REGION Network 8: IMMEDIATE STOP & STOP END OF CYCLE ALARMS
   RUNG wire#powerrail
      I_Contact( #interlocksDB.PROGRAM_SELCT_ALARM )
      Not()
      { S7_GenerateENO := "TRUE" } Move(in := #DB_NUMBER, out1 => "DB440_MACHINE_ALARM_DECODING".GLOBAL_ALARMS_MACHINE.ALARM_DECODING)
      wire#w1
      { S7_Templates := "SrcType := Int" } EQ_Contact(in1 := #CHANNEL, in2 := 1)
      wire#w2
      S_Coil( "DB440_MACHINE_ALARM_DECODING".ALARMS_UNIT_1.ST0_TRANSFER.IS_SEOC_ALARMS )
   END_RUNG
   RUNG wire#w2
      S_Coil( "DB440_MACHINE_ALARM_DECODING".ALARMS_UNIT_1.ST1_LOAD_UNLOAD.IS_SEOC_ALARMS )
   END_RUNG
   RUNG wire#w1
      { S7_Templates := "SrcType := Int" } EQ_Contact(in1 := #CHANNEL, in2 := 2)
      S_Coil( "DB440_MACHINE_ALARM_DECODING".ALARMS_UNIT_1.ST3_CLADDING.IS_SEOC_ALARMS )
   END_RUNG
   RUNG wire#w1
      { S7_Templates := "SrcType := Int" } EQ_Contact(in1 := #CHANNEL, in2 := 3)
      S_Coil( "DB440_MACHINE_ALARM_DECODING".ALARMS_UNIT_1.ST4_CLEANING.IS_SEOC_ALARMS )
   END_RUNG
   RUNG wire#w1
      { S7_Templates := "SrcType := Int" } EQ_Contact(in1 := #CHANNEL, in2 := 4)
      wire#w3
      S_Coil( "DB440_MACHINE_ALARM_DECODING".ALARMS_UNIT_2.ST0_TRANSFER.IS_SEOC_ALARMS )
   END_RUNG
   RUNG wire#w3
      S_Coil( "DB440_MACHINE_ALARM_DECODING".ALARMS_UNIT_2.ST1_LOAD_UNLOAD.IS_SEOC_ALARMS )
   END_RUNG
   RUNG wire#w1
      { S7_Templates := "SrcType := Int" } EQ_Contact(in1 := #CHANNEL, in2 := 5)
      S_Coil( "DB440_MACHINE_ALARM_DECODING".ALARMS_UNIT_2.ST2_MEASURING.IS_SEOC_ALARMS )
   END_RUNG
   RUNG wire#w1
      { S7_Templates := "SrcType := Int" } EQ_Contact(in1 := #CHANNEL, in2 := 6)
      S_Coil( "DB440_MACHINE_ALARM_DECODING".ALARMS_UNIT_2.ST3_CLADDING.IS_SEOC_ALARMS )
   END_RUNG
   RUNG wire#w1
      { S7_Templates := "SrcType := Int" } EQ_Contact(in1 := #CHANNEL, in2 := 7)
      S_Coil( "DB440_MACHINE_ALARM_DECODING".ALARMS_UNIT_2.ST4_CLEANING.IS_SEOC_ALARMS )
   END_RUNG
   RUNG wire#w1
      { S7_Templates := "SrcType := Int" } EQ_Contact(in1 := #CHANNEL, in2 := 8)
      S_Coil( "DB440_MACHINE_ALARM_DECODING".ALARMS_UNIT_3.IS_SEOC_ALARMS )
   END_RUNG
   RUNG wire#w1
      { S7_Templates := "SrcType := Int" } EQ_Contact(in1 := #CHANNEL, in2 := 9)
      S_Coil( "DB440_MACHINE_ALARM_DECODING".ALARMS_UNIT_4.IS_SEOC_ALARMS )
   END_RUNG
   // the same network as SCL:
   // ENO of a box is taken as its EN; it also drops when the box reports an error
   #_w1 := NOT (NOT #interlocksDB.PROGRAM_SELCT_ALARM);
   IF #_w1 THEN "DB440_MACHINE_ALARM_DECODING".GLOBAL_ALARMS_MACHINE.ALARM_DECODING := #DB_NUMBER; END_IF;
   IF #_w1 AND (#CHANNEL = 1) THEN
       "DB440_MACHINE_ALARM_DECODING".ALARMS_UNIT_1.ST0_TRANSFER.IS_SEOC_ALARMS := TRUE;
       "DB440_MACHINE_ALARM_DECODING".ALARMS_UNIT_1.ST1_LOAD_UNLOAD.IS_SEOC_ALARMS := TRUE;
   END_IF;
   IF #_w1 AND (#CHANNEL = 2) THEN
       "DB440_MACHINE_ALARM_DECODING".ALARMS_UNIT_1.ST3_CLADDING.IS_SEOC_ALARMS := TRUE;
   END_IF;
   IF #_w1 AND (#CHANNEL = 3) THEN
       "DB440_MACHINE_ALARM_DECODING".ALARMS_UNIT_1.ST4_CLEANING.IS_SEOC_ALARMS := TRUE;
   END_IF;
   IF #_w1 AND (#CHANNEL = 4) THEN
       "DB440_MACHINE_ALARM_DECODING".ALARMS_UNIT_2.ST0_TRANSFER.IS_SEOC_ALARMS := TRUE;
       "DB440_MACHINE_ALARM_DECODING".ALARMS_UNIT_2.ST1_LOAD_UNLOAD.IS_SEOC_ALARMS := TRUE;
   END_IF;
   IF #_w1 AND (#CHANNEL = 5) THEN
       "DB440_MACHINE_ALARM_DECODING".ALARMS_UNIT_2.ST2_MEASURING.IS_SEOC_ALARMS := TRUE;
   END_IF;
   IF #_w1 AND (#CHANNEL = 6) THEN
       "DB440_MACHINE_ALARM_DECODING".ALARMS_UNIT_2.ST3_CLADDING.IS_SEOC_ALARMS := TRUE;
   END_IF;
   IF #_w1 AND (#CHANNEL = 7) THEN
       "DB440_MACHINE_ALARM_DECODING".ALARMS_UNIT_2.ST4_CLEANING.IS_SEOC_ALARMS := TRUE;
   END_IF;
   IF #_w1 AND (#CHANNEL = 8) THEN
       "DB440_MACHINE_ALARM_DECODING".ALARMS_UNIT_3.IS_SEOC_ALARMS := TRUE;
   END_IF;
   IF #_w1 AND (#CHANNEL = 9) THEN
       "DB440_MACHINE_ALARM_DECODING".ALARMS_UNIT_4.IS_SEOC_ALARMS := TRUE;
   END_IF;
END_REGION

REGION Network 9: PROGRAMMING ALARM
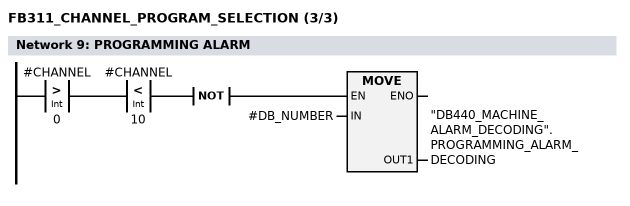
   RUNG wire#powerrail
      { S7_Templates := "SrcType := Int" } GT_Contact(in1 := #CHANNEL, in2 := 0)
      { S7_Templates := "SrcType := Int" } LT_Contact(in1 := #CHANNEL, in2 := 10)
      Not()
      Move(in := #DB_NUMBER, out1 => "DB440_MACHINE_ALARM_DECODING".PROGRAMMING_ALARM_DECODING)
   END_RUNG
   // the same network as SCL:
   IF NOT ((#CHANNEL > 0) AND (#CHANNEL < 10)) THEN
       "DB440_MACHINE_ALARM_DECODING".PROGRAMMING_ALARM_DECODING := #DB_NUMBER;
   END_IF;
END_REGION
END_FUNCTION_BLOCK

FUNCTION_BLOCK "FB321_CHANNEL"   // FB321, LAD
{ S7_Optimized_Access := 'FALSE' }
AUTHOR : ETXETAR
VERSION : 1.0
// stored: AutoNumber false, IsIECCheckEnabled false, SetENOAutomatically false, UDAEnableTagReadback false
   VAR_INPUT
      CHANNEL_MODE_GROUP : Int;   // CHANNEL MODE GROUP
      JERK_PARAMETERS_ENABLE { ExternalAccessible := 'False'; ExternalVisible := 'False'; ExternalWritable := 'False'} : Bool;   // JERK PARAMETERS ENABLE
      ENABLE_M01 { ExternalAccessible := 'False'; ExternalVisible := 'False'; ExternalWritable := 'False'} : Bool;   // ENABLE M01
      ENABLE_DRY_RUN_TEST_PRGM { ExternalAccessible := 'False'; ExternalVisible := 'False'; ExternalWritable := 'False'} : Bool;   // ENABLE DRY RUN TEST PRGM
      FEED_DISABLE { ExternalAccessible := 'False'; ExternalVisible := 'False'; ExternalWritable := 'False'} : Bool;   // FEED DISABLE
      ENABLE_OVERRIDE { ExternalAccessible := 'False'; ExternalVisible := 'False'; ExternalWritable := 'False'} : Bool;   // OVERRIDE 0 OR 100 =0 // OVERRIDE ENABLED =1
      ENABLE_OVERRIDE_FROM_MP_OR_HT10 { ExternalAccessible := 'False'; ExternalVisible := 'False'; ExternalWritable := 'False'} : Bool;   // ENABLE OVERRIDE FROM MAIN PANEL OR HT10, TRUE = YES, FALSE = NO (VALUE IS OBTAINED FROM AN HMI SCREEN OR ANOTHER DEVICE)
      OVERRIDE_VALUE : Byte;   // OVERRIDE VALUE
      BA3_SOFTKEYS_STOP { ExternalAccessible := 'False'; ExternalVisible := 'False'; ExternalWritable := 'False'} : Bool;   // BA3 SOFTKEYS STOP
      PROG_SLECT_FAULT_CH { ExternalAccessible := 'False'; ExternalVisible := 'False'; ExternalWritable := 'False'} : Bool;   // N.O / PROGRAM SELECTION FAULT CH
      MACHINE_IS_ALARMS : Bool;   // MACHINE IS ALARMS
      MACHINE_IS_WARNINGS : Bool;   // MACHINE IS WARNINGS
      UNIT_IS_SEOC { ExternalAccessible := 'False'; ExternalVisible := 'False'; ExternalWritable := 'False'} : Bool;   // UNIT IS SEOC
      CHANNEL_M201 { ExternalAccessible := 'False'; ExternalVisible := 'False'; ExternalWritable := 'False'} : Bool;   // CHANNEL M201
      CHANNEL_MCH_RESET : Bool;   // CHANNEL MACHINE RESET
      NC_START_DUMMY_FOR_OPT { ExternalAccessible := 'False'; ExternalVisible := 'False'; ExternalWritable := 'False'} : Bool;   // NC START DUMMY FOR OPTIMIZATION
      MPP_PUSH_BUTTON_START { ExternalAccessible := 'False'; ExternalVisible := 'False'; ExternalWritable := 'False'} : Bool;   // MPP PUSH BUTTON START
      MPP_PUSH_BUTTON_NC_START : Bool;   // MPP PUSH BUTTON NC START
      MPP_BUTTON_HOME_POS { ExternalAccessible := 'False'; ExternalVisible := 'False'; ExternalWritable := 'False'} : Bool;   // MPP BUTTON HOME POSITION
      UNIT_HOME_STEP_3 { ExternalAccessible := 'False'; ExternalVisible := 'False'; ExternalWritable := 'False'} : Bool;   // UNIT HOME STEP 3
      UNIT_CYCLE_STEP_3 { ExternalAccessible := 'False'; ExternalVisible := 'False'; ExternalWritable := 'False'} : Bool;   // UNIT CYCLE STEP 3
   END_VAR
   VAR_OUTPUT
      "CH_NOT_IN SOFT_MODE_ALARM" { ExternalAccessible := 'False'; ExternalVisible := 'False'; ExternalWritable := 'False'} : Bool;   // CHANNEL NOT IN SOFT MODE ALARM
   END_VAR
   VAR_IN_OUT
      ChannelDB : "LBP_typeChanX";
   END_VAR
   VAR DB_SPECIFIC
      CH_NOT_IN_SOFT_MODE { ExternalAccessible := 'False'; ExternalVisible := 'False'; ExternalWritable := 'False'} : Bool;   // CHANNEL NOT IN SOFT MODE
      RESET_CH { ExternalAccessible := 'False'; ExternalVisible := 'False'; ExternalWritable := 'False'} : Bool;   // RESET CHANNEL
      START_CH { ExternalAccessible := 'False'; ExternalVisible := 'False'; ExternalWritable := 'False'} : Bool;   // START CHANNEL
      RESET_AUX { ExternalAccessible := 'False'; ExternalVisible := 'False'; ExternalWritable := 'False'} : Bool;   // RESET AUX
      RESET_1 { ExternalAccessible := 'False'; ExternalVisible := 'False'; ExternalWritable := 'False'} : Bool;   // RESET 1
      RESET_2 { ExternalAccessible := 'False'; ExternalVisible := 'False'; ExternalWritable := 'False'} : Bool;   // RESET 2
      PULSE { ExternalAccessible := 'False'; ExternalVisible := 'False'; ExternalWritable := 'False'} : Bool;   // PULSE
      TIMER_CH_NOT_IN_SOFT_MODE { ExternalAccessible := 'False'; ExternalVisible := 'False'; ExternalWritable := 'False'; S7_SetPoint := 'True'} : TON_TIME;   // CHANNEL NOT IN SOFT MODE TIMER
   END_VAR
   VAR_TEMP
      DB_NUMBER : DInt;   // DB NUMBER FOR ALARM AND HELP DECODING
      CHANNEL_NUM : Int;   // CHANNEL NUMBER
   END_VAR
   // TIMER_CH_NOT_IN_SOFT_MODE.PT := T#1s;
   VAR_TEMP   // added for the SCL form of the ladder/FBD networks
      _w1 : Bool;
      _w2 : Bool;
   END_VAR
BEGIN

NETWORK
TITLE = READ INSTANCE DB
      L     DINO;
      +     10#800000;
      T     #DB_NUMBER;
//READ CHANNEL NUMBER
      L     DINO;
      L     10#320;
      -I;
      T     #CHANNEL_NUM;


REGION Network 2: ACTIVATE SINGLE BLOCK / ENABLE SINGLE BLOCK
   // Step by Step mode
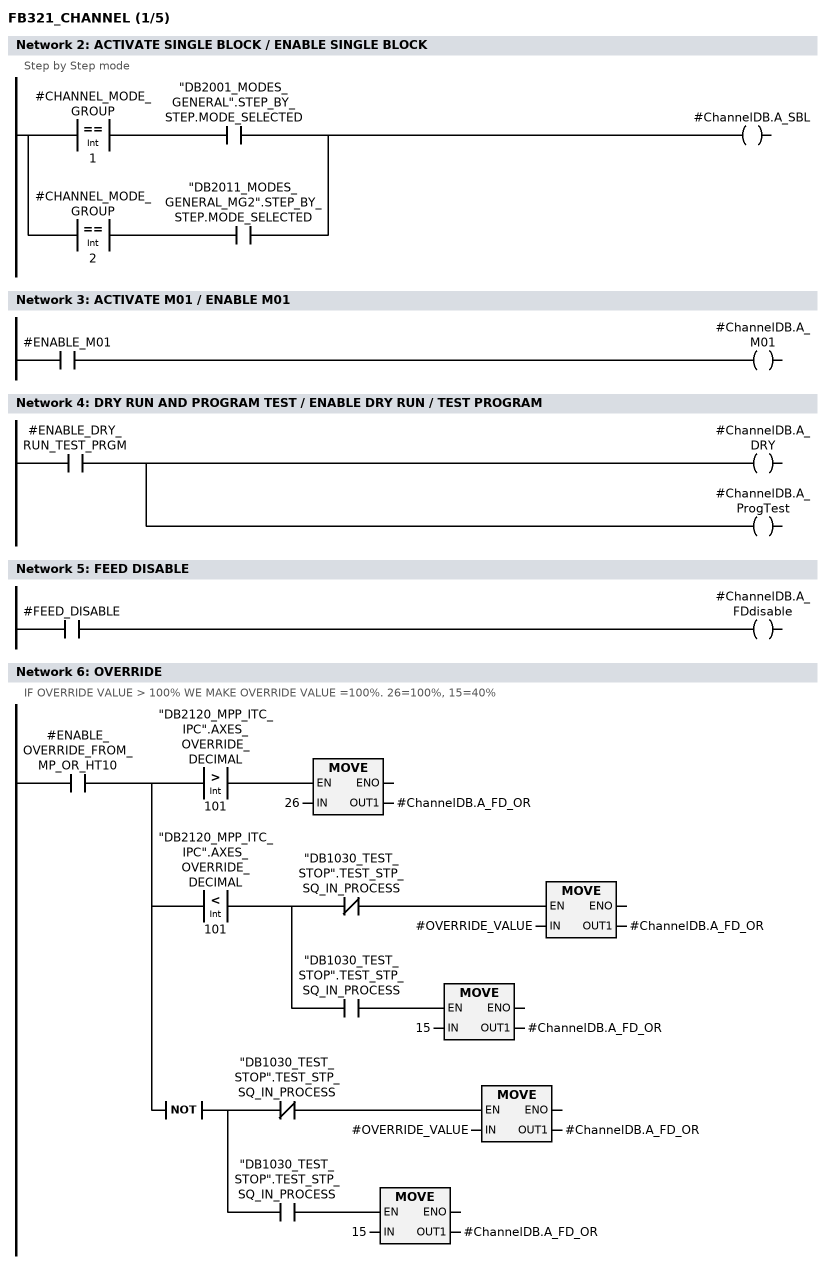
   RUNG wire#powerrail
      { S7_Templates := "SrcType := Int" } EQ_Contact(in1 := #CHANNEL_MODE_GROUP, in2 := 1)
      Contact( "DB2001_MODES_GENERAL".STEP_BY_STEP.MODE_SELECTED )
      wire#w1
      Coil( #ChannelDB.A_SBL )
   END_RUNG
   RUNG wire#powerrail
      { S7_Templates := "SrcType := Int" } EQ_Contact(in1 := #CHANNEL_MODE_GROUP, in2 := 2)
      Contact( "DB2011_MODES_GENERAL_MG2".STEP_BY_STEP.MODE_SELECTED )
   END_RUNG wire#w1
   // the same network as SCL:
   #ChannelDB.A_SBL := ((#CHANNEL_MODE_GROUP = 1) AND "DB2001_MODES_GENERAL".STEP_BY_STEP.MODE_SELECTED) OR ((#CHANNEL_MODE_GROUP = 2) AND "DB2011_MODES_GENERAL_MG2".STEP_BY_STEP.MODE_SELECTED);
END_REGION

REGION Network 3: ACTIVATE M01 / ENABLE M01
   RUNG wire#powerrail
      Contact( #ENABLE_M01 )
      Coil( #ChannelDB.A_M01 )
   END_RUNG
   // the same network as SCL:
   #ChannelDB.A_M01 := #ENABLE_M01;
END_REGION

REGION Network 4: DRY RUN AND PROGRAM TEST / ENABLE DRY RUN / TEST PROGRAM
   RUNG wire#powerrail
      Contact( #ENABLE_DRY_RUN_TEST_PRGM )
      wire#w1
      Coil( #ChannelDB.A_DRY )
   END_RUNG
   RUNG wire#w1
      Coil( #ChannelDB.A_ProgTest )
   END_RUNG
   // the same network as SCL:
   #ChannelDB.A_DRY := #ENABLE_DRY_RUN_TEST_PRGM;
   #ChannelDB.A_ProgTest := #ENABLE_DRY_RUN_TEST_PRGM;
END_REGION

REGION Network 5: FEED DISABLE
   RUNG wire#powerrail
      Contact( #FEED_DISABLE )
      Coil( #ChannelDB.A_FDdisable )
   END_RUNG
   // the same network as SCL:
   #ChannelDB.A_FDdisable := #FEED_DISABLE;
END_REGION

REGION Network 6: OVERRIDE
   // IF OVERRIDE VALUE > 100% WE MAKE OVERRIDE VALUE =100%. 26=100%, 15=40%
   RUNG wire#powerrail
      Contact( #ENABLE_OVERRIDE_FROM_MP_OR_HT10 )
      wire#w1
      { S7_Templates := "SrcType := Int" } GT_Contact(in1 := "DB2120_MPP_ITC_IPC".AXES_OVERRIDE_DECIMAL, in2 := 101)
      { S7_GenerateENO := "TRUE" } Move(in := 26, out1 => #ChannelDB.A_FD_OR)
   END_RUNG
   RUNG wire#w1
      { S7_Templates := "SrcType := Int" } LT_Contact(in1 := "DB2120_MPP_ITC_IPC".AXES_OVERRIDE_DECIMAL, in2 := 101)
      wire#w2
      I_Contact( "DB1030_TEST_STOP".TEST_STP_SQ_IN_PROCESS )
      { S7_GenerateENO := "TRUE" } Move(in := #OVERRIDE_VALUE, out1 => #ChannelDB.A_FD_OR)
   END_RUNG
   RUNG wire#w2
      Contact( "DB1030_TEST_STOP".TEST_STP_SQ_IN_PROCESS )
      { S7_GenerateENO := "TRUE" } Move(in := 15, out1 => #ChannelDB.A_FD_OR)
   END_RUNG
   RUNG wire#w1
      Not()
      wire#w3
      I_Contact( "DB1030_TEST_STOP".TEST_STP_SQ_IN_PROCESS )
      { S7_GenerateENO := "TRUE" } Move(in := #OVERRIDE_VALUE, out1 => #ChannelDB.A_FD_OR)
   END_RUNG
   RUNG wire#w3
      Contact( "DB1030_TEST_STOP".TEST_STP_SQ_IN_PROCESS )
      { S7_GenerateENO := "TRUE" } Move(in := 15, out1 => #ChannelDB.A_FD_OR)
   END_RUNG
   // the same network as SCL:
   IF #ENABLE_OVERRIDE_FROM_MP_OR_HT10 AND ("DB2120_MPP_ITC_IPC".AXES_OVERRIDE_DECIMAL > 101) THEN
       #ChannelDB.A_FD_OR := 26;
   END_IF;
   #_w1 := #ENABLE_OVERRIDE_FROM_MP_OR_HT10 AND ("DB2120_MPP_ITC_IPC".AXES_OVERRIDE_DECIMAL < 101);
   IF #_w1 AND NOT "DB1030_TEST_STOP".TEST_STP_SQ_IN_PROCESS THEN
       #ChannelDB.A_FD_OR := #OVERRIDE_VALUE;
   END_IF;
   IF #_w1 AND "DB1030_TEST_STOP".TEST_STP_SQ_IN_PROCESS THEN #ChannelDB.A_FD_OR := 15; END_IF;
   #_w2 := NOT #ENABLE_OVERRIDE_FROM_MP_OR_HT10;
   IF #_w2 AND NOT "DB1030_TEST_STOP".TEST_STP_SQ_IN_PROCESS THEN
       #ChannelDB.A_FD_OR := #OVERRIDE_VALUE;
   END_IF;
   IF #_w2 AND "DB1030_TEST_STOP".TEST_STP_SQ_IN_PROCESS THEN #ChannelDB.A_FD_OR := 15; END_IF;
END_REGION

REGION Network 7: OVERRIDE ACTIVE / FEEDRATE OVERRIDE ACTIVE
   // REMOVE DUMMY ON IF REQUIRED
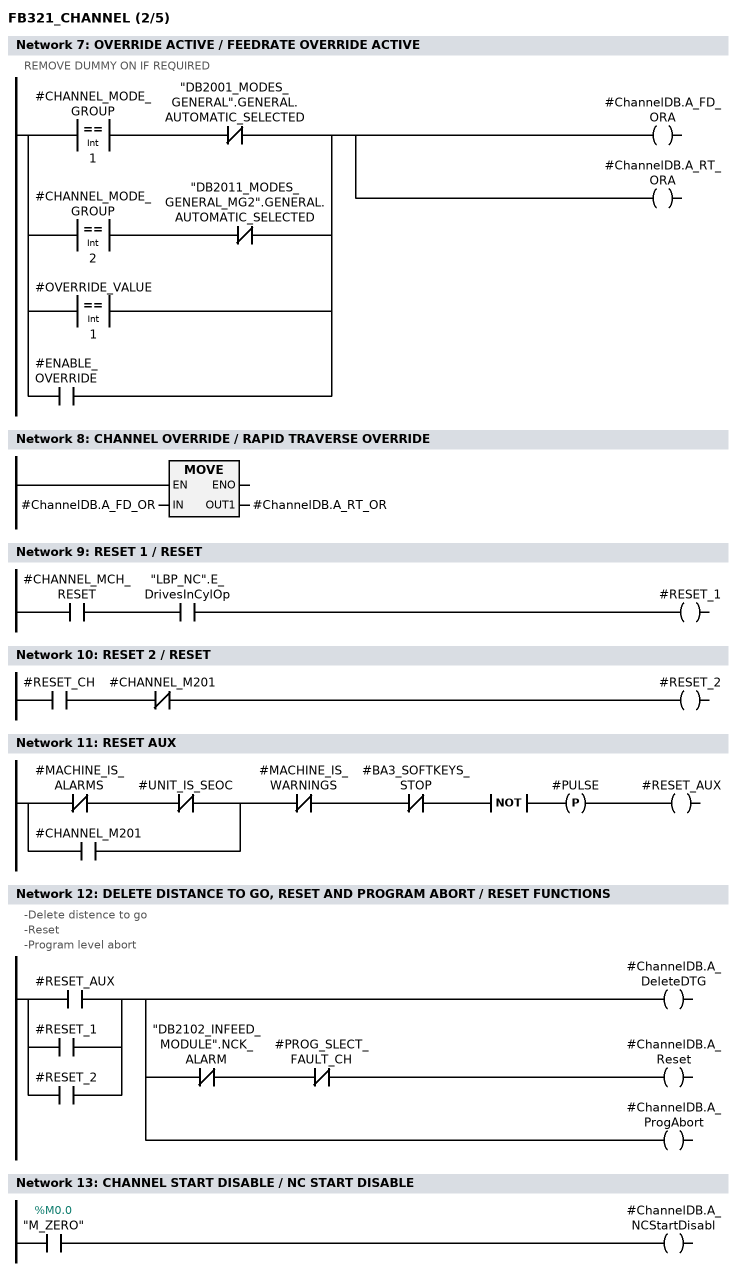
   RUNG wire#powerrail
      { S7_Templates := "SrcType := Int" } EQ_Contact(in1 := #CHANNEL_MODE_GROUP, in2 := 1)
      I_Contact( "DB2001_MODES_GENERAL".GENERAL.AUTOMATIC_SELECTED )
      wire#w1
      Coil( #ChannelDB.A_FD_ORA )
   END_RUNG
   RUNG wire#powerrail
      { S7_Templates := "SrcType := Int" } EQ_Contact(in1 := #CHANNEL_MODE_GROUP, in2 := 2)
      I_Contact( "DB2011_MODES_GENERAL_MG2".GENERAL.AUTOMATIC_SELECTED )
   END_RUNG wire#w1
   RUNG wire#powerrail
      { S7_Templates := "SrcType := Int" } EQ_Contact(in1 := #OVERRIDE_VALUE, in2 := 1)
   END_RUNG wire#w1
   RUNG wire#powerrail
      Contact( #ENABLE_OVERRIDE )
   END_RUNG wire#w1
   RUNG wire#w1
      Coil( #ChannelDB.A_RT_ORA )
   END_RUNG
   // the same network as SCL:
   #ChannelDB.A_FD_ORA := ((#CHANNEL_MODE_GROUP = 1) AND NOT "DB2001_MODES_GENERAL".GENERAL.AUTOMATIC_SELECTED) OR ((#CHANNEL_MODE_GROUP = 2) AND NOT "DB2011_MODES_GENERAL_MG2".GENERAL.AUTOMATIC_SELECTED) OR (#OVERRIDE_VALUE = 1) OR #ENABLE_OVERRIDE;
   #ChannelDB.A_RT_ORA := #ChannelDB.A_FD_ORA;
END_REGION

REGION Network 8: CHANNEL OVERRIDE / RAPID TRAVERSE OVERRIDE
   RUNG wire#powerrail
      { S7_GenerateENO := "TRUE" } Move(in := #ChannelDB.A_FD_OR, out1 => #ChannelDB.A_RT_OR)
   END_RUNG
   // the same network as SCL:
   #ChannelDB.A_RT_OR := #ChannelDB.A_FD_OR;
END_REGION

REGION Network 9: RESET 1 / RESET
   RUNG wire#powerrail
      Contact( #CHANNEL_MCH_RESET )
      Contact( "LBP_NC".E_DrivesInCylOp )
      Coil( #RESET_1 )
   END_RUNG
   // the same network as SCL:
   #RESET_1 := #CHANNEL_MCH_RESET AND "LBP_NC".E_DrivesInCylOp;
END_REGION

REGION Network 10: RESET 2 / RESET
   RUNG wire#powerrail
      Contact( #RESET_CH )
      I_Contact( #CHANNEL_M201 )
      Coil( #RESET_2 )
   END_RUNG
   // the same network as SCL:
   #RESET_2 := #RESET_CH AND NOT #CHANNEL_M201;
END_REGION

REGION Network 11: RESET AUX
   RUNG wire#powerrail
      I_Contact( #MACHINE_IS_ALARMS )
      I_Contact( #UNIT_IS_SEOC )
      wire#w1
      I_Contact( #MACHINE_IS_WARNINGS )
      I_Contact( #BA3_SOFTKEYS_STOP )
      Not()
      P_Trig( #PULSE )
      Coil( #RESET_AUX )
   END_RUNG
   RUNG wire#powerrail
      Contact( #CHANNEL_M201 )
   END_RUNG wire#w1
   // the same network as SCL:
   #_w1 := NOT (((NOT #MACHINE_IS_ALARMS AND NOT #UNIT_IS_SEOC) OR #CHANNEL_M201) AND NOT #MACHINE_IS_WARNINGS AND NOT #BA3_SOFTKEYS_STOP);
   #_w2 := #_w1 AND NOT #PULSE;   // rising edge
   #PULSE := #_w1;
   #RESET_AUX := #_w2;
END_REGION

REGION Network 12: DELETE DISTANCE TO GO, RESET AND PROGRAM ABORT / RESET FUNCTIONS
   // -Delete distence to go
   // -Reset
   // -Program level abort
   RUNG wire#powerrail
      Contact( #RESET_AUX )
      wire#w1
      Coil( #ChannelDB.A_DeleteDTG )
   END_RUNG
   RUNG wire#powerrail
      Contact( #RESET_1 )
   END_RUNG wire#w1
   RUNG wire#powerrail
      Contact( #RESET_2 )
   END_RUNG wire#w1
   RUNG wire#w1
      I_Contact( "DB2102_INFEED_MODULE".NCK_ALARM )
      I_Contact( #PROG_SLECT_FAULT_CH )
      Coil( #ChannelDB.A_Reset )
   END_RUNG
   RUNG wire#w1
      Coil( #ChannelDB.A_ProgAbort )
   END_RUNG
   // the same network as SCL:
   #ChannelDB.A_DeleteDTG := #RESET_AUX OR #RESET_1 OR #RESET_2;
   #ChannelDB.A_Reset := #ChannelDB.A_DeleteDTG AND NOT "DB2102_INFEED_MODULE".NCK_ALARM AND NOT #PROG_SLECT_FAULT_CH;
   #ChannelDB.A_ProgAbort := #ChannelDB.A_DeleteDTG;
END_REGION

REGION Network 13: CHANNEL START DISABLE / NC START DISABLE
   RUNG wire#powerrail
      Contact( "M_ZERO" )
      Coil( #ChannelDB.A_NCStartDisabl )
   END_RUNG
   // the same network as SCL:
   #ChannelDB.A_NCStartDisabl := "M_ZERO";
END_REGION

REGION Network 14: START CHANNEL / NC START
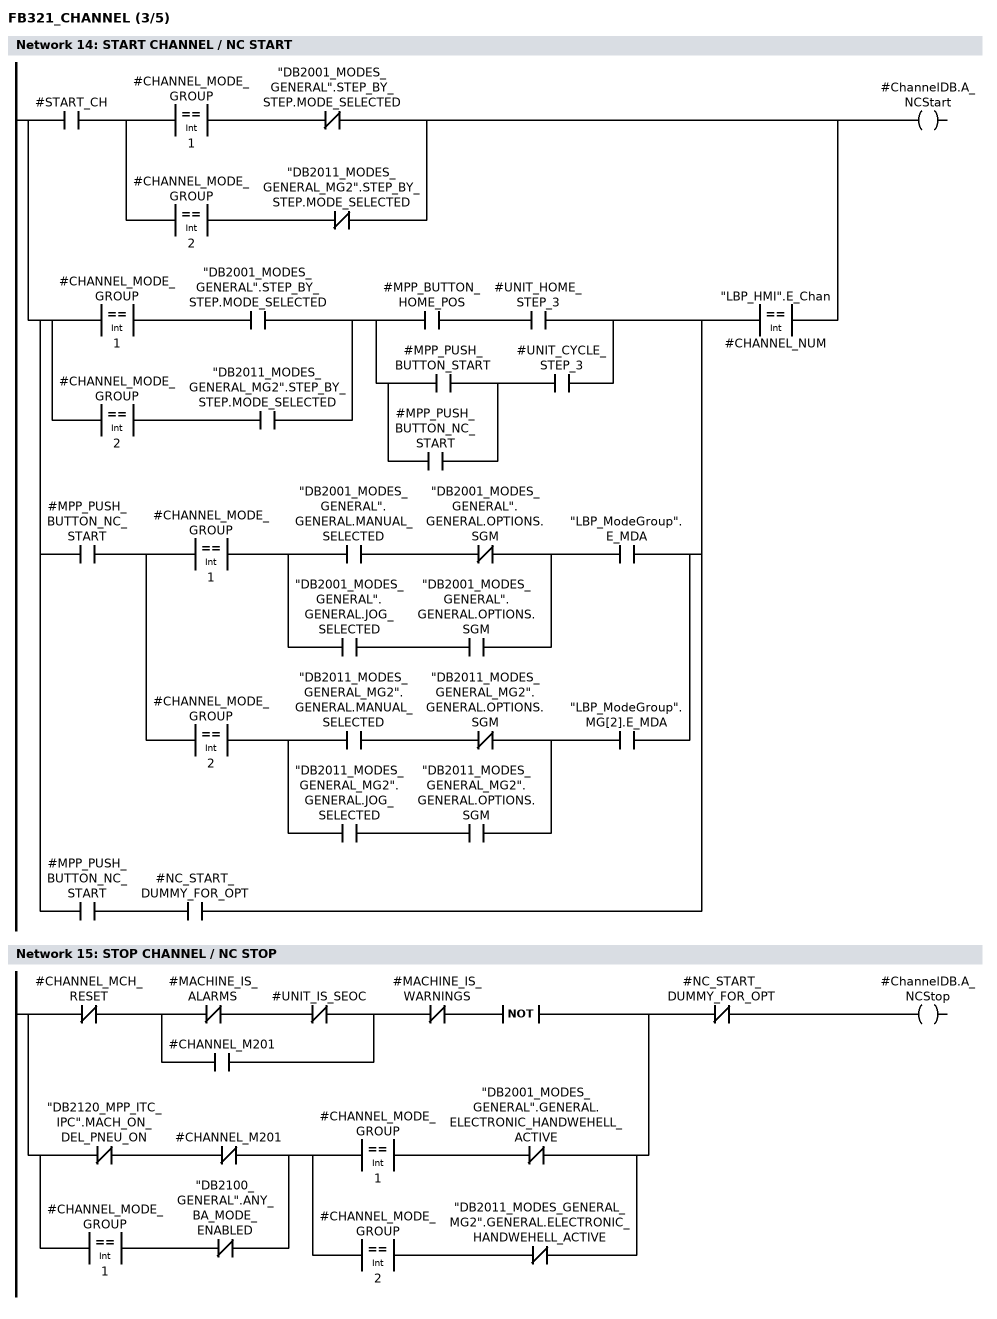
   RUNG wire#powerrail
      Contact( #START_CH )
      wire#w1
      { S7_Templates := "SrcType := Int" } EQ_Contact(in1 := #CHANNEL_MODE_GROUP, in2 := 1)
      I_Contact( "DB2001_MODES_GENERAL".STEP_BY_STEP.MODE_SELECTED )
      wire#w2
      Coil( #ChannelDB.A_NCStart )
   END_RUNG
   RUNG wire#w1
      { S7_Templates := "SrcType := Int" } EQ_Contact(in1 := #CHANNEL_MODE_GROUP, in2 := 2)
      I_Contact( "DB2011_MODES_GENERAL_MG2".STEP_BY_STEP.MODE_SELECTED )
   END_RUNG wire#w2
   RUNG wire#powerrail
      { S7_Templates := "SrcType := Int" } EQ_Contact(in1 := #CHANNEL_MODE_GROUP, in2 := 1)
      Contact( "DB2001_MODES_GENERAL".STEP_BY_STEP.MODE_SELECTED )
      wire#w3
      Contact( #MPP_BUTTON_HOME_POS )
      Contact( #UNIT_HOME_STEP_3 )
      wire#w4
      { S7_Templates := "SrcType := Int" } EQ_Contact(in1 := "LBP_HMI".E_Chan, in2 := #CHANNEL_NUM)
   END_RUNG wire#w2
   RUNG wire#powerrail
      { S7_Templates := "SrcType := Int" } EQ_Contact(in1 := #CHANNEL_MODE_GROUP, in2 := 2)
      Contact( "DB2011_MODES_GENERAL_MG2".STEP_BY_STEP.MODE_SELECTED )
   END_RUNG wire#w3
   RUNG wire#w3
      Contact( #MPP_PUSH_BUTTON_START )
      wire#w5
      Contact( #UNIT_CYCLE_STEP_3 )
   END_RUNG wire#w4
   RUNG wire#w3
      Contact( #MPP_PUSH_BUTTON_NC_START )
   END_RUNG wire#w5
   RUNG wire#powerrail
      Contact( #MPP_PUSH_BUTTON_NC_START )
      wire#w6
      { S7_Templates := "SrcType := Int" } EQ_Contact(in1 := #CHANNEL_MODE_GROUP, in2 := 1)
      wire#w7
      Contact( "DB2001_MODES_GENERAL".GENERAL.MANUAL_SELECTED )
      I_Contact( "DB2001_MODES_GENERAL".GENERAL.OPTIONS.SGM )
      wire#w8
      Contact( "LBP_ModeGroup".E_MDA )
   END_RUNG wire#w4
   RUNG wire#w7
      Contact( "DB2001_MODES_GENERAL".GENERAL.JOG_SELECTED )
      Contact( "DB2001_MODES_GENERAL".GENERAL.OPTIONS.SGM )
   END_RUNG wire#w8
   RUNG wire#w6
      { S7_Templates := "SrcType := Int" } EQ_Contact(in1 := #CHANNEL_MODE_GROUP, in2 := 2)
      wire#w9
      Contact( "DB2011_MODES_GENERAL_MG2".GENERAL.MANUAL_SELECTED )
      I_Contact( "DB2011_MODES_GENERAL_MG2".GENERAL.OPTIONS.SGM )
      wire#w10
      Contact( "LBP_ModeGroup".MG[2].E_MDA )
   END_RUNG wire#w4
   RUNG wire#w9
      Contact( "DB2011_MODES_GENERAL_MG2".GENERAL.JOG_SELECTED )
      Contact( "DB2011_MODES_GENERAL_MG2".GENERAL.OPTIONS.SGM )
   END_RUNG wire#w10
   RUNG wire#powerrail
      Contact( #MPP_PUSH_BUTTON_NC_START )
      Contact( #NC_START_DUMMY_FOR_OPT )
   END_RUNG wire#w4
   // the same network as SCL:
   #ChannelDB.A_NCStart := (#START_CH AND (((#CHANNEL_MODE_GROUP = 1) AND NOT "DB2001_MODES_GENERAL".STEP_BY_STEP.MODE_SELECTED) OR ((#CHANNEL_MODE_GROUP = 2) AND NOT "DB2011_MODES_GENERAL_MG2".STEP_BY_STEP.MODE_SELECTED))) OR ((((((#CHANNEL_MODE_GROUP = 1) AND "DB2001_MODES_GENERAL".STEP_BY_STEP.MODE_SELECTED) OR ((#CHANNEL_MODE_GROUP = 2) AND "DB2011_MODES_GENERAL_MG2".STEP_BY_STEP.MODE_SELECTED)) AND ((#MPP_BUTTON_HOME_POS AND #UNIT_HOME_STEP_3) OR ((#MPP_PUSH_BUTTON_START OR #MPP_PUSH_BUTTON_NC_START) AND #UNIT_CYCLE_STEP_3))) OR (#MPP_PUSH_BUTTON_NC_START AND (((#CHANNEL_MODE_GROUP = 1) AND (("DB2001_MODES_GENERAL".GENERAL.MANUAL_SELECTED AND NOT "DB2001_MODES_GENERAL".GENERAL.OPTIONS.SGM) OR ("DB2001_MODES_GENERAL".GENERAL.JOG_SELECTED AND "DB2001_MODES_GENERAL".GENERAL.OPTIONS.SGM)) AND "LBP_ModeGroup".E_MDA) OR ((#CHANNEL_MODE_GROUP = 2) AND (("DB2011_MODES_GENERAL_MG2".GENERAL.MANUAL_SELECTED AND NOT "DB2011_MODES_GENERAL_MG2".GENERAL.OPTIONS.SGM) OR ("DB2011_MODES_GENERAL_MG2".GENERAL.JOG_SELECTED AND "DB2011_MODES_GENERAL_MG2".GENERAL.OPTIONS.SGM)) AND "LBP_ModeGroup".MG[2].E_MDA))) OR (#MPP_PUSH_BUTTON_NC_START AND #NC_START_DUMMY_FOR_OPT)) AND ("LBP_HMI".E_Chan = #CHANNEL_NUM));
END_REGION

REGION Network 15: STOP CHANNEL / NC STOP
   RUNG wire#powerrail
      I_Contact( #CHANNEL_MCH_RESET )
      wire#w1
      I_Contact( #MACHINE_IS_ALARMS )
      I_Contact( #UNIT_IS_SEOC )
      wire#w2
      I_Contact( #MACHINE_IS_WARNINGS )
      Not()
      wire#w3
      I_Contact( #NC_START_DUMMY_FOR_OPT )
      Coil( #ChannelDB.A_NCStop )
   END_RUNG
   RUNG wire#w1
      Contact( #CHANNEL_M201 )
   END_RUNG wire#w2
   RUNG wire#powerrail
      I_Contact( "DB2120_MPP_ITC_IPC".MACH_ON_DEL_PNEU_ON )
      I_Contact( #CHANNEL_M201 )
      wire#w4
      { S7_Templates := "SrcType := Int" } EQ_Contact(in1 := #CHANNEL_MODE_GROUP, in2 := 1)
      I_Contact( "DB2001_MODES_GENERAL".GENERAL.ELECTRONIC_HANDWEHELL_ACTIVE )
   END_RUNG wire#w3
   RUNG wire#powerrail
      { S7_Templates := "SrcType := Int" } EQ_Contact(in1 := #CHANNEL_MODE_GROUP, in2 := 1)
      I_Contact( "DB2100_GENERAL".ANY_BA_MODE_ENABLED )
   END_RUNG wire#w4
   RUNG wire#w4
      { S7_Templates := "SrcType := Int" } EQ_Contact(in1 := #CHANNEL_MODE_GROUP, in2 := 2)
      I_Contact( "DB2011_MODES_GENERAL_MG2".GENERAL.ELECTRONIC_HANDWEHELL_ACTIVE )
   END_RUNG wire#w3
   // the same network as SCL:
   #ChannelDB.A_NCStop := (NOT (NOT #CHANNEL_MCH_RESET AND ((NOT #MACHINE_IS_ALARMS AND NOT #UNIT_IS_SEOC) OR #CHANNEL_M201) AND NOT #MACHINE_IS_WARNINGS) OR (((NOT "DB2120_MPP_ITC_IPC".MACH_ON_DEL_PNEU_ON AND NOT #CHANNEL_M201) OR ((#CHANNEL_MODE_GROUP = 1) AND NOT "DB2100_GENERAL".ANY_BA_MODE_ENABLED)) AND (((#CHANNEL_MODE_GROUP = 1) AND NOT "DB2001_MODES_GENERAL".GENERAL.ELECTRONIC_HANDWEHELL_ACTIVE) OR ((#CHANNEL_MODE_GROUP = 2) AND NOT "DB2011_MODES_GENERAL_MG2".GENERAL.ELECTRONIC_HANDWEHELL_ACTIVE)))) AND NOT #NC_START_DUMMY_FOR_OPT;
END_REGION

REGION Network 16: CHANNEL NOT IN SOFT MODE ALARM / SOFT MODE ACTIVE CHANNEL
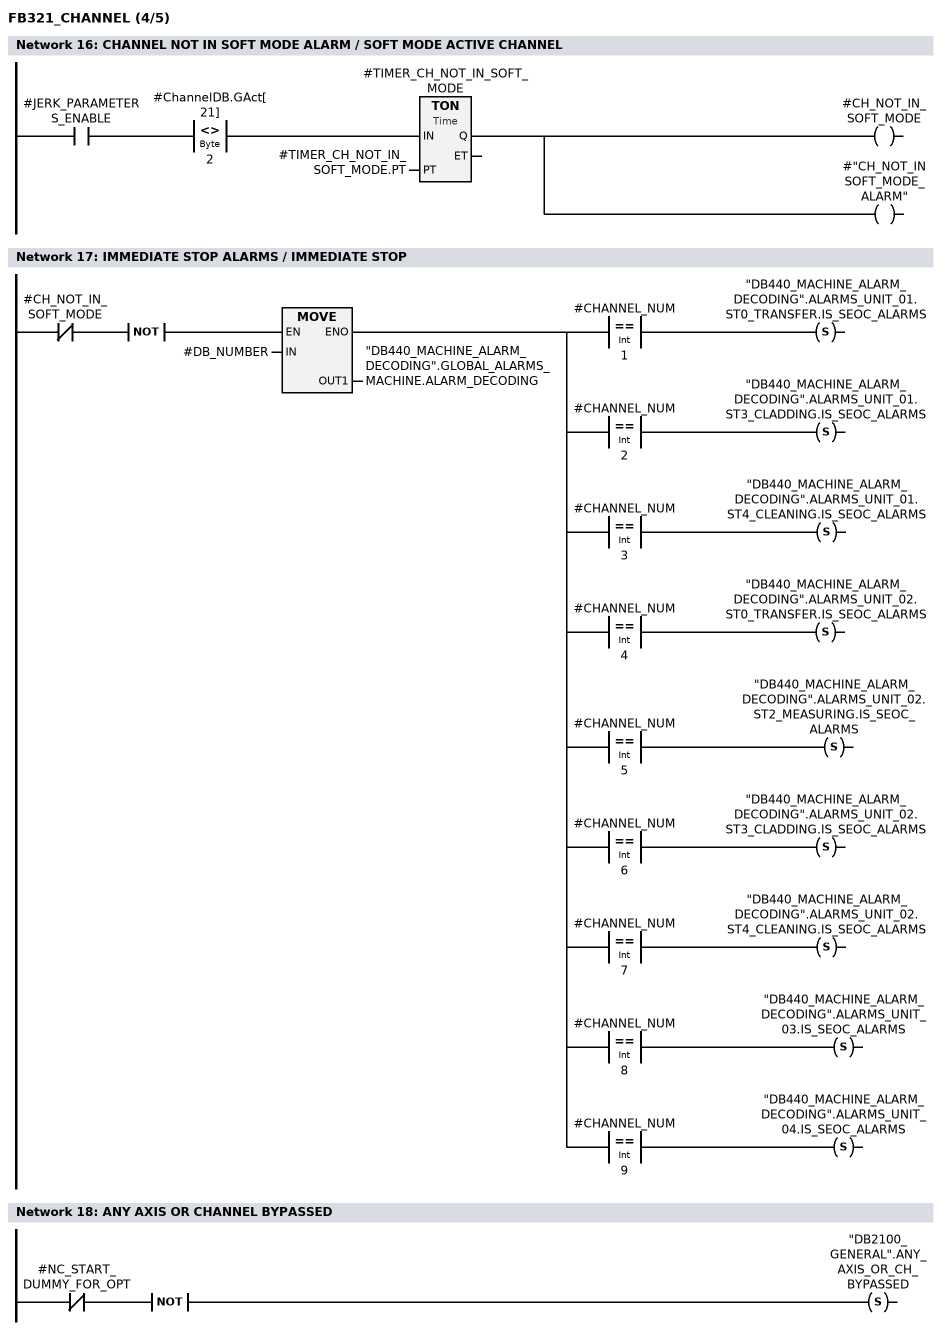
   RUNG wire#powerrail
      Contact( #JERK_PARAMETERS_ENABLE )
      { S7_Templates := "SrcType := Byte" } NE_Contact(in1 := #ChannelDB.GAct[21], in2 := 2)
      { S7_Templates := "time_type := Time" } #TIMER_CH_NOT_IN_SOFT_MODE.TON(pt := #TIMER_CH_NOT_IN_SOFT_MODE.PT, et =>)
      wire#w1
      Coil( #CH_NOT_IN_SOFT_MODE )
   END_RUNG
   RUNG wire#w1
      Coil( #"CH_NOT_IN SOFT_MODE_ALARM" )
   END_RUNG
   // the same network as SCL:
   #TIMER_CH_NOT_IN_SOFT_MODE(IN := #JERK_PARAMETERS_ENABLE AND (#ChannelDB.GAct[21] <> 2),   // TON
                           PT := #TIMER_CH_NOT_IN_SOFT_MODE.PT);
   #CH_NOT_IN_SOFT_MODE := #TIMER_CH_NOT_IN_SOFT_MODE.Q;
   #"CH_NOT_IN SOFT_MODE_ALARM" := #TIMER_CH_NOT_IN_SOFT_MODE.Q;
END_REGION

REGION Network 17: IMMEDIATE STOP ALARMS / IMMEDIATE STOP
   RUNG wire#powerrail
      I_Contact( #CH_NOT_IN_SOFT_MODE )
      Not()
      { S7_GenerateENO := "TRUE" } Move(in := #DB_NUMBER, out1 => "DB440_MACHINE_ALARM_DECODING".GLOBAL_ALARMS_MACHINE.ALARM_DECODING)
      wire#w1
      { S7_Templates := "SrcType := Int" } EQ_Contact(in1 := #CHANNEL_NUM, in2 := 1)
      S_Coil( "DB440_MACHINE_ALARM_DECODING".ALARMS_UNIT_01.ST0_TRANSFER.IS_SEOC_ALARMS )
   END_RUNG
   RUNG wire#w1
      { S7_Templates := "SrcType := Int" } EQ_Contact(in1 := #CHANNEL_NUM, in2 := 2)
      S_Coil( "DB440_MACHINE_ALARM_DECODING".ALARMS_UNIT_01.ST3_CLADDING.IS_SEOC_ALARMS )
   END_RUNG
   RUNG wire#w1
      { S7_Templates := "SrcType := Int" } EQ_Contact(in1 := #CHANNEL_NUM, in2 := 3)
      S_Coil( "DB440_MACHINE_ALARM_DECODING".ALARMS_UNIT_01.ST4_CLEANING.IS_SEOC_ALARMS )
   END_RUNG
   RUNG wire#w1
      { S7_Templates := "SrcType := Int" } EQ_Contact(in1 := #CHANNEL_NUM, in2 := 4)
      S_Coil( "DB440_MACHINE_ALARM_DECODING".ALARMS_UNIT_02.ST0_TRANSFER.IS_SEOC_ALARMS )
   END_RUNG
   RUNG wire#w1
      { S7_Templates := "SrcType := Int" } EQ_Contact(in1 := #CHANNEL_NUM, in2 := 5)
      S_Coil( "DB440_MACHINE_ALARM_DECODING".ALARMS_UNIT_02.ST2_MEASURING.IS_SEOC_ALARMS )
   END_RUNG
   RUNG wire#w1
      { S7_Templates := "SrcType := Int" } EQ_Contact(in1 := #CHANNEL_NUM, in2 := 6)
      S_Coil( "DB440_MACHINE_ALARM_DECODING".ALARMS_UNIT_02.ST3_CLADDING.IS_SEOC_ALARMS )
   END_RUNG
   RUNG wire#w1
      { S7_Templates := "SrcType := Int" } EQ_Contact(in1 := #CHANNEL_NUM, in2 := 7)
      S_Coil( "DB440_MACHINE_ALARM_DECODING".ALARMS_UNIT_02.ST4_CLEANING.IS_SEOC_ALARMS )
   END_RUNG
   RUNG wire#w1
      { S7_Templates := "SrcType := Int" } EQ_Contact(in1 := #CHANNEL_NUM, in2 := 8)
      S_Coil( "DB440_MACHINE_ALARM_DECODING".ALARMS_UNIT_03.IS_SEOC_ALARMS )
   END_RUNG
   RUNG wire#w1
      { S7_Templates := "SrcType := Int" } EQ_Contact(in1 := #CHANNEL_NUM, in2 := 9)
      S_Coil( "DB440_MACHINE_ALARM_DECODING".ALARMS_UNIT_04.IS_SEOC_ALARMS )
   END_RUNG
   // the same network as SCL:
   // ENO of a box is taken as its EN; it also drops when the box reports an error
   #_w1 := NOT (NOT #CH_NOT_IN_SOFT_MODE);
   IF #_w1 THEN "DB440_MACHINE_ALARM_DECODING".GLOBAL_ALARMS_MACHINE.ALARM_DECODING := #DB_NUMBER; END_IF;
   IF #_w1 AND (#CHANNEL_NUM = 1) THEN
       "DB440_MACHINE_ALARM_DECODING".ALARMS_UNIT_01.ST0_TRANSFER.IS_SEOC_ALARMS := TRUE;
   END_IF;
   IF #_w1 AND (#CHANNEL_NUM = 2) THEN
       "DB440_MACHINE_ALARM_DECODING".ALARMS_UNIT_01.ST3_CLADDING.IS_SEOC_ALARMS := TRUE;
   END_IF;
   IF #_w1 AND (#CHANNEL_NUM = 3) THEN
       "DB440_MACHINE_ALARM_DECODING".ALARMS_UNIT_01.ST4_CLEANING.IS_SEOC_ALARMS := TRUE;
   END_IF;
   IF #_w1 AND (#CHANNEL_NUM = 4) THEN
       "DB440_MACHINE_ALARM_DECODING".ALARMS_UNIT_02.ST0_TRANSFER.IS_SEOC_ALARMS := TRUE;
   END_IF;
   IF #_w1 AND (#CHANNEL_NUM = 5) THEN
       "DB440_MACHINE_ALARM_DECODING".ALARMS_UNIT_02.ST2_MEASURING.IS_SEOC_ALARMS := TRUE;
   END_IF;
   IF #_w1 AND (#CHANNEL_NUM = 6) THEN
       "DB440_MACHINE_ALARM_DECODING".ALARMS_UNIT_02.ST3_CLADDING.IS_SEOC_ALARMS := TRUE;
   END_IF;
   IF #_w1 AND (#CHANNEL_NUM = 7) THEN
       "DB440_MACHINE_ALARM_DECODING".ALARMS_UNIT_02.ST4_CLEANING.IS_SEOC_ALARMS := TRUE;
   END_IF;
   IF #_w1 AND (#CHANNEL_NUM = 8) THEN
       "DB440_MACHINE_ALARM_DECODING".ALARMS_UNIT_03.IS_SEOC_ALARMS := TRUE;
   END_IF;
   IF #_w1 AND (#CHANNEL_NUM = 9) THEN
       "DB440_MACHINE_ALARM_DECODING".ALARMS_UNIT_04.IS_SEOC_ALARMS := TRUE;
   END_IF;
END_REGION

REGION Network 18: ANY AXIS OR CHANNEL BYPASSED
   RUNG wire#powerrail
      I_Contact( #NC_START_DUMMY_FOR_OPT )
      Not()
      S_Coil( "DB2100_GENERAL".ANY_AXIS_OR_CH_BYPASSED )
   END_RUNG
   // the same network as SCL:
   IF NOT (NOT #NC_START_DUMMY_FOR_OPT) THEN "DB2100_GENERAL".ANY_AXIS_OR_CH_BYPASSED := TRUE; END_IF;
END_REGION

REGION Network 19: PROGRAMMING ALARM
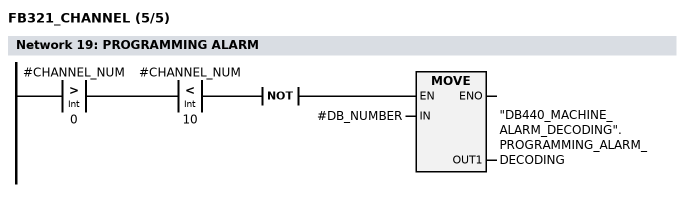
   RUNG wire#powerrail
      { S7_Templates := "SrcType := Int" } GT_Contact(in1 := #CHANNEL_NUM, in2 := 0)
      { S7_Templates := "SrcType := Int" } LT_Contact(in1 := #CHANNEL_NUM, in2 := 10)
      Not()
      Move(in := #DB_NUMBER, out1 => "DB440_MACHINE_ALARM_DECODING".PROGRAMMING_ALARM_DECODING)
   END_RUNG
   // the same network as SCL:
   IF NOT ((#CHANNEL_NUM > 0) AND (#CHANNEL_NUM < 10)) THEN
       "DB440_MACHINE_ALARM_DECODING".PROGRAMMING_ALARM_DECODING := #DB_NUMBER;
   END_IF;
END_REGION
END_FUNCTION_BLOCK

FUNCTION_BLOCK "FB331_M_CODE_EXTENDED"   // FB331, LAD
{ S7_Optimized_Access := 'FALSE' }
AUTHOR : ETXETAR
VERSION : 1.0
// stored: AutoNumber false, IsIECCheckEnabled false, SetENOAutomatically false, UDAEnableTagReadback false
   VAR_INPUT
      NC_Chan_Num_Chan : Int;   // Channel Number to monitoring
   END_VAR
   VAR DB_SPECIFIC
      INDEX : Int;
      M_code : Array[100..999] of Bool;   // EXTENDED M CODE
   END_VAR
   VAR_TEMP
      TEMP0 : Int;
      DB_Channel : Int;
      Inst_DB : Int;
   END_VAR
BEGIN

NETWORK
TITLE = READ DATA / Data block for monitoring channel

//DB from channel
      L     #NC_Chan_Num_Chan;
      +     20;
      T     #DB_Channel;
//set DB instance assigned to FB
      L     DINO;
      T     #Inst_DB;
      NOP   0;

NETWORK
TITLE = Reset signal from M Code
      LAR1  P#0.0;
      L     900;
R001: T     #TEMP0;
      OPN   DB [#Inst_DB];
      A     "M_ONE";
      R     DBX [AR1, P#4.0];
      +AR1  P#0.1;
      L     #TEMP0;
      LOOP  R001;

NETWORK
TITLE = Set signal from "M function 1 (DInt)"
      OPN   DB [#DB_Channel];
      A     %DBX58.0;  // M function 1 change
      JCN   END1;

      LAR1  P#0.0;
      L     100;
      T     #INDEX;
      L     900;
S001: T     #TEMP0;

      L     %DBW72;
      L     #INDEX;
      ==I;
      JC    Mse1;
      L     #INDEX;
      +     1;
      T     #INDEX;
      +AR1  P#0.1;
      L     #TEMP0;
      LOOP  S001;
      JU    END1;
Mse1: OPN   DB [#Inst_DB];
      S     DBX [AR1, P#4.0];

END1: NOP   0;

NETWORK
TITLE = Set signal from "M function 2 (DInt)"
      OPN   DB [#DB_Channel];
      A     %DBX58.1;  // M function 2 change
      JCN   END2;

      LAR1  P#0.0;
      L     100;
      T     #INDEX;
      L     900;
S002: T     #TEMP0;

      L     %DBW78;
      L     #INDEX;
      ==I;
      JC    Mse2;
      L     #INDEX;
      +     1;
      T     #INDEX;
      +AR1  P#0.1;
      L     #TEMP0;
      LOOP  S002;
      JU    END2;
Mse2: OPN   DB [#Inst_DB];
      S     DBX [AR1, P#4.0];

END2: NOP   0;

NETWORK
TITLE = Set signal from "M function 3 (DInt)"
      OPN   DB [#DB_Channel];
      A     %DBX58.2;  // M function 3 change
      JCN   END3;

      LAR1  P#0.0;
      L     100;
      T     #INDEX;
      L     900;
S003: T     #TEMP0;

      L     %DBW84;
      L     #INDEX;
      ==I;
      JC    Mse3;
      L     #INDEX;
      +     1;
      T     #INDEX;
      +AR1  P#0.1;
      L     #TEMP0;
      LOOP  S003;
      JU    END3;
Mse3: OPN   DB [#Inst_DB];
      S     DBX [AR1, P#4.0];

END3: NOP   0;

NETWORK
TITLE = Set signal from "M function 4 (DInt)"
      OPN   DB [#DB_Channel];
      A     %DBX58.3;  // M function 4 change
      JCN   END4;

      LAR1  P#0.0;
      L     100;
      T     #INDEX;
      L     900;
S004: T     #TEMP0;

      L     %DBW90;
      L     #INDEX;
      ==I;
      JC    Mse4;
      L     #INDEX;
      +     1;
      T     #INDEX;
      +AR1  P#0.1;
      L     #TEMP0;
      LOOP  S004;
      JU    END4;
Mse4: OPN   DB [#Inst_DB];
      S     DBX [AR1, P#4.0];

END4: NOP   0;

NETWORK
TITLE = Set signal from "M function 5 (DInt)"
      OPN   DB [#DB_Channel];
      A     %DBX58.4;  // M function 5 change
      JCN   END5;

      LAR1  P#0.0;
      L     100;
      T     #INDEX;
      L     900;
S005: T     #TEMP0;

      L     %DBW96;
      L     #INDEX;
      ==I;
      JC    Mse5;
      L     #INDEX;
      +     1;
      T     #INDEX;
      +AR1  P#0.1;
      L     #TEMP0;
      LOOP  S005;
      JU    END5;
Mse5: OPN   DB [#Inst_DB];
      S     DBX [AR1, P#4.0];

END5: NOP   0;

NETWORK
TITLE = 
      BE;

END_FUNCTION_BLOCK

FUNCTION_BLOCK "FB2001_AUTO_SINGLE_SEMI_MANUAL"   // FB2001, LAD
{ S7_Optimized_Access := 'TRUE' }
VERSION : 0.1
// stored: AutoNumber false, IsIECCheckEnabled false, IsRetainMemResEnabled false, MemoryReserve 100, SetENOAutomatically false, UDAEnableTagReadback false
   VAR_INPUT
      OPTIONS_0 { ExternalAccessible := 'False'; ExternalVisible := 'False'; ExternalWritable := 'False'} : Byte := 2#0000_0000;   // OPTIONS BYTE 0
      MODE_GROUP_NUMBER : Int;
   END_VAR
   VAR_IN_OUT
      MODE_GROUP_1_DB : Struct
         GENERAL : "AUTO_SINGLE_SEMI_MANUAL";
         STEP_BY_STEP : "MODES";
         MDA : "MODES";
         REFERENCE : "MODES";
         INCREMENTAL : "INCREMENTAL";
         BA : "BA_MODE";
      END_STRUCT;
      EXTRA_MODE_GROUP_DB : Struct
         GENERAL : "AUTO_SINGLE_SEMI_MANUAL";
         STEP_BY_STEP : "MODES";
         MDA : "MODES";
         REFERENCE : "MODES";
         INCREMENTAL : "INCREMENTAL";
         BA : "BA_MODE";
      END_STRUCT;
   END_VAR
   VAR_TEMP
      INPUTS_MASK : Byte;   // INPUT MASK
      O_BYTE_0 : Struct   // OPTIONS BYTE 0
         CHANGE_MODE_SEOC_ALARM : Bool;   // CHANGE MODE SEOC ALARM OPTION
         MODE_SELECTED_MEMORY : Bool;   // MODE SELECTED MEMORY OPTION
         SPARE : Bool;
         SPARE_1 : Bool;
         SPARE_2 : Bool;
         SPARE_3 : Bool;
         SPARE_4 : Bool;
         SPARE_5 : Bool;
      END_STRUCT;
      DB_NUMBER : DInt;   // DB NUMBER FOR ALARM DECODING
      MODE_GROUP_DB : Struct
         GENERAL : "AUTO_SINGLE_SEMI_MANUAL";
         STEP_BY_STEP : "MODES";
         MDA : "MODES";
         REFERENCE : "MODES";
         INCREMENTAL : "INCREMENTAL";
         BA : "BA_MODE";
      END_STRUCT;
   END_VAR
   // // MODE_GROUP_1_DB.STEP_BY_STEP.MODE_SELECTED : STEP BY STEP MODE SELECTED
   // // MODE_GROUP_1_DB.MDA.MODE_SELECTED : MDA MODE SELECTED
   // // MODE_GROUP_1_DB.REFERENCE.MODE_SELECTED : REFERENCE MODE SELECTED
   // // EXTRA_MODE_GROUP_DB.STEP_BY_STEP.MODE_SELECTED : STEP BY STEP MODE SELECTED
   // // EXTRA_MODE_GROUP_DB.MDA.MODE_SELECTED : MDA MODE SELECTED
   // // EXTRA_MODE_GROUP_DB.REFERENCE.MODE_SELECTED : REFERENCE MODE SELECTED
   // // MODE_GROUP_DB.STEP_BY_STEP.MODE_SELECTED : STEP BY STEP MODE SELECTED
   // // MODE_GROUP_DB.MDA.MODE_SELECTED : MDA MODE SELECTED
   // // MODE_GROUP_DB.REFERENCE.MODE_SELECTED : REFERENCE MODE SELECTED
   VAR_TEMP   // added for the SCL form of the ladder/FBD networks
      _w1 : Bool;
      _w2 : Bool;
   END_VAR
BEGIN

NETWORK
TITLE = READ INSTANCE DB
      L     DINO;
      +     10#800000;
      T     #DB_NUMBER;


REGION Network 2: OPTIONS
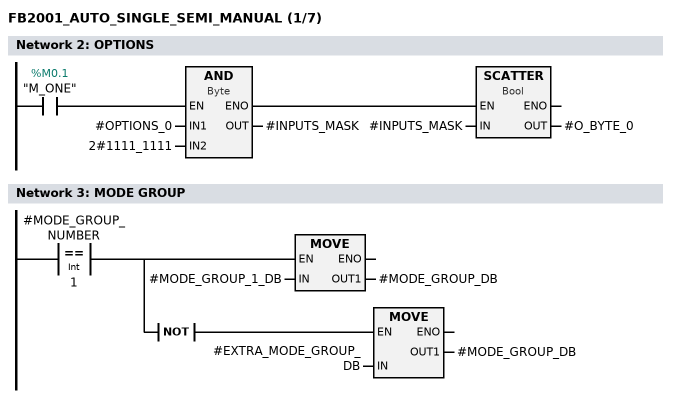
   RUNG wire#powerrail
      Contact( "M_ONE" )
      { S7_Templates := "SrcType := Byte"; S7_GenerateENO := "TRUE" } And(in1 := #OPTIONS_0, in2 := 2#1111_1111, out => #INPUTS_MASK)
      { S7_Templates := "[dest_type := Bool, src_type := Byte]" } SCATTER(IN := #INPUTS_MASK, OUT => #O_BYTE_0)
   END_RUNG
   // the same network as SCL:
   IF "M_ONE" THEN
       #INPUTS_MASK := #OPTIONS_0 AND 2#1111_1111;
       SCATTER(IN := #INPUTS_MASK, OUT => #O_BYTE_0);
   END_IF;
END_REGION

REGION Network 3: MODE GROUP
   RUNG wire#powerrail
      { S7_Templates := "SrcType := Int" } EQ_Contact(in1 := #MODE_GROUP_NUMBER, in2 := 1)
      wire#w1
      Move(in := #MODE_GROUP_1_DB, out1 => #MODE_GROUP_DB)
   END_RUNG
   RUNG wire#w1
      Not()
      Move(in := #EXTRA_MODE_GROUP_DB, out1 => #MODE_GROUP_DB)
   END_RUNG
   // the same network as SCL:
   #_w1 := #MODE_GROUP_NUMBER = 1;
   IF #_w1 THEN #MODE_GROUP_DB := #MODE_GROUP_1_DB; END_IF;
   IF NOT #_w1 THEN #MODE_GROUP_DB := #EXTRA_MODE_GROUP_DB; END_IF;
END_REGION

REGION Network 4: INPUTS
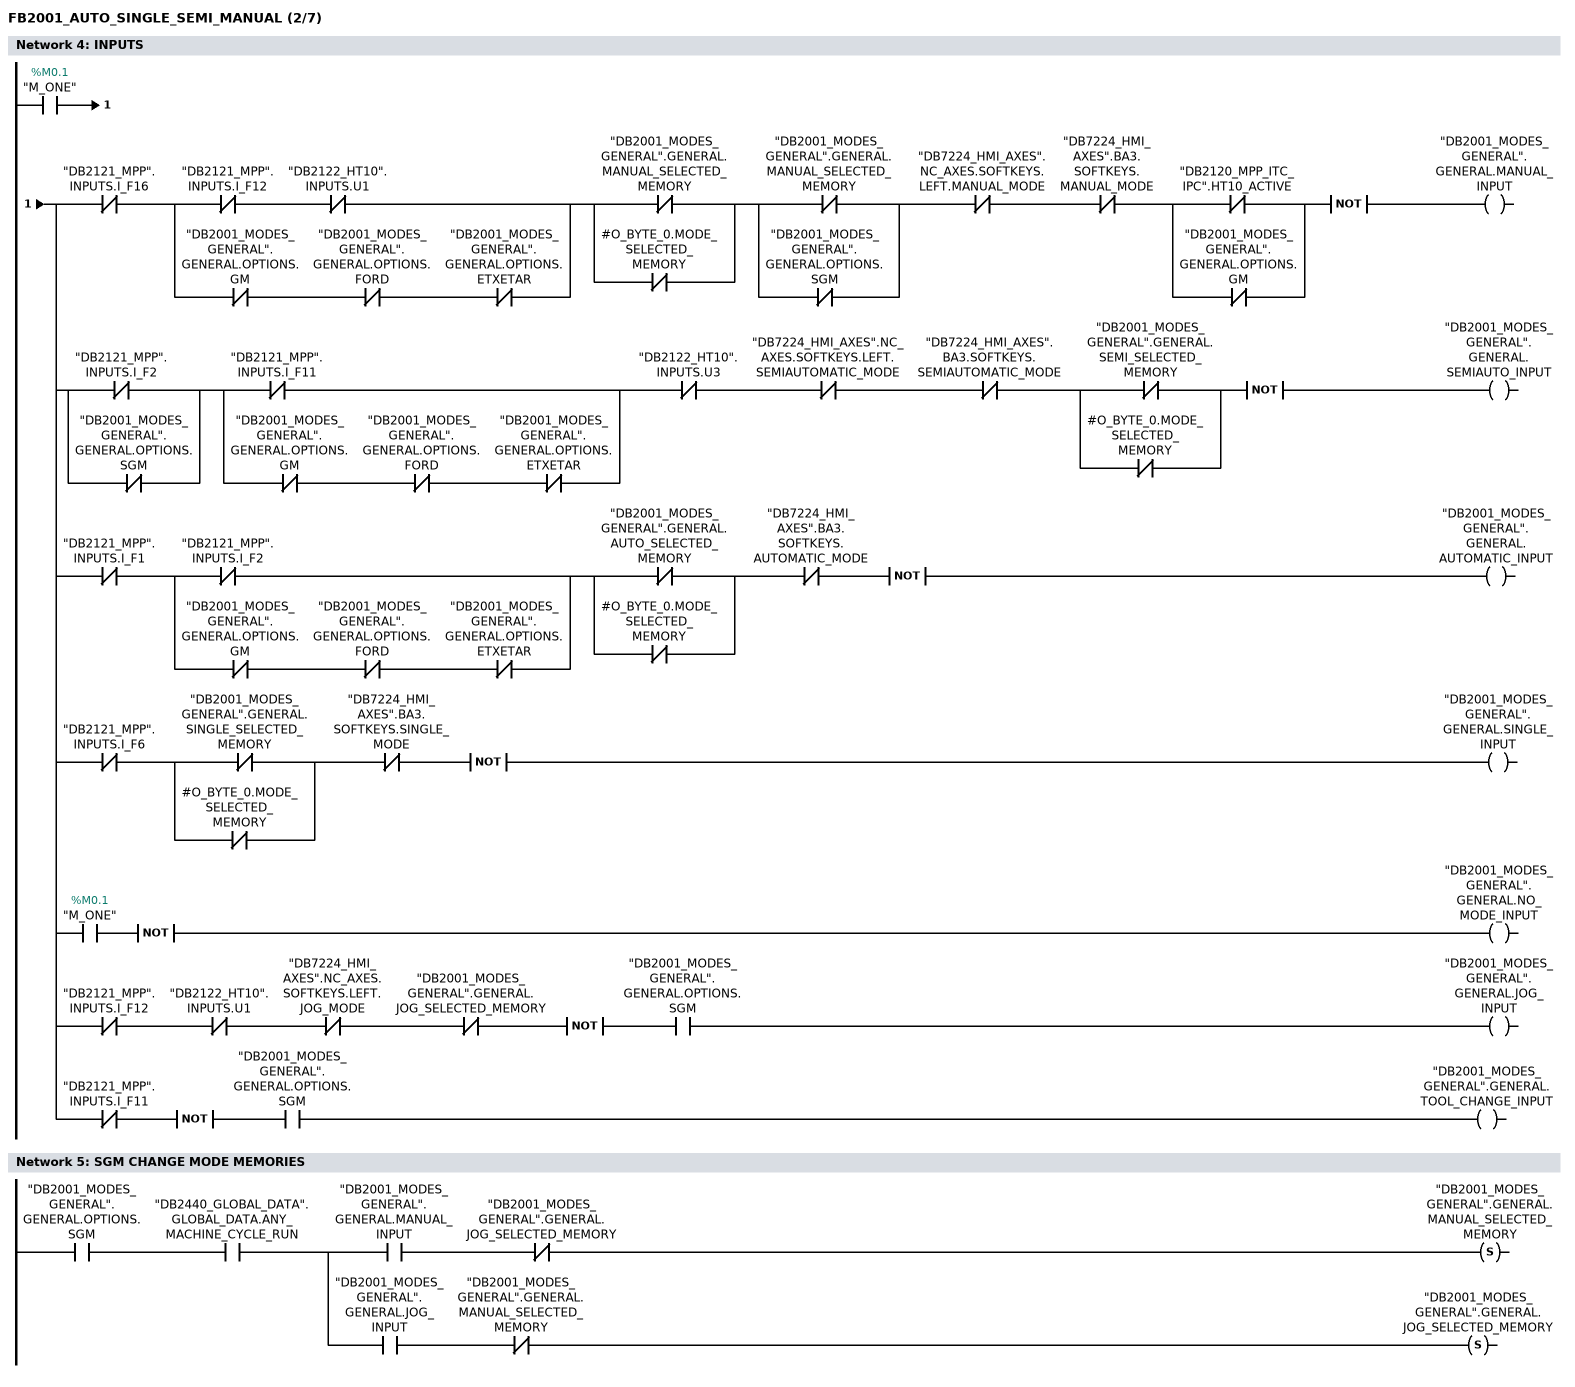
   RUNG wire#powerrail
      Contact( "M_ONE" )
      wire#w1
      I_Contact( "DB2121_MPP".INPUTS.I_F16 )
      wire#w2
      I_Contact( "DB2121_MPP".INPUTS.I_F12 )
      I_Contact( "DB2122_HT10".INPUTS.U1 )
      wire#w3
      I_Contact( "DB2001_MODES_GENERAL".GENERAL.MANUAL_SELECTED_MEMORY )
      wire#w4
      I_Contact( "DB2001_MODES_GENERAL".GENERAL.MANUAL_SELECTED_MEMORY )
      wire#w5
      I_Contact( "DB7224_HMI_AXES".NC_AXES.SOFTKEYS.LEFT.MANUAL_MODE )
      I_Contact( "DB7224_HMI_AXES".BA3.SOFTKEYS.MANUAL_MODE )
      wire#w6
      I_Contact( "DB2120_MPP_ITC_IPC".HT10_ACTIVE )
      wire#w7
      Not()
      Coil( "DB2001_MODES_GENERAL".GENERAL.MANUAL_INPUT )
   END_RUNG
   RUNG wire#w2
      I_Contact( "DB2001_MODES_GENERAL".GENERAL.OPTIONS.GM )
      I_Contact( "DB2001_MODES_GENERAL".GENERAL.OPTIONS.FORD )
      I_Contact( "DB2001_MODES_GENERAL".GENERAL.OPTIONS.ETXETAR )
   END_RUNG wire#w3
   RUNG wire#w3
      I_Contact( #O_BYTE_0.MODE_SELECTED_MEMORY )
   END_RUNG wire#w4
   RUNG wire#w4
      I_Contact( "DB2001_MODES_GENERAL".GENERAL.OPTIONS.SGM )
   END_RUNG wire#w5
   RUNG wire#w6
      I_Contact( "DB2001_MODES_GENERAL".GENERAL.OPTIONS.GM )
   END_RUNG wire#w7
   RUNG wire#w1
      I_Contact( "DB2121_MPP".INPUTS.I_F2 )
      wire#w8
      I_Contact( "DB2121_MPP".INPUTS.I_F11 )
      wire#w9
      I_Contact( "DB2122_HT10".INPUTS.U3 )
      I_Contact( "DB7224_HMI_AXES".NC_AXES.SOFTKEYS.LEFT.SEMIAUTOMATIC_MODE )
      I_Contact( "DB7224_HMI_AXES".BA3.SOFTKEYS.SEMIAUTOMATIC_MODE )
      wire#w10
      I_Contact( "DB2001_MODES_GENERAL".GENERAL.SEMI_SELECTED_MEMORY )
      wire#w11
      Not()
      Coil( "DB2001_MODES_GENERAL".GENERAL.SEMIAUTO_INPUT )
   END_RUNG
   RUNG wire#w1
      I_Contact( "DB2001_MODES_GENERAL".GENERAL.OPTIONS.SGM )
   END_RUNG wire#w8
   RUNG wire#w8
      I_Contact( "DB2001_MODES_GENERAL".GENERAL.OPTIONS.GM )
      I_Contact( "DB2001_MODES_GENERAL".GENERAL.OPTIONS.FORD )
      I_Contact( "DB2001_MODES_GENERAL".GENERAL.OPTIONS.ETXETAR )
   END_RUNG wire#w9
   RUNG wire#w10
      I_Contact( #O_BYTE_0.MODE_SELECTED_MEMORY )
   END_RUNG wire#w11
   RUNG wire#w1
      I_Contact( "DB2121_MPP".INPUTS.I_F1 )
      wire#w12
      I_Contact( "DB2121_MPP".INPUTS.I_F2 )
      wire#w13
      I_Contact( "DB2001_MODES_GENERAL".GENERAL.AUTO_SELECTED_MEMORY )
      wire#w14
      I_Contact( "DB7224_HMI_AXES".BA3.SOFTKEYS.AUTOMATIC_MODE )
      Not()
      Coil( "DB2001_MODES_GENERAL".GENERAL.AUTOMATIC_INPUT )
   END_RUNG
   RUNG wire#w12
      I_Contact( "DB2001_MODES_GENERAL".GENERAL.OPTIONS.GM )
      I_Contact( "DB2001_MODES_GENERAL".GENERAL.OPTIONS.FORD )
      I_Contact( "DB2001_MODES_GENERAL".GENERAL.OPTIONS.ETXETAR )
   END_RUNG wire#w13
   RUNG wire#w13
      I_Contact( #O_BYTE_0.MODE_SELECTED_MEMORY )
   END_RUNG wire#w14
   RUNG wire#w1
      I_Contact( "DB2121_MPP".INPUTS.I_F6 )
      wire#w15
      I_Contact( "DB2001_MODES_GENERAL".GENERAL.SINGLE_SELECTED_MEMORY )
      wire#w16
      I_Contact( "DB7224_HMI_AXES".BA3.SOFTKEYS.SINGLE_MODE )
      Not()
      Coil( "DB2001_MODES_GENERAL".GENERAL.SINGLE_INPUT )
   END_RUNG
   RUNG wire#w15
      I_Contact( #O_BYTE_0.MODE_SELECTED_MEMORY )
   END_RUNG wire#w16
   RUNG wire#w1
      Contact( "M_ONE" )
      Not()
      Coil( "DB2001_MODES_GENERAL".GENERAL.NO_MODE_INPUT )
   END_RUNG
   RUNG wire#w1
      I_Contact( "DB2121_MPP".INPUTS.I_F12 )
      I_Contact( "DB2122_HT10".INPUTS.U1 )
      I_Contact( "DB7224_HMI_AXES".NC_AXES.SOFTKEYS.LEFT.JOG_MODE )
      I_Contact( "DB2001_MODES_GENERAL".GENERAL.JOG_SELECTED_MEMORY )
      Not()
      Contact( "DB2001_MODES_GENERAL".GENERAL.OPTIONS.SGM )
      Coil( "DB2001_MODES_GENERAL".GENERAL.JOG_INPUT )
   END_RUNG
   RUNG wire#w1
      I_Contact( "DB2121_MPP".INPUTS.I_F11 )
      Not()
      Contact( "DB2001_MODES_GENERAL".GENERAL.OPTIONS.SGM )
      Coil( "DB2001_MODES_GENERAL".GENERAL.TOOL_CHANGE_INPUT )
   END_RUNG
   // the same network as SCL:
   "DB2001_MODES_GENERAL".GENERAL.MANUAL_INPUT := NOT ("M_ONE" AND NOT "DB2121_MPP".INPUTS.I_F16 AND ((NOT "DB2121_MPP".INPUTS.I_F12 AND NOT "DB2122_HT10".INPUTS.U1) OR (NOT "DB2001_MODES_GENERAL".GENERAL.OPTIONS.GM AND NOT "DB2001_MODES_GENERAL".GENERAL.OPTIONS.FORD AND NOT "DB2001_MODES_GENERAL".GENERAL.OPTIONS.ETXETAR)) AND (NOT "DB2001_MODES_GENERAL".GENERAL.MANUAL_SELECTED_MEMORY OR NOT #O_BYTE_0.MODE_SELECTED_MEMORY) AND (NOT "DB2001_MODES_GENERAL".GENERAL.MANUAL_SELECTED_MEMORY OR NOT "DB2001_MODES_GENERAL".GENERAL.OPTIONS.SGM) AND NOT "DB7224_HMI_AXES".NC_AXES.SOFTKEYS.LEFT.MANUAL_MODE AND NOT "DB7224_HMI_AXES".BA3.SOFTKEYS.MANUAL_MODE AND (NOT "DB2120_MPP_ITC_IPC".HT10_ACTIVE OR NOT "DB2001_MODES_GENERAL".GENERAL.OPTIONS.GM));
   "DB2001_MODES_GENERAL".GENERAL.SEMIAUTO_INPUT := NOT ("M_ONE" AND (NOT "DB2121_MPP".INPUTS.I_F2 OR NOT "DB2001_MODES_GENERAL".GENERAL.OPTIONS.SGM) AND (NOT "DB2121_MPP".INPUTS.I_F11 OR (NOT "DB2001_MODES_GENERAL".GENERAL.OPTIONS.GM AND NOT "DB2001_MODES_GENERAL".GENERAL.OPTIONS.FORD AND NOT "DB2001_MODES_GENERAL".GENERAL.OPTIONS.ETXETAR)) AND NOT "DB2122_HT10".INPUTS.U3 AND NOT "DB7224_HMI_AXES".NC_AXES.SOFTKEYS.LEFT.SEMIAUTOMATIC_MODE AND NOT "DB7224_HMI_AXES".BA3.SOFTKEYS.SEMIAUTOMATIC_MODE AND (NOT "DB2001_MODES_GENERAL".GENERAL.SEMI_SELECTED_MEMORY OR NOT #O_BYTE_0.MODE_SELECTED_MEMORY));
   "DB2001_MODES_GENERAL".GENERAL.AUTOMATIC_INPUT := NOT ("M_ONE" AND NOT "DB2121_MPP".INPUTS.I_F1 AND (NOT "DB2121_MPP".INPUTS.I_F2 OR (NOT "DB2001_MODES_GENERAL".GENERAL.OPTIONS.GM AND NOT "DB2001_MODES_GENERAL".GENERAL.OPTIONS.FORD AND NOT "DB2001_MODES_GENERAL".GENERAL.OPTIONS.ETXETAR)) AND (NOT "DB2001_MODES_GENERAL".GENERAL.AUTO_SELECTED_MEMORY OR NOT #O_BYTE_0.MODE_SELECTED_MEMORY) AND NOT "DB7224_HMI_AXES".BA3.SOFTKEYS.AUTOMATIC_MODE);
   "DB2001_MODES_GENERAL".GENERAL.SINGLE_INPUT := NOT ("M_ONE" AND NOT "DB2121_MPP".INPUTS.I_F6 AND (NOT "DB2001_MODES_GENERAL".GENERAL.SINGLE_SELECTED_MEMORY OR NOT #O_BYTE_0.MODE_SELECTED_MEMORY) AND NOT "DB7224_HMI_AXES".BA3.SOFTKEYS.SINGLE_MODE);
   "DB2001_MODES_GENERAL".GENERAL.NO_MODE_INPUT := NOT ("M_ONE" AND "M_ONE");
   "DB2001_MODES_GENERAL".GENERAL.JOG_INPUT := NOT ("M_ONE" AND NOT "DB2121_MPP".INPUTS.I_F12 AND NOT "DB2122_HT10".INPUTS.U1 AND NOT "DB7224_HMI_AXES".NC_AXES.SOFTKEYS.LEFT.JOG_MODE AND NOT "DB2001_MODES_GENERAL".GENERAL.JOG_SELECTED_MEMORY) AND "DB2001_MODES_GENERAL".GENERAL.OPTIONS.SGM;
   "DB2001_MODES_GENERAL".GENERAL.TOOL_CHANGE_INPUT := NOT ("M_ONE" AND NOT "DB2121_MPP".INPUTS.I_F11) AND "DB2001_MODES_GENERAL".GENERAL.OPTIONS.SGM;
END_REGION

REGION Network 5: SGM CHANGE MODE MEMORIES
   RUNG wire#powerrail
      Contact( "DB2001_MODES_GENERAL".GENERAL.OPTIONS.SGM )
      Contact( "DB2440_GLOBAL_DATA".GLOBAL_DATA.ANY_MACHINE_CYCLE_RUN )
      wire#w1
      Contact( "DB2001_MODES_GENERAL".GENERAL.MANUAL_INPUT )
      I_Contact( "DB2001_MODES_GENERAL".GENERAL.JOG_SELECTED_MEMORY )
      S_Coil( "DB2001_MODES_GENERAL".GENERAL.MANUAL_SELECTED_MEMORY )
   END_RUNG
   RUNG wire#w1
      Contact( "DB2001_MODES_GENERAL".GENERAL.JOG_INPUT )
      I_Contact( "DB2001_MODES_GENERAL".GENERAL.MANUAL_SELECTED_MEMORY )
      S_Coil( "DB2001_MODES_GENERAL".GENERAL.JOG_SELECTED_MEMORY )
   END_RUNG
   // the same network as SCL:
   #_w1 := "DB2001_MODES_GENERAL".GENERAL.OPTIONS.SGM AND "DB2440_GLOBAL_DATA".GLOBAL_DATA.ANY_MACHINE_CYCLE_RUN;
   IF #_w1 AND "DB2001_MODES_GENERAL".GENERAL.MANUAL_INPUT AND NOT "DB2001_MODES_GENERAL".GENERAL.JOG_SELECTED_MEMORY THEN
       "DB2001_MODES_GENERAL".GENERAL.MANUAL_SELECTED_MEMORY := TRUE;
   END_IF;
   IF #_w1 AND "DB2001_MODES_GENERAL".GENERAL.JOG_INPUT AND NOT "DB2001_MODES_GENERAL".GENERAL.MANUAL_SELECTED_MEMORY THEN
       "DB2001_MODES_GENERAL".GENERAL.JOG_SELECTED_MEMORY := TRUE;
   END_IF;
END_REGION

REGION Network 6: CHANGE MODE GENERAL CONDITIONS
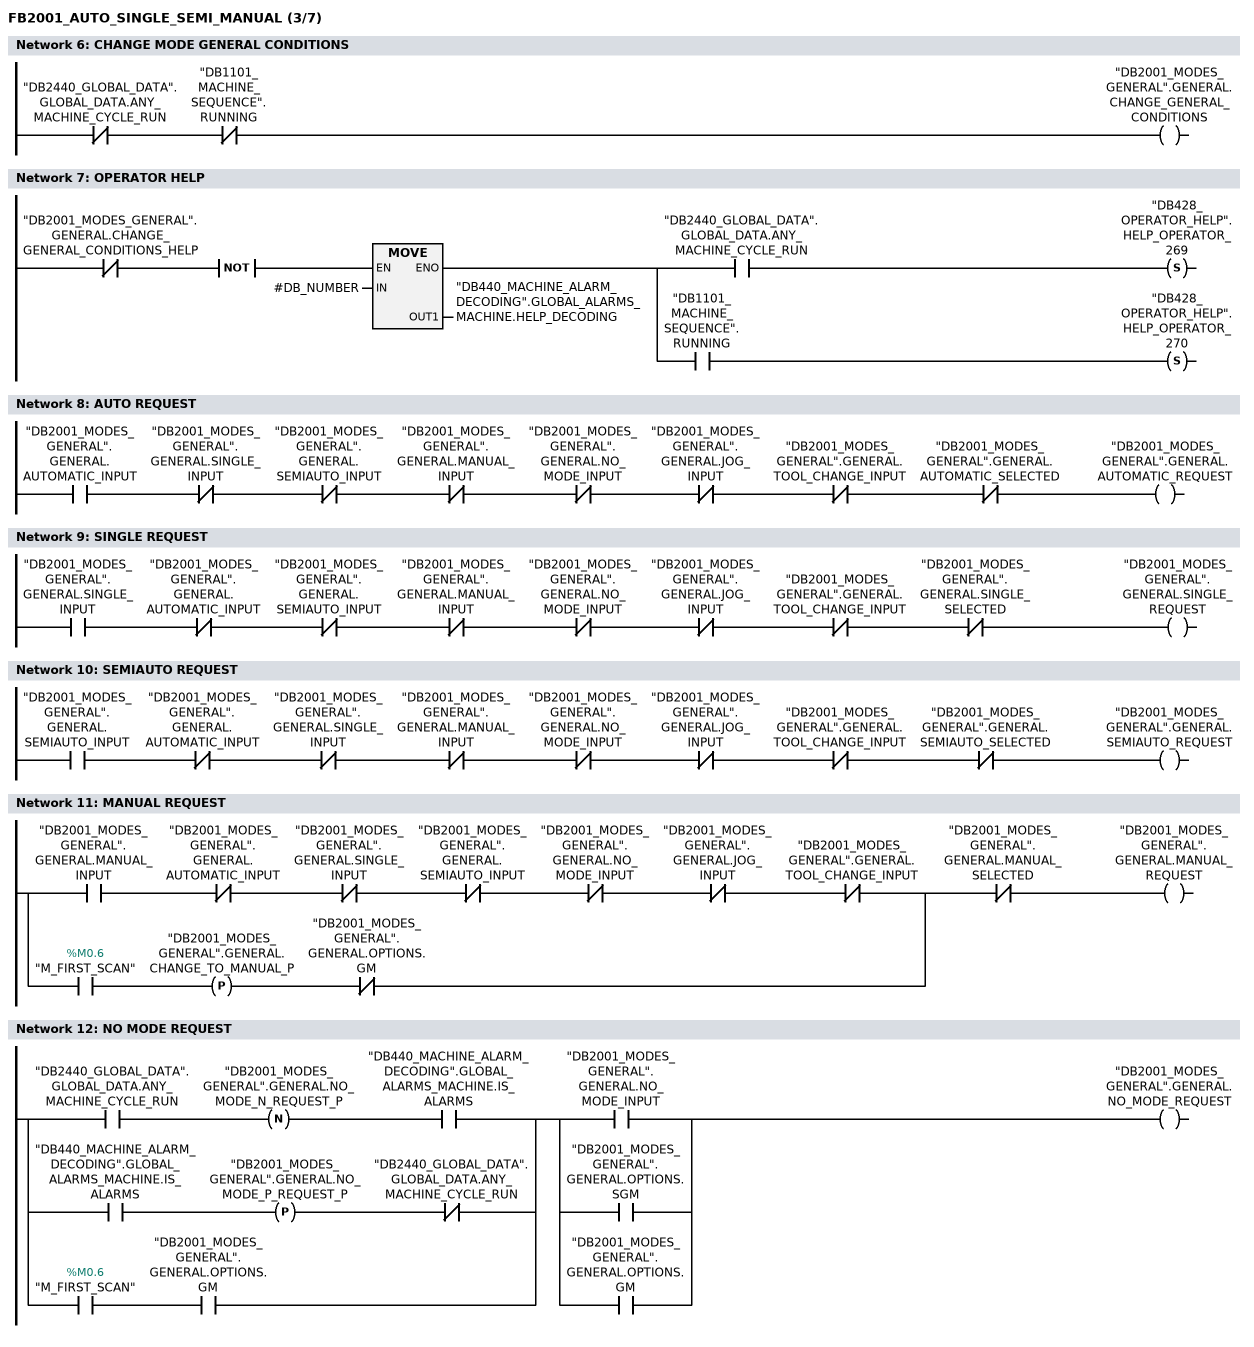
   RUNG wire#powerrail
      I_Contact( "DB2440_GLOBAL_DATA".GLOBAL_DATA.ANY_MACHINE_CYCLE_RUN )
      I_Contact( "DB1101_MACHINE_SEQUENCE".RUNNING )
      Coil( "DB2001_MODES_GENERAL".GENERAL.CHANGE_GENERAL_CONDITIONS )
   END_RUNG
   // the same network as SCL:
   "DB2001_MODES_GENERAL".GENERAL.CHANGE_GENERAL_CONDITIONS := NOT "DB2440_GLOBAL_DATA".GLOBAL_DATA.ANY_MACHINE_CYCLE_RUN AND NOT "DB1101_MACHINE_SEQUENCE".RUNNING;
END_REGION

REGION Network 7: OPERATOR HELP
   RUNG wire#powerrail
      I_Contact( "DB2001_MODES_GENERAL".GENERAL.CHANGE_GENERAL_CONDITIONS_HELP )
      Not()
      { S7_GenerateENO := "TRUE" } Move(in := #DB_NUMBER, out1 => "DB440_MACHINE_ALARM_DECODING".GLOBAL_ALARMS_MACHINE.HELP_DECODING)
      wire#w1
      Contact( "DB2440_GLOBAL_DATA".GLOBAL_DATA.ANY_MACHINE_CYCLE_RUN )
      S_Coil( "DB428_OPERATOR_HELP".HELP_OPERATOR_269 )
   END_RUNG
   RUNG wire#w1
      Contact( "DB1101_MACHINE_SEQUENCE".RUNNING )
      S_Coil( "DB428_OPERATOR_HELP".HELP_OPERATOR_270 )
   END_RUNG
   // the same network as SCL:
   // ENO of a box is taken as its EN; it also drops when the box reports an error
   #_w1 := NOT (NOT "DB2001_MODES_GENERAL".GENERAL.CHANGE_GENERAL_CONDITIONS_HELP);
   IF #_w1 THEN "DB440_MACHINE_ALARM_DECODING".GLOBAL_ALARMS_MACHINE.HELP_DECODING := #DB_NUMBER; END_IF;
   IF #_w1 AND "DB2440_GLOBAL_DATA".GLOBAL_DATA.ANY_MACHINE_CYCLE_RUN THEN
       "DB428_OPERATOR_HELP".HELP_OPERATOR_269 := TRUE;
   END_IF;
   IF #_w1 AND "DB1101_MACHINE_SEQUENCE".RUNNING THEN
       "DB428_OPERATOR_HELP".HELP_OPERATOR_270 := TRUE;
   END_IF;
END_REGION

REGION Network 8: AUTO REQUEST
   RUNG wire#powerrail
      Contact( "DB2001_MODES_GENERAL".GENERAL.AUTOMATIC_INPUT )
      I_Contact( "DB2001_MODES_GENERAL".GENERAL.SINGLE_INPUT )
      I_Contact( "DB2001_MODES_GENERAL".GENERAL.SEMIAUTO_INPUT )
      I_Contact( "DB2001_MODES_GENERAL".GENERAL.MANUAL_INPUT )
      I_Contact( "DB2001_MODES_GENERAL".GENERAL.NO_MODE_INPUT )
      I_Contact( "DB2001_MODES_GENERAL".GENERAL.JOG_INPUT )
      I_Contact( "DB2001_MODES_GENERAL".GENERAL.TOOL_CHANGE_INPUT )
      I_Contact( "DB2001_MODES_GENERAL".GENERAL.AUTOMATIC_SELECTED )
      Coil( "DB2001_MODES_GENERAL".GENERAL.AUTOMATIC_REQUEST )
   END_RUNG
   // the same network as SCL:
   "DB2001_MODES_GENERAL".GENERAL.AUTOMATIC_REQUEST := "DB2001_MODES_GENERAL".GENERAL.AUTOMATIC_INPUT AND NOT "DB2001_MODES_GENERAL".GENERAL.SINGLE_INPUT AND NOT "DB2001_MODES_GENERAL".GENERAL.SEMIAUTO_INPUT AND NOT "DB2001_MODES_GENERAL".GENERAL.MANUAL_INPUT AND NOT "DB2001_MODES_GENERAL".GENERAL.NO_MODE_INPUT AND NOT "DB2001_MODES_GENERAL".GENERAL.JOG_INPUT AND NOT "DB2001_MODES_GENERAL".GENERAL.TOOL_CHANGE_INPUT AND NOT "DB2001_MODES_GENERAL".GENERAL.AUTOMATIC_SELECTED;
END_REGION

REGION Network 9: SINGLE REQUEST
   RUNG wire#powerrail
      Contact( "DB2001_MODES_GENERAL".GENERAL.SINGLE_INPUT )
      I_Contact( "DB2001_MODES_GENERAL".GENERAL.AUTOMATIC_INPUT )
      I_Contact( "DB2001_MODES_GENERAL".GENERAL.SEMIAUTO_INPUT )
      I_Contact( "DB2001_MODES_GENERAL".GENERAL.MANUAL_INPUT )
      I_Contact( "DB2001_MODES_GENERAL".GENERAL.NO_MODE_INPUT )
      I_Contact( "DB2001_MODES_GENERAL".GENERAL.JOG_INPUT )
      I_Contact( "DB2001_MODES_GENERAL".GENERAL.TOOL_CHANGE_INPUT )
      I_Contact( "DB2001_MODES_GENERAL".GENERAL.SINGLE_SELECTED )
      Coil( "DB2001_MODES_GENERAL".GENERAL.SINGLE_REQUEST )
   END_RUNG
   // the same network as SCL:
   "DB2001_MODES_GENERAL".GENERAL.SINGLE_REQUEST := "DB2001_MODES_GENERAL".GENERAL.SINGLE_INPUT AND NOT "DB2001_MODES_GENERAL".GENERAL.AUTOMATIC_INPUT AND NOT "DB2001_MODES_GENERAL".GENERAL.SEMIAUTO_INPUT AND NOT "DB2001_MODES_GENERAL".GENERAL.MANUAL_INPUT AND NOT "DB2001_MODES_GENERAL".GENERAL.NO_MODE_INPUT AND NOT "DB2001_MODES_GENERAL".GENERAL.JOG_INPUT AND NOT "DB2001_MODES_GENERAL".GENERAL.TOOL_CHANGE_INPUT AND NOT "DB2001_MODES_GENERAL".GENERAL.SINGLE_SELECTED;
END_REGION

REGION Network 10: SEMIAUTO REQUEST
   RUNG wire#powerrail
      Contact( "DB2001_MODES_GENERAL".GENERAL.SEMIAUTO_INPUT )
      I_Contact( "DB2001_MODES_GENERAL".GENERAL.AUTOMATIC_INPUT )
      I_Contact( "DB2001_MODES_GENERAL".GENERAL.SINGLE_INPUT )
      I_Contact( "DB2001_MODES_GENERAL".GENERAL.MANUAL_INPUT )
      I_Contact( "DB2001_MODES_GENERAL".GENERAL.NO_MODE_INPUT )
      I_Contact( "DB2001_MODES_GENERAL".GENERAL.JOG_INPUT )
      I_Contact( "DB2001_MODES_GENERAL".GENERAL.TOOL_CHANGE_INPUT )
      I_Contact( "DB2001_MODES_GENERAL".GENERAL.SEMIAUTO_SELECTED )
      Coil( "DB2001_MODES_GENERAL".GENERAL.SEMIAUTO_REQUEST )
   END_RUNG
   // the same network as SCL:
   "DB2001_MODES_GENERAL".GENERAL.SEMIAUTO_REQUEST := "DB2001_MODES_GENERAL".GENERAL.SEMIAUTO_INPUT AND NOT "DB2001_MODES_GENERAL".GENERAL.AUTOMATIC_INPUT AND NOT "DB2001_MODES_GENERAL".GENERAL.SINGLE_INPUT AND NOT "DB2001_MODES_GENERAL".GENERAL.MANUAL_INPUT AND NOT "DB2001_MODES_GENERAL".GENERAL.NO_MODE_INPUT AND NOT "DB2001_MODES_GENERAL".GENERAL.JOG_INPUT AND NOT "DB2001_MODES_GENERAL".GENERAL.TOOL_CHANGE_INPUT AND NOT "DB2001_MODES_GENERAL".GENERAL.SEMIAUTO_SELECTED;
END_REGION

REGION Network 11: MANUAL REQUEST
   RUNG wire#powerrail
      Contact( "DB2001_MODES_GENERAL".GENERAL.MANUAL_INPUT )
      I_Contact( "DB2001_MODES_GENERAL".GENERAL.AUTOMATIC_INPUT )
      I_Contact( "DB2001_MODES_GENERAL".GENERAL.SINGLE_INPUT )
      I_Contact( "DB2001_MODES_GENERAL".GENERAL.SEMIAUTO_INPUT )
      I_Contact( "DB2001_MODES_GENERAL".GENERAL.NO_MODE_INPUT )
      I_Contact( "DB2001_MODES_GENERAL".GENERAL.JOG_INPUT )
      I_Contact( "DB2001_MODES_GENERAL".GENERAL.TOOL_CHANGE_INPUT )
      wire#w1
      I_Contact( "DB2001_MODES_GENERAL".GENERAL.MANUAL_SELECTED )
      Coil( "DB2001_MODES_GENERAL".GENERAL.MANUAL_REQUEST )
   END_RUNG
   RUNG wire#powerrail
      Contact( "M_FIRST_SCAN" )
      P_Trig( "DB2001_MODES_GENERAL".GENERAL.CHANGE_TO_MANUAL_P )
      I_Contact( "DB2001_MODES_GENERAL".GENERAL.OPTIONS.GM )
   END_RUNG wire#w1
   // the same network as SCL:
   #_w1 := "M_FIRST_SCAN" AND NOT "DB2001_MODES_GENERAL".GENERAL.CHANGE_TO_MANUAL_P;   // rising edge
   "DB2001_MODES_GENERAL".GENERAL.CHANGE_TO_MANUAL_P := "M_FIRST_SCAN";
   "DB2001_MODES_GENERAL".GENERAL.MANUAL_REQUEST := (("DB2001_MODES_GENERAL".GENERAL.MANUAL_INPUT AND NOT "DB2001_MODES_GENERAL".GENERAL.AUTOMATIC_INPUT AND NOT "DB2001_MODES_GENERAL".GENERAL.SINGLE_INPUT AND NOT "DB2001_MODES_GENERAL".GENERAL.SEMIAUTO_INPUT AND NOT "DB2001_MODES_GENERAL".GENERAL.NO_MODE_INPUT AND NOT "DB2001_MODES_GENERAL".GENERAL.JOG_INPUT AND NOT "DB2001_MODES_GENERAL".GENERAL.TOOL_CHANGE_INPUT) OR (#_w1 AND NOT "DB2001_MODES_GENERAL".GENERAL.OPTIONS.GM)) AND NOT "DB2001_MODES_GENERAL".GENERAL.MANUAL_SELECTED;
END_REGION

REGION Network 12: NO MODE REQUEST
   RUNG wire#powerrail
      Contact( "DB2440_GLOBAL_DATA".GLOBAL_DATA.ANY_MACHINE_CYCLE_RUN )
      N_Trig( "DB2001_MODES_GENERAL".GENERAL.NO_MODE_N_REQUEST_P )
      Contact( "DB440_MACHINE_ALARM_DECODING".GLOBAL_ALARMS_MACHINE.IS_ALARMS )
      wire#w1
      Contact( "DB2001_MODES_GENERAL".GENERAL.NO_MODE_INPUT )
      wire#w2
      Coil( "DB2001_MODES_GENERAL".GENERAL.NO_MODE_REQUEST )
   END_RUNG
   RUNG wire#powerrail
      Contact( "DB440_MACHINE_ALARM_DECODING".GLOBAL_ALARMS_MACHINE.IS_ALARMS )
      P_Trig( "DB2001_MODES_GENERAL".GENERAL.NO_MODE_P_REQUEST_P )
      I_Contact( "DB2440_GLOBAL_DATA".GLOBAL_DATA.ANY_MACHINE_CYCLE_RUN )
   END_RUNG wire#w1
   RUNG wire#powerrail
      Contact( "M_FIRST_SCAN" )
      Contact( "DB2001_MODES_GENERAL".GENERAL.OPTIONS.GM )
   END_RUNG wire#w1
   RUNG wire#w1
      Contact( "DB2001_MODES_GENERAL".GENERAL.OPTIONS.SGM )
   END_RUNG wire#w2
   RUNG wire#w1
      Contact( "DB2001_MODES_GENERAL".GENERAL.OPTIONS.GM )
   END_RUNG wire#w2
   // the same network as SCL:
   #_w1 := NOT "DB2440_GLOBAL_DATA".GLOBAL_DATA.ANY_MACHINE_CYCLE_RUN AND "DB2001_MODES_GENERAL".GENERAL.NO_MODE_N_REQUEST_P;   // falling edge
   "DB2001_MODES_GENERAL".GENERAL.NO_MODE_N_REQUEST_P := "DB2440_GLOBAL_DATA".GLOBAL_DATA.ANY_MACHINE_CYCLE_RUN;
   #_w2 := "DB440_MACHINE_ALARM_DECODING".GLOBAL_ALARMS_MACHINE.IS_ALARMS AND NOT "DB2001_MODES_GENERAL".GENERAL.NO_MODE_P_REQUEST_P;   // rising edge
   "DB2001_MODES_GENERAL".GENERAL.NO_MODE_P_REQUEST_P := "DB440_MACHINE_ALARM_DECODING".GLOBAL_ALARMS_MACHINE.IS_ALARMS;
   "DB2001_MODES_GENERAL".GENERAL.NO_MODE_REQUEST := ((#_w1 AND "DB440_MACHINE_ALARM_DECODING".GLOBAL_ALARMS_MACHINE.IS_ALARMS) OR (#_w2 AND NOT "DB2440_GLOBAL_DATA".GLOBAL_DATA.ANY_MACHINE_CYCLE_RUN) OR ("M_FIRST_SCAN" AND "DB2001_MODES_GENERAL".GENERAL.OPTIONS.GM)) AND ("DB2001_MODES_GENERAL".GENERAL.NO_MODE_INPUT OR "DB2001_MODES_GENERAL".GENERAL.OPTIONS.SGM OR "DB2001_MODES_GENERAL".GENERAL.OPTIONS.GM);
END_REGION

REGION Network 13: JOG REQUEST
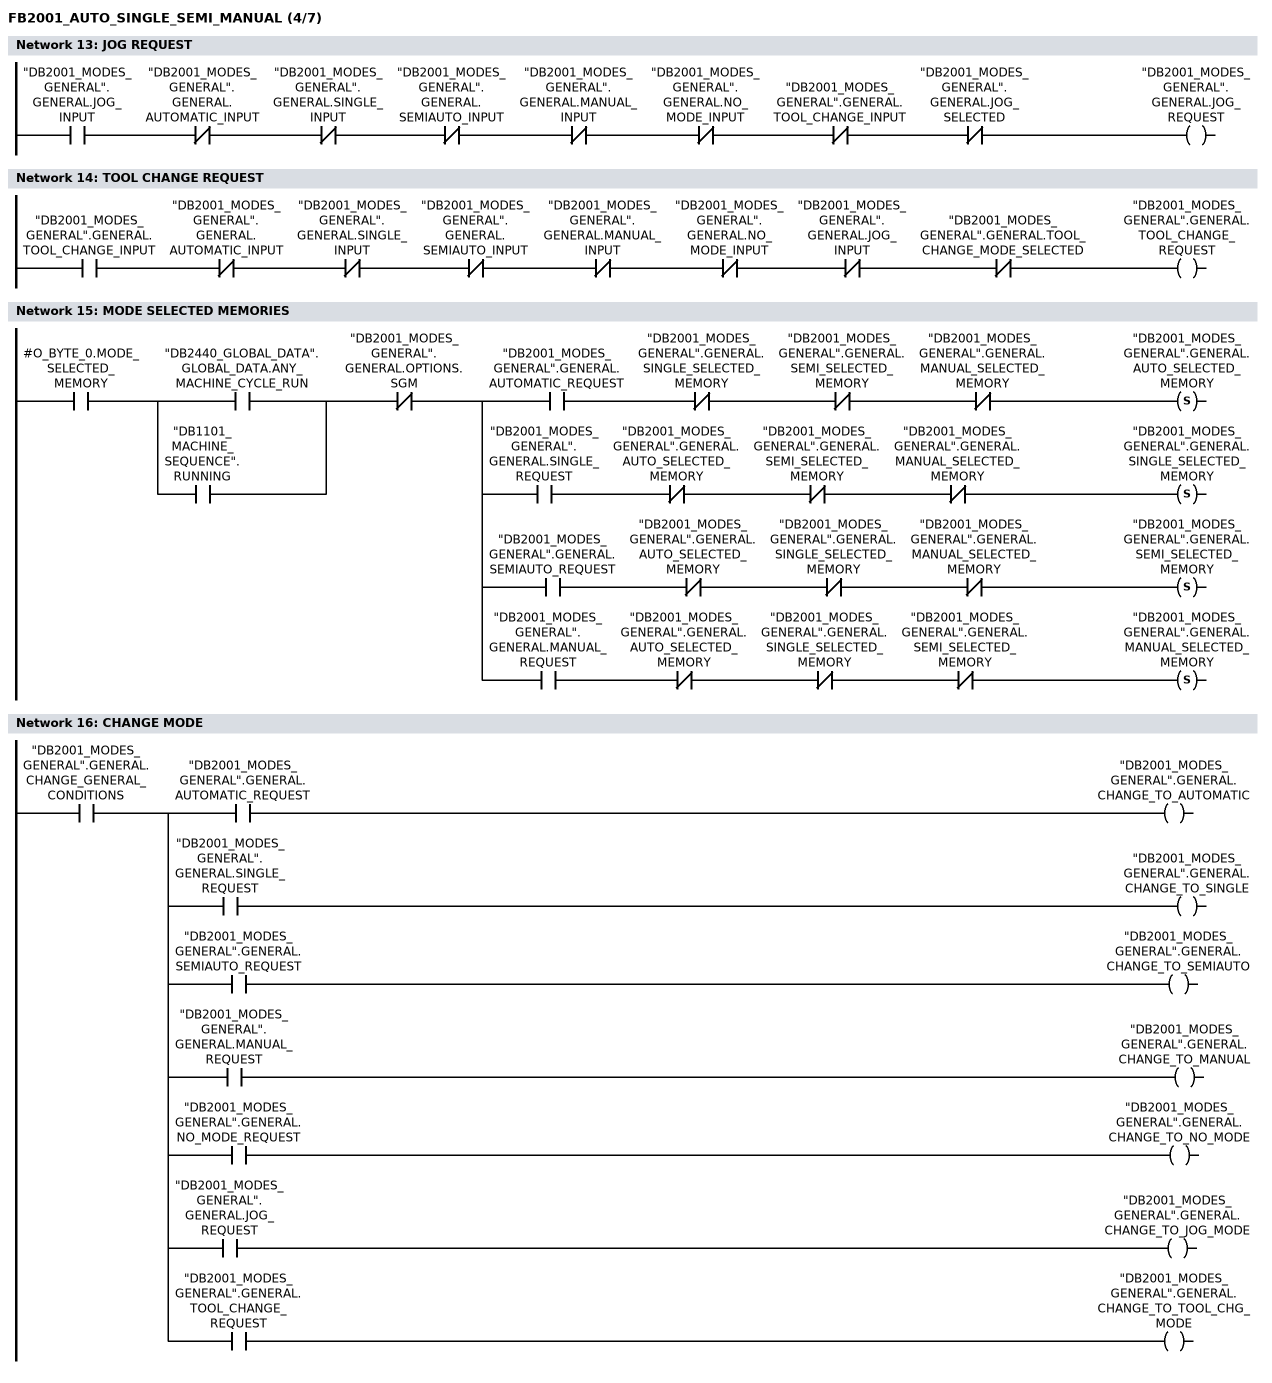
   RUNG wire#powerrail
      Contact( "DB2001_MODES_GENERAL".GENERAL.JOG_INPUT )
      I_Contact( "DB2001_MODES_GENERAL".GENERAL.AUTOMATIC_INPUT )
      I_Contact( "DB2001_MODES_GENERAL".GENERAL.SINGLE_INPUT )
      I_Contact( "DB2001_MODES_GENERAL".GENERAL.SEMIAUTO_INPUT )
      I_Contact( "DB2001_MODES_GENERAL".GENERAL.MANUAL_INPUT )
      I_Contact( "DB2001_MODES_GENERAL".GENERAL.NO_MODE_INPUT )
      I_Contact( "DB2001_MODES_GENERAL".GENERAL.TOOL_CHANGE_INPUT )
      I_Contact( "DB2001_MODES_GENERAL".GENERAL.JOG_SELECTED )
      Coil( "DB2001_MODES_GENERAL".GENERAL.JOG_REQUEST )
   END_RUNG
   // the same network as SCL:
   "DB2001_MODES_GENERAL".GENERAL.JOG_REQUEST := "DB2001_MODES_GENERAL".GENERAL.JOG_INPUT AND NOT "DB2001_MODES_GENERAL".GENERAL.AUTOMATIC_INPUT AND NOT "DB2001_MODES_GENERAL".GENERAL.SINGLE_INPUT AND NOT "DB2001_MODES_GENERAL".GENERAL.SEMIAUTO_INPUT AND NOT "DB2001_MODES_GENERAL".GENERAL.MANUAL_INPUT AND NOT "DB2001_MODES_GENERAL".GENERAL.NO_MODE_INPUT AND NOT "DB2001_MODES_GENERAL".GENERAL.TOOL_CHANGE_INPUT AND NOT "DB2001_MODES_GENERAL".GENERAL.JOG_SELECTED;
END_REGION

REGION Network 14: TOOL CHANGE REQUEST
   RUNG wire#powerrail
      Contact( "DB2001_MODES_GENERAL".GENERAL.TOOL_CHANGE_INPUT )
      I_Contact( "DB2001_MODES_GENERAL".GENERAL.AUTOMATIC_INPUT )
      I_Contact( "DB2001_MODES_GENERAL".GENERAL.SINGLE_INPUT )
      I_Contact( "DB2001_MODES_GENERAL".GENERAL.SEMIAUTO_INPUT )
      I_Contact( "DB2001_MODES_GENERAL".GENERAL.MANUAL_INPUT )
      I_Contact( "DB2001_MODES_GENERAL".GENERAL.NO_MODE_INPUT )
      I_Contact( "DB2001_MODES_GENERAL".GENERAL.JOG_INPUT )
      I_Contact( "DB2001_MODES_GENERAL".GENERAL.TOOL_CHANGE_MODE_SELECTED )
      Coil( "DB2001_MODES_GENERAL".GENERAL.TOOL_CHANGE_REQUEST )
   END_RUNG
   // the same network as SCL:
   "DB2001_MODES_GENERAL".GENERAL.TOOL_CHANGE_REQUEST := "DB2001_MODES_GENERAL".GENERAL.TOOL_CHANGE_INPUT AND NOT "DB2001_MODES_GENERAL".GENERAL.AUTOMATIC_INPUT AND NOT "DB2001_MODES_GENERAL".GENERAL.SINGLE_INPUT AND NOT "DB2001_MODES_GENERAL".GENERAL.SEMIAUTO_INPUT AND NOT "DB2001_MODES_GENERAL".GENERAL.MANUAL_INPUT AND NOT "DB2001_MODES_GENERAL".GENERAL.NO_MODE_INPUT AND NOT "DB2001_MODES_GENERAL".GENERAL.JOG_INPUT AND NOT "DB2001_MODES_GENERAL".GENERAL.TOOL_CHANGE_MODE_SELECTED;
END_REGION

REGION Network 15: MODE SELECTED MEMORIES
   RUNG wire#powerrail
      Contact( #O_BYTE_0.MODE_SELECTED_MEMORY )
      wire#w1
      Contact( "DB2440_GLOBAL_DATA".GLOBAL_DATA.ANY_MACHINE_CYCLE_RUN )
      wire#w2
      I_Contact( "DB2001_MODES_GENERAL".GENERAL.OPTIONS.SGM )
      wire#w3
      Contact( "DB2001_MODES_GENERAL".GENERAL.AUTOMATIC_REQUEST )
      I_Contact( "DB2001_MODES_GENERAL".GENERAL.SINGLE_SELECTED_MEMORY )
      I_Contact( "DB2001_MODES_GENERAL".GENERAL.SEMI_SELECTED_MEMORY )
      I_Contact( "DB2001_MODES_GENERAL".GENERAL.MANUAL_SELECTED_MEMORY )
      S_Coil( "DB2001_MODES_GENERAL".GENERAL.AUTO_SELECTED_MEMORY )
   END_RUNG
   RUNG wire#w1
      Contact( "DB1101_MACHINE_SEQUENCE".RUNNING )
   END_RUNG wire#w2
   RUNG wire#w3
      Contact( "DB2001_MODES_GENERAL".GENERAL.SINGLE_REQUEST )
      I_Contact( "DB2001_MODES_GENERAL".GENERAL.AUTO_SELECTED_MEMORY )
      I_Contact( "DB2001_MODES_GENERAL".GENERAL.SEMI_SELECTED_MEMORY )
      I_Contact( "DB2001_MODES_GENERAL".GENERAL.MANUAL_SELECTED_MEMORY )
      S_Coil( "DB2001_MODES_GENERAL".GENERAL.SINGLE_SELECTED_MEMORY )
   END_RUNG
   RUNG wire#w3
      Contact( "DB2001_MODES_GENERAL".GENERAL.SEMIAUTO_REQUEST )
      I_Contact( "DB2001_MODES_GENERAL".GENERAL.AUTO_SELECTED_MEMORY )
      I_Contact( "DB2001_MODES_GENERAL".GENERAL.SINGLE_SELECTED_MEMORY )
      I_Contact( "DB2001_MODES_GENERAL".GENERAL.MANUAL_SELECTED_MEMORY )
      S_Coil( "DB2001_MODES_GENERAL".GENERAL.SEMI_SELECTED_MEMORY )
   END_RUNG
   RUNG wire#w3
      Contact( "DB2001_MODES_GENERAL".GENERAL.MANUAL_REQUEST )
      I_Contact( "DB2001_MODES_GENERAL".GENERAL.AUTO_SELECTED_MEMORY )
      I_Contact( "DB2001_MODES_GENERAL".GENERAL.SINGLE_SELECTED_MEMORY )
      I_Contact( "DB2001_MODES_GENERAL".GENERAL.SEMI_SELECTED_MEMORY )
      S_Coil( "DB2001_MODES_GENERAL".GENERAL.MANUAL_SELECTED_MEMORY )
   END_RUNG
   // the same network as SCL:
   #_w1 := #O_BYTE_0.MODE_SELECTED_MEMORY AND ("DB2440_GLOBAL_DATA".GLOBAL_DATA.ANY_MACHINE_CYCLE_RUN OR "DB1101_MACHINE_SEQUENCE".RUNNING) AND NOT "DB2001_MODES_GENERAL".GENERAL.OPTIONS.SGM;
   IF #_w1 AND "DB2001_MODES_GENERAL".GENERAL.AUTOMATIC_REQUEST AND NOT "DB2001_MODES_GENERAL".GENERAL.SINGLE_SELECTED_MEMORY AND NOT "DB2001_MODES_GENERAL".GENERAL.SEMI_SELECTED_MEMORY AND NOT "DB2001_MODES_GENERAL".GENERAL.MANUAL_SELECTED_MEMORY THEN
       "DB2001_MODES_GENERAL".GENERAL.AUTO_SELECTED_MEMORY := TRUE;
   END_IF;
   IF #_w1 AND "DB2001_MODES_GENERAL".GENERAL.SINGLE_REQUEST AND NOT "DB2001_MODES_GENERAL".GENERAL.AUTO_SELECTED_MEMORY AND NOT "DB2001_MODES_GENERAL".GENERAL.SEMI_SELECTED_MEMORY AND NOT "DB2001_MODES_GENERAL".GENERAL.MANUAL_SELECTED_MEMORY THEN
       "DB2001_MODES_GENERAL".GENERAL.SINGLE_SELECTED_MEMORY := TRUE;
   END_IF;
   IF #_w1 AND "DB2001_MODES_GENERAL".GENERAL.SEMIAUTO_REQUEST AND NOT "DB2001_MODES_GENERAL".GENERAL.AUTO_SELECTED_MEMORY AND NOT "DB2001_MODES_GENERAL".GENERAL.SINGLE_SELECTED_MEMORY AND NOT "DB2001_MODES_GENERAL".GENERAL.MANUAL_SELECTED_MEMORY THEN
       "DB2001_MODES_GENERAL".GENERAL.SEMI_SELECTED_MEMORY := TRUE;
   END_IF;
   IF #_w1 AND "DB2001_MODES_GENERAL".GENERAL.MANUAL_REQUEST AND NOT "DB2001_MODES_GENERAL".GENERAL.AUTO_SELECTED_MEMORY AND NOT "DB2001_MODES_GENERAL".GENERAL.SINGLE_SELECTED_MEMORY AND NOT "DB2001_MODES_GENERAL".GENERAL.SEMI_SELECTED_MEMORY THEN
       "DB2001_MODES_GENERAL".GENERAL.MANUAL_SELECTED_MEMORY := TRUE;
   END_IF;
END_REGION

REGION Network 16: CHANGE MODE
   RUNG wire#powerrail
      Contact( "DB2001_MODES_GENERAL".GENERAL.CHANGE_GENERAL_CONDITIONS )
      wire#w1
      Contact( "DB2001_MODES_GENERAL".GENERAL.AUTOMATIC_REQUEST )
      Coil( "DB2001_MODES_GENERAL".GENERAL.CHANGE_TO_AUTOMATIC )
   END_RUNG
   RUNG wire#w1
      Contact( "DB2001_MODES_GENERAL".GENERAL.SINGLE_REQUEST )
      Coil( "DB2001_MODES_GENERAL".GENERAL.CHANGE_TO_SINGLE )
   END_RUNG
   RUNG wire#w1
      Contact( "DB2001_MODES_GENERAL".GENERAL.SEMIAUTO_REQUEST )
      Coil( "DB2001_MODES_GENERAL".GENERAL.CHANGE_TO_SEMIAUTO )
   END_RUNG
   RUNG wire#w1
      Contact( "DB2001_MODES_GENERAL".GENERAL.MANUAL_REQUEST )
      Coil( "DB2001_MODES_GENERAL".GENERAL.CHANGE_TO_MANUAL )
   END_RUNG
   RUNG wire#w1
      Contact( "DB2001_MODES_GENERAL".GENERAL.NO_MODE_REQUEST )
      Coil( "DB2001_MODES_GENERAL".GENERAL.CHANGE_TO_NO_MODE )
   END_RUNG
   RUNG wire#w1
      Contact( "DB2001_MODES_GENERAL".GENERAL.JOG_REQUEST )
      Coil( "DB2001_MODES_GENERAL".GENERAL.CHANGE_TO_JOG_MODE )
   END_RUNG
   RUNG wire#w1
      Contact( "DB2001_MODES_GENERAL".GENERAL.TOOL_CHANGE_REQUEST )
      Coil( "DB2001_MODES_GENERAL".GENERAL.CHANGE_TO_TOOL_CHG_MODE )
   END_RUNG
   // the same network as SCL:
   "DB2001_MODES_GENERAL".GENERAL.CHANGE_TO_AUTOMATIC := "DB2001_MODES_GENERAL".GENERAL.CHANGE_GENERAL_CONDITIONS AND "DB2001_MODES_GENERAL".GENERAL.AUTOMATIC_REQUEST;
   "DB2001_MODES_GENERAL".GENERAL.CHANGE_TO_SINGLE := "DB2001_MODES_GENERAL".GENERAL.CHANGE_GENERAL_CONDITIONS AND "DB2001_MODES_GENERAL".GENERAL.SINGLE_REQUEST;
   "DB2001_MODES_GENERAL".GENERAL.CHANGE_TO_SEMIAUTO := "DB2001_MODES_GENERAL".GENERAL.CHANGE_GENERAL_CONDITIONS AND "DB2001_MODES_GENERAL".GENERAL.SEMIAUTO_REQUEST;
   "DB2001_MODES_GENERAL".GENERAL.CHANGE_TO_MANUAL := "DB2001_MODES_GENERAL".GENERAL.CHANGE_GENERAL_CONDITIONS AND "DB2001_MODES_GENERAL".GENERAL.MANUAL_REQUEST;
   "DB2001_MODES_GENERAL".GENERAL.CHANGE_TO_NO_MODE := "DB2001_MODES_GENERAL".GENERAL.CHANGE_GENERAL_CONDITIONS AND "DB2001_MODES_GENERAL".GENERAL.NO_MODE_REQUEST;
   "DB2001_MODES_GENERAL".GENERAL.CHANGE_TO_JOG_MODE := "DB2001_MODES_GENERAL".GENERAL.CHANGE_GENERAL_CONDITIONS AND "DB2001_MODES_GENERAL".GENERAL.JOG_REQUEST;
   "DB2001_MODES_GENERAL".GENERAL.CHANGE_TO_TOOL_CHG_MODE := "DB2001_MODES_GENERAL".GENERAL.CHANGE_GENERAL_CONDITIONS AND "DB2001_MODES_GENERAL".GENERAL.TOOL_CHANGE_REQUEST;
END_REGION

REGION Network 17: AUTOMATIC SELECTED
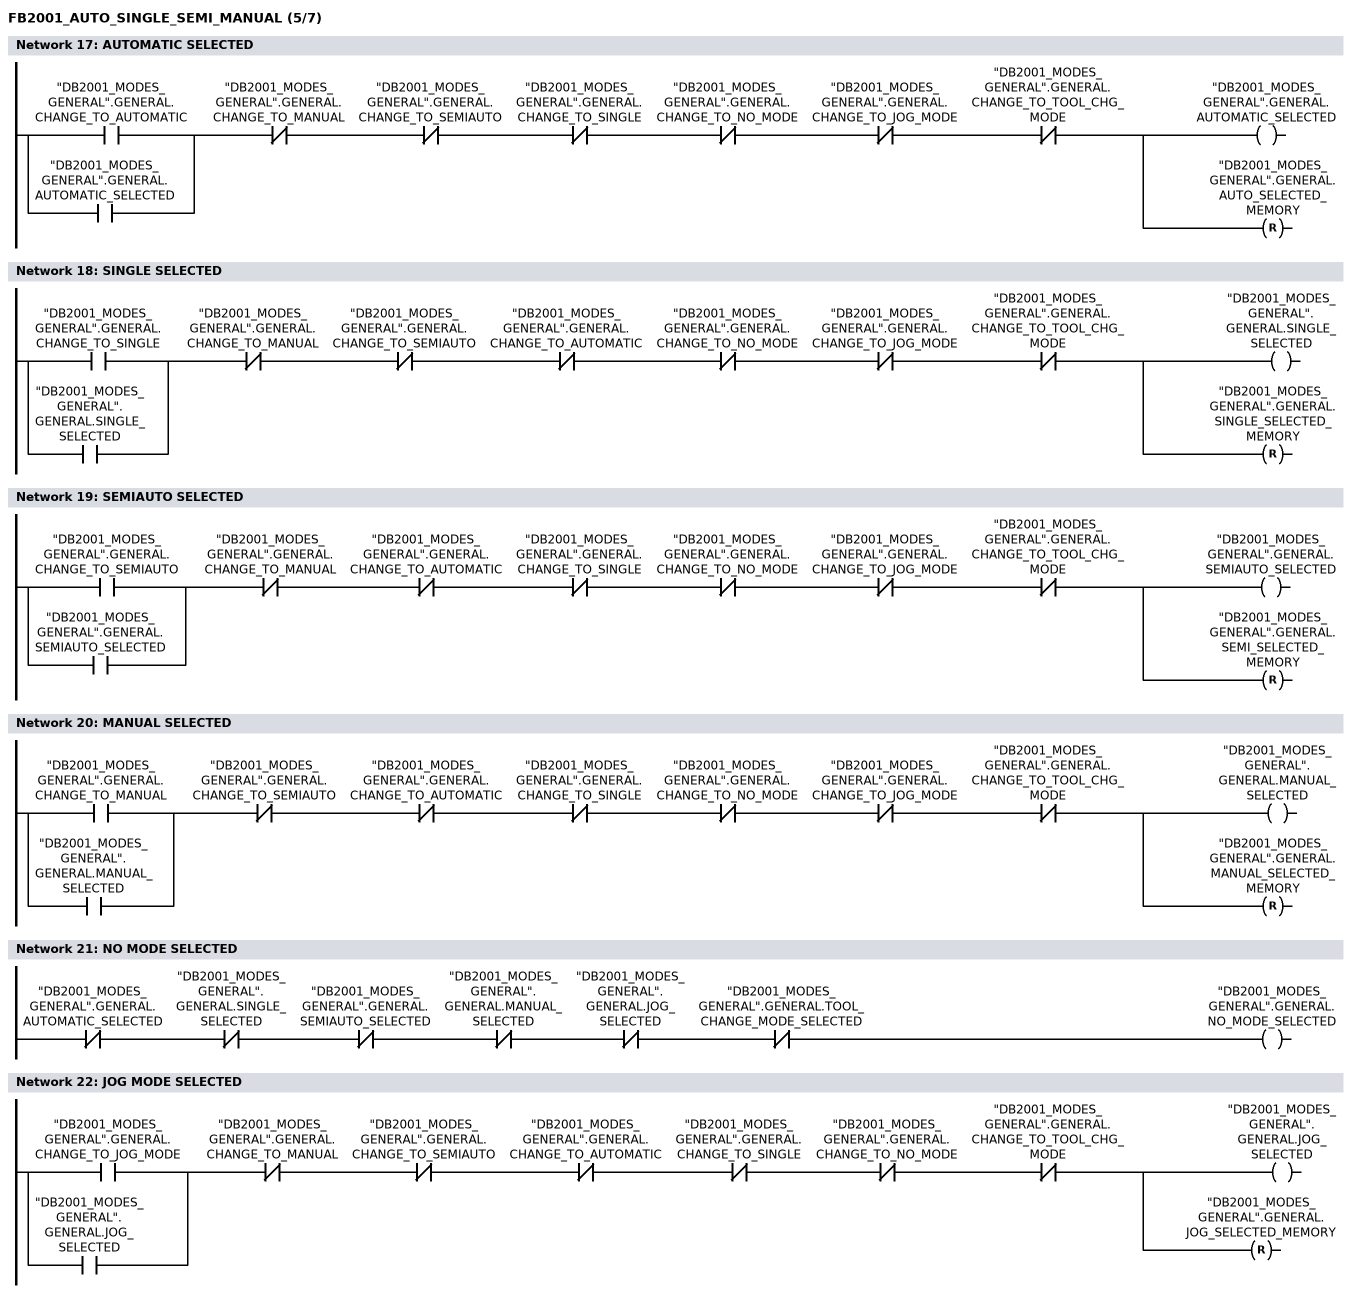
   RUNG wire#powerrail
      Contact( "DB2001_MODES_GENERAL".GENERAL.CHANGE_TO_AUTOMATIC )
      wire#w1
      I_Contact( "DB2001_MODES_GENERAL".GENERAL.CHANGE_TO_MANUAL )
      I_Contact( "DB2001_MODES_GENERAL".GENERAL.CHANGE_TO_SEMIAUTO )
      I_Contact( "DB2001_MODES_GENERAL".GENERAL.CHANGE_TO_SINGLE )
      I_Contact( "DB2001_MODES_GENERAL".GENERAL.CHANGE_TO_NO_MODE )
      I_Contact( "DB2001_MODES_GENERAL".GENERAL.CHANGE_TO_JOG_MODE )
      I_Contact( "DB2001_MODES_GENERAL".GENERAL.CHANGE_TO_TOOL_CHG_MODE )
      wire#w2
      Coil( "DB2001_MODES_GENERAL".GENERAL.AUTOMATIC_SELECTED )
   END_RUNG
   RUNG wire#powerrail
      Contact( "DB2001_MODES_GENERAL".GENERAL.AUTOMATIC_SELECTED )
   END_RUNG wire#w1
   RUNG wire#w2
      R_Coil( "DB2001_MODES_GENERAL".GENERAL.AUTO_SELECTED_MEMORY )
   END_RUNG
   // the same network as SCL:
   "DB2001_MODES_GENERAL".GENERAL.AUTOMATIC_SELECTED := ("DB2001_MODES_GENERAL".GENERAL.CHANGE_TO_AUTOMATIC OR "DB2001_MODES_GENERAL".GENERAL.AUTOMATIC_SELECTED) AND NOT "DB2001_MODES_GENERAL".GENERAL.CHANGE_TO_MANUAL AND NOT "DB2001_MODES_GENERAL".GENERAL.CHANGE_TO_SEMIAUTO AND NOT "DB2001_MODES_GENERAL".GENERAL.CHANGE_TO_SINGLE AND NOT "DB2001_MODES_GENERAL".GENERAL.CHANGE_TO_NO_MODE AND NOT "DB2001_MODES_GENERAL".GENERAL.CHANGE_TO_JOG_MODE AND NOT "DB2001_MODES_GENERAL".GENERAL.CHANGE_TO_TOOL_CHG_MODE;
   IF "DB2001_MODES_GENERAL".GENERAL.AUTOMATIC_SELECTED THEN
       "DB2001_MODES_GENERAL".GENERAL.AUTO_SELECTED_MEMORY := FALSE;
   END_IF;
END_REGION

REGION Network 18: SINGLE SELECTED
   RUNG wire#powerrail
      Contact( "DB2001_MODES_GENERAL".GENERAL.CHANGE_TO_SINGLE )
      wire#w1
      I_Contact( "DB2001_MODES_GENERAL".GENERAL.CHANGE_TO_MANUAL )
      I_Contact( "DB2001_MODES_GENERAL".GENERAL.CHANGE_TO_SEMIAUTO )
      I_Contact( "DB2001_MODES_GENERAL".GENERAL.CHANGE_TO_AUTOMATIC )
      I_Contact( "DB2001_MODES_GENERAL".GENERAL.CHANGE_TO_NO_MODE )
      I_Contact( "DB2001_MODES_GENERAL".GENERAL.CHANGE_TO_JOG_MODE )
      I_Contact( "DB2001_MODES_GENERAL".GENERAL.CHANGE_TO_TOOL_CHG_MODE )
      wire#w2
      Coil( "DB2001_MODES_GENERAL".GENERAL.SINGLE_SELECTED )
   END_RUNG
   RUNG wire#powerrail
      Contact( "DB2001_MODES_GENERAL".GENERAL.SINGLE_SELECTED )
   END_RUNG wire#w1
   RUNG wire#w2
      R_Coil( "DB2001_MODES_GENERAL".GENERAL.SINGLE_SELECTED_MEMORY )
   END_RUNG
   // the same network as SCL:
   "DB2001_MODES_GENERAL".GENERAL.SINGLE_SELECTED := ("DB2001_MODES_GENERAL".GENERAL.CHANGE_TO_SINGLE OR "DB2001_MODES_GENERAL".GENERAL.SINGLE_SELECTED) AND NOT "DB2001_MODES_GENERAL".GENERAL.CHANGE_TO_MANUAL AND NOT "DB2001_MODES_GENERAL".GENERAL.CHANGE_TO_SEMIAUTO AND NOT "DB2001_MODES_GENERAL".GENERAL.CHANGE_TO_AUTOMATIC AND NOT "DB2001_MODES_GENERAL".GENERAL.CHANGE_TO_NO_MODE AND NOT "DB2001_MODES_GENERAL".GENERAL.CHANGE_TO_JOG_MODE AND NOT "DB2001_MODES_GENERAL".GENERAL.CHANGE_TO_TOOL_CHG_MODE;
   IF "DB2001_MODES_GENERAL".GENERAL.SINGLE_SELECTED THEN
       "DB2001_MODES_GENERAL".GENERAL.SINGLE_SELECTED_MEMORY := FALSE;
   END_IF;
END_REGION

REGION Network 19: SEMIAUTO SELECTED
   RUNG wire#powerrail
      Contact( "DB2001_MODES_GENERAL".GENERAL.CHANGE_TO_SEMIAUTO )
      wire#w1
      I_Contact( "DB2001_MODES_GENERAL".GENERAL.CHANGE_TO_MANUAL )
      I_Contact( "DB2001_MODES_GENERAL".GENERAL.CHANGE_TO_AUTOMATIC )
      I_Contact( "DB2001_MODES_GENERAL".GENERAL.CHANGE_TO_SINGLE )
      I_Contact( "DB2001_MODES_GENERAL".GENERAL.CHANGE_TO_NO_MODE )
      I_Contact( "DB2001_MODES_GENERAL".GENERAL.CHANGE_TO_JOG_MODE )
      I_Contact( "DB2001_MODES_GENERAL".GENERAL.CHANGE_TO_TOOL_CHG_MODE )
      wire#w2
      Coil( "DB2001_MODES_GENERAL".GENERAL.SEMIAUTO_SELECTED )
   END_RUNG
   RUNG wire#powerrail
      Contact( "DB2001_MODES_GENERAL".GENERAL.SEMIAUTO_SELECTED )
   END_RUNG wire#w1
   RUNG wire#w2
      R_Coil( "DB2001_MODES_GENERAL".GENERAL.SEMI_SELECTED_MEMORY )
   END_RUNG
   // the same network as SCL:
   "DB2001_MODES_GENERAL".GENERAL.SEMIAUTO_SELECTED := ("DB2001_MODES_GENERAL".GENERAL.CHANGE_TO_SEMIAUTO OR "DB2001_MODES_GENERAL".GENERAL.SEMIAUTO_SELECTED) AND NOT "DB2001_MODES_GENERAL".GENERAL.CHANGE_TO_MANUAL AND NOT "DB2001_MODES_GENERAL".GENERAL.CHANGE_TO_AUTOMATIC AND NOT "DB2001_MODES_GENERAL".GENERAL.CHANGE_TO_SINGLE AND NOT "DB2001_MODES_GENERAL".GENERAL.CHANGE_TO_NO_MODE AND NOT "DB2001_MODES_GENERAL".GENERAL.CHANGE_TO_JOG_MODE AND NOT "DB2001_MODES_GENERAL".GENERAL.CHANGE_TO_TOOL_CHG_MODE;
   IF "DB2001_MODES_GENERAL".GENERAL.SEMIAUTO_SELECTED THEN
       "DB2001_MODES_GENERAL".GENERAL.SEMI_SELECTED_MEMORY := FALSE;
   END_IF;
END_REGION

REGION Network 20: MANUAL SELECTED
   RUNG wire#powerrail
      Contact( "DB2001_MODES_GENERAL".GENERAL.CHANGE_TO_MANUAL )
      wire#w1
      I_Contact( "DB2001_MODES_GENERAL".GENERAL.CHANGE_TO_SEMIAUTO )
      I_Contact( "DB2001_MODES_GENERAL".GENERAL.CHANGE_TO_AUTOMATIC )
      I_Contact( "DB2001_MODES_GENERAL".GENERAL.CHANGE_TO_SINGLE )
      I_Contact( "DB2001_MODES_GENERAL".GENERAL.CHANGE_TO_NO_MODE )
      I_Contact( "DB2001_MODES_GENERAL".GENERAL.CHANGE_TO_JOG_MODE )
      I_Contact( "DB2001_MODES_GENERAL".GENERAL.CHANGE_TO_TOOL_CHG_MODE )
      wire#w2
      Coil( "DB2001_MODES_GENERAL".GENERAL.MANUAL_SELECTED )
   END_RUNG
   RUNG wire#powerrail
      Contact( "DB2001_MODES_GENERAL".GENERAL.MANUAL_SELECTED )
   END_RUNG wire#w1
   RUNG wire#w2
      R_Coil( "DB2001_MODES_GENERAL".GENERAL.MANUAL_SELECTED_MEMORY )
   END_RUNG
   // the same network as SCL:
   "DB2001_MODES_GENERAL".GENERAL.MANUAL_SELECTED := ("DB2001_MODES_GENERAL".GENERAL.CHANGE_TO_MANUAL OR "DB2001_MODES_GENERAL".GENERAL.MANUAL_SELECTED) AND NOT "DB2001_MODES_GENERAL".GENERAL.CHANGE_TO_SEMIAUTO AND NOT "DB2001_MODES_GENERAL".GENERAL.CHANGE_TO_AUTOMATIC AND NOT "DB2001_MODES_GENERAL".GENERAL.CHANGE_TO_SINGLE AND NOT "DB2001_MODES_GENERAL".GENERAL.CHANGE_TO_NO_MODE AND NOT "DB2001_MODES_GENERAL".GENERAL.CHANGE_TO_JOG_MODE AND NOT "DB2001_MODES_GENERAL".GENERAL.CHANGE_TO_TOOL_CHG_MODE;
   IF "DB2001_MODES_GENERAL".GENERAL.MANUAL_SELECTED THEN
       "DB2001_MODES_GENERAL".GENERAL.MANUAL_SELECTED_MEMORY := FALSE;
   END_IF;
END_REGION

REGION Network 21: NO MODE SELECTED
   RUNG wire#powerrail
      I_Contact( "DB2001_MODES_GENERAL".GENERAL.AUTOMATIC_SELECTED )
      I_Contact( "DB2001_MODES_GENERAL".GENERAL.SINGLE_SELECTED )
      I_Contact( "DB2001_MODES_GENERAL".GENERAL.SEMIAUTO_SELECTED )
      I_Contact( "DB2001_MODES_GENERAL".GENERAL.MANUAL_SELECTED )
      I_Contact( "DB2001_MODES_GENERAL".GENERAL.JOG_SELECTED )
      I_Contact( "DB2001_MODES_GENERAL".GENERAL.TOOL_CHANGE_MODE_SELECTED )
      Coil( "DB2001_MODES_GENERAL".GENERAL.NO_MODE_SELECTED )
   END_RUNG
   // the same network as SCL:
   "DB2001_MODES_GENERAL".GENERAL.NO_MODE_SELECTED := NOT "DB2001_MODES_GENERAL".GENERAL.AUTOMATIC_SELECTED AND NOT "DB2001_MODES_GENERAL".GENERAL.SINGLE_SELECTED AND NOT "DB2001_MODES_GENERAL".GENERAL.SEMIAUTO_SELECTED AND NOT "DB2001_MODES_GENERAL".GENERAL.MANUAL_SELECTED AND NOT "DB2001_MODES_GENERAL".GENERAL.JOG_SELECTED AND NOT "DB2001_MODES_GENERAL".GENERAL.TOOL_CHANGE_MODE_SELECTED;
END_REGION

REGION Network 22: JOG MODE SELECTED
   RUNG wire#powerrail
      Contact( "DB2001_MODES_GENERAL".GENERAL.CHANGE_TO_JOG_MODE )
      wire#w1
      I_Contact( "DB2001_MODES_GENERAL".GENERAL.CHANGE_TO_MANUAL )
      I_Contact( "DB2001_MODES_GENERAL".GENERAL.CHANGE_TO_SEMIAUTO )
      I_Contact( "DB2001_MODES_GENERAL".GENERAL.CHANGE_TO_AUTOMATIC )
      I_Contact( "DB2001_MODES_GENERAL".GENERAL.CHANGE_TO_SINGLE )
      I_Contact( "DB2001_MODES_GENERAL".GENERAL.CHANGE_TO_NO_MODE )
      I_Contact( "DB2001_MODES_GENERAL".GENERAL.CHANGE_TO_TOOL_CHG_MODE )
      wire#w2
      Coil( "DB2001_MODES_GENERAL".GENERAL.JOG_SELECTED )
   END_RUNG
   RUNG wire#powerrail
      Contact( "DB2001_MODES_GENERAL".GENERAL.JOG_SELECTED )
   END_RUNG wire#w1
   RUNG wire#w2
      R_Coil( "DB2001_MODES_GENERAL".GENERAL.JOG_SELECTED_MEMORY )
   END_RUNG
   // the same network as SCL:
   "DB2001_MODES_GENERAL".GENERAL.JOG_SELECTED := ("DB2001_MODES_GENERAL".GENERAL.CHANGE_TO_JOG_MODE OR "DB2001_MODES_GENERAL".GENERAL.JOG_SELECTED) AND NOT "DB2001_MODES_GENERAL".GENERAL.CHANGE_TO_MANUAL AND NOT "DB2001_MODES_GENERAL".GENERAL.CHANGE_TO_SEMIAUTO AND NOT "DB2001_MODES_GENERAL".GENERAL.CHANGE_TO_AUTOMATIC AND NOT "DB2001_MODES_GENERAL".GENERAL.CHANGE_TO_SINGLE AND NOT "DB2001_MODES_GENERAL".GENERAL.CHANGE_TO_NO_MODE AND NOT "DB2001_MODES_GENERAL".GENERAL.CHANGE_TO_TOOL_CHG_MODE;
   IF "DB2001_MODES_GENERAL".GENERAL.JOG_SELECTED THEN
       "DB2001_MODES_GENERAL".GENERAL.JOG_SELECTED_MEMORY := FALSE;
   END_IF;
END_REGION

REGION Network 23: AUTO SINGLE SEMI SELECTED
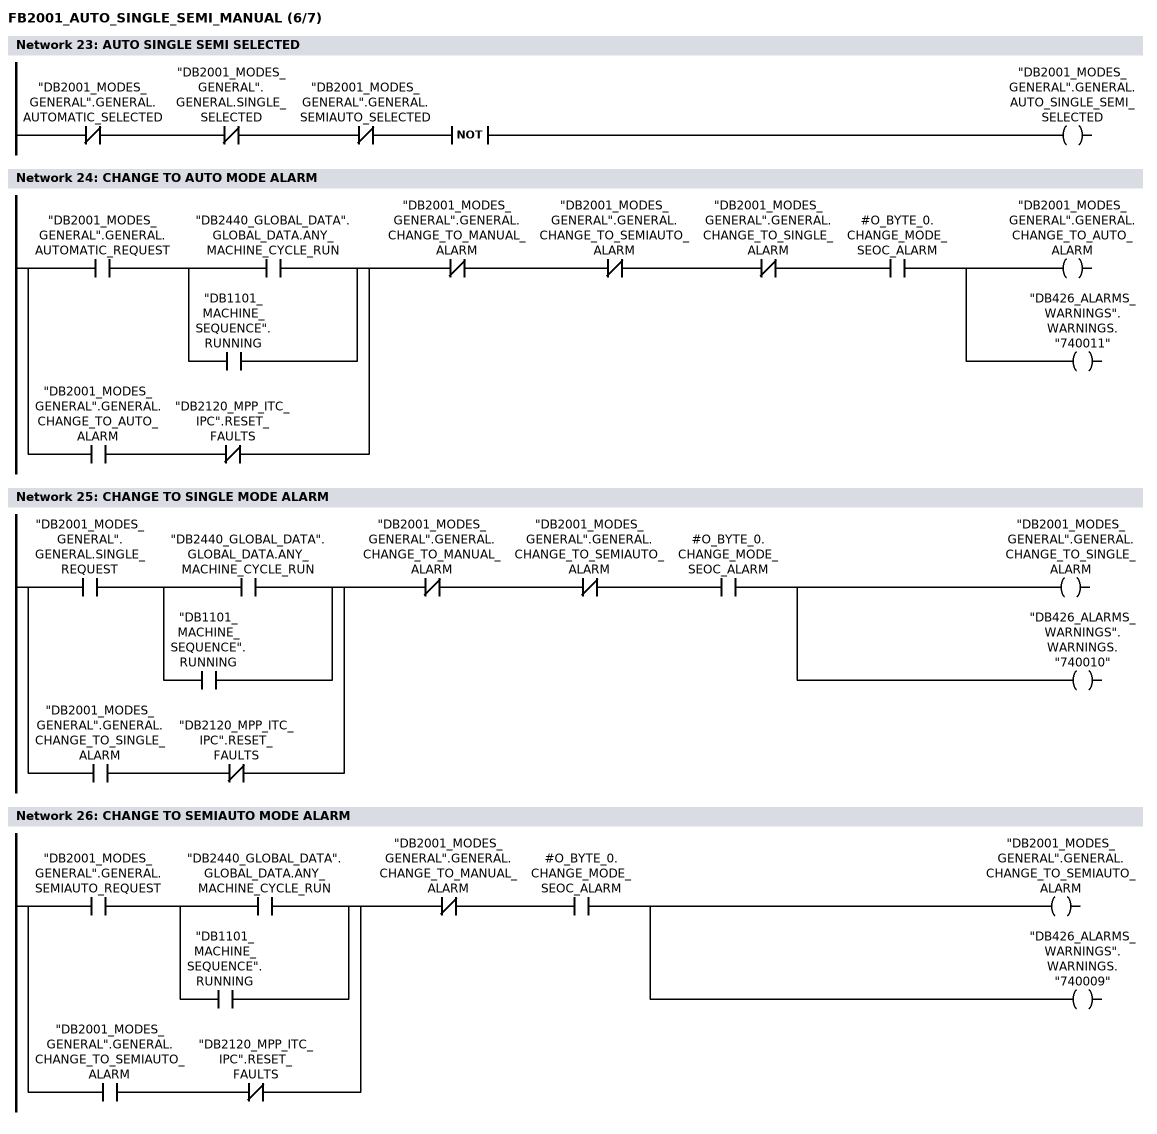
   RUNG wire#powerrail
      I_Contact( "DB2001_MODES_GENERAL".GENERAL.AUTOMATIC_SELECTED )
      I_Contact( "DB2001_MODES_GENERAL".GENERAL.SINGLE_SELECTED )
      I_Contact( "DB2001_MODES_GENERAL".GENERAL.SEMIAUTO_SELECTED )
      Not()
      Coil( "DB2001_MODES_GENERAL".GENERAL.AUTO_SINGLE_SEMI_SELECTED )
   END_RUNG
   // the same network as SCL:
   "DB2001_MODES_GENERAL".GENERAL.AUTO_SINGLE_SEMI_SELECTED := NOT (NOT "DB2001_MODES_GENERAL".GENERAL.AUTOMATIC_SELECTED AND NOT "DB2001_MODES_GENERAL".GENERAL.SINGLE_SELECTED AND NOT "DB2001_MODES_GENERAL".GENERAL.SEMIAUTO_SELECTED);
END_REGION

REGION Network 24: CHANGE TO AUTO MODE ALARM
   RUNG wire#powerrail
      Contact( "DB2001_MODES_GENERAL".GENERAL.AUTOMATIC_REQUEST )
      wire#w1
      Contact( "DB2440_GLOBAL_DATA".GLOBAL_DATA.ANY_MACHINE_CYCLE_RUN )
      wire#w2
      I_Contact( "DB2001_MODES_GENERAL".GENERAL.CHANGE_TO_MANUAL_ALARM )
      I_Contact( "DB2001_MODES_GENERAL".GENERAL.CHANGE_TO_SEMIAUTO_ALARM )
      I_Contact( "DB2001_MODES_GENERAL".GENERAL.CHANGE_TO_SINGLE_ALARM )
      Contact( #O_BYTE_0.CHANGE_MODE_SEOC_ALARM )
      wire#w3
      Coil( "DB2001_MODES_GENERAL".GENERAL.CHANGE_TO_AUTO_ALARM )
   END_RUNG
   RUNG wire#w1
      Contact( "DB1101_MACHINE_SEQUENCE".RUNNING )
   END_RUNG wire#w2
   RUNG wire#powerrail
      Contact( "DB2001_MODES_GENERAL".GENERAL.CHANGE_TO_AUTO_ALARM )
      I_Contact( "DB2120_MPP_ITC_IPC".RESET_FAULTS )
   END_RUNG wire#w2
   RUNG wire#w3
      Coil( "DB426_ALARMS_WARNINGS".WARNINGS."740011" )
   END_RUNG
   // the same network as SCL:
   "DB2001_MODES_GENERAL".GENERAL.CHANGE_TO_AUTO_ALARM := (("DB2001_MODES_GENERAL".GENERAL.AUTOMATIC_REQUEST AND ("DB2440_GLOBAL_DATA".GLOBAL_DATA.ANY_MACHINE_CYCLE_RUN OR "DB1101_MACHINE_SEQUENCE".RUNNING)) OR ("DB2001_MODES_GENERAL".GENERAL.CHANGE_TO_AUTO_ALARM AND NOT "DB2120_MPP_ITC_IPC".RESET_FAULTS)) AND NOT "DB2001_MODES_GENERAL".GENERAL.CHANGE_TO_MANUAL_ALARM AND NOT "DB2001_MODES_GENERAL".GENERAL.CHANGE_TO_SEMIAUTO_ALARM AND NOT "DB2001_MODES_GENERAL".GENERAL.CHANGE_TO_SINGLE_ALARM AND #O_BYTE_0.CHANGE_MODE_SEOC_ALARM;
   "DB426_ALARMS_WARNINGS".WARNINGS."740011" := "DB2001_MODES_GENERAL".GENERAL.CHANGE_TO_AUTO_ALARM;
END_REGION

REGION Network 25: CHANGE TO SINGLE MODE ALARM
   RUNG wire#powerrail
      Contact( "DB2001_MODES_GENERAL".GENERAL.SINGLE_REQUEST )
      wire#w1
      Contact( "DB2440_GLOBAL_DATA".GLOBAL_DATA.ANY_MACHINE_CYCLE_RUN )
      wire#w2
      I_Contact( "DB2001_MODES_GENERAL".GENERAL.CHANGE_TO_MANUAL_ALARM )
      I_Contact( "DB2001_MODES_GENERAL".GENERAL.CHANGE_TO_SEMIAUTO_ALARM )
      Contact( #O_BYTE_0.CHANGE_MODE_SEOC_ALARM )
      wire#w3
      Coil( "DB2001_MODES_GENERAL".GENERAL.CHANGE_TO_SINGLE_ALARM )
   END_RUNG
   RUNG wire#w1
      Contact( "DB1101_MACHINE_SEQUENCE".RUNNING )
   END_RUNG wire#w2
   RUNG wire#powerrail
      Contact( "DB2001_MODES_GENERAL".GENERAL.CHANGE_TO_SINGLE_ALARM )
      I_Contact( "DB2120_MPP_ITC_IPC".RESET_FAULTS )
   END_RUNG wire#w2
   RUNG wire#w3
      Coil( "DB426_ALARMS_WARNINGS".WARNINGS."740010" )
   END_RUNG
   // the same network as SCL:
   "DB2001_MODES_GENERAL".GENERAL.CHANGE_TO_SINGLE_ALARM := (("DB2001_MODES_GENERAL".GENERAL.SINGLE_REQUEST AND ("DB2440_GLOBAL_DATA".GLOBAL_DATA.ANY_MACHINE_CYCLE_RUN OR "DB1101_MACHINE_SEQUENCE".RUNNING)) OR ("DB2001_MODES_GENERAL".GENERAL.CHANGE_TO_SINGLE_ALARM AND NOT "DB2120_MPP_ITC_IPC".RESET_FAULTS)) AND NOT "DB2001_MODES_GENERAL".GENERAL.CHANGE_TO_MANUAL_ALARM AND NOT "DB2001_MODES_GENERAL".GENERAL.CHANGE_TO_SEMIAUTO_ALARM AND #O_BYTE_0.CHANGE_MODE_SEOC_ALARM;
   "DB426_ALARMS_WARNINGS".WARNINGS."740010" := "DB2001_MODES_GENERAL".GENERAL.CHANGE_TO_SINGLE_ALARM;
END_REGION

REGION Network 26: CHANGE TO SEMIAUTO MODE ALARM
   RUNG wire#powerrail
      Contact( "DB2001_MODES_GENERAL".GENERAL.SEMIAUTO_REQUEST )
      wire#w1
      Contact( "DB2440_GLOBAL_DATA".GLOBAL_DATA.ANY_MACHINE_CYCLE_RUN )
      wire#w2
      I_Contact( "DB2001_MODES_GENERAL".GENERAL.CHANGE_TO_MANUAL_ALARM )
      Contact( #O_BYTE_0.CHANGE_MODE_SEOC_ALARM )
      wire#w3
      Coil( "DB2001_MODES_GENERAL".GENERAL.CHANGE_TO_SEMIAUTO_ALARM )
   END_RUNG
   RUNG wire#w1
      Contact( "DB1101_MACHINE_SEQUENCE".RUNNING )
   END_RUNG wire#w2
   RUNG wire#powerrail
      Contact( "DB2001_MODES_GENERAL".GENERAL.CHANGE_TO_SEMIAUTO_ALARM )
      I_Contact( "DB2120_MPP_ITC_IPC".RESET_FAULTS )
   END_RUNG wire#w2
   RUNG wire#w3
      Coil( "DB426_ALARMS_WARNINGS".WARNINGS."740009" )
   END_RUNG
   // the same network as SCL:
   "DB2001_MODES_GENERAL".GENERAL.CHANGE_TO_SEMIAUTO_ALARM := (("DB2001_MODES_GENERAL".GENERAL.SEMIAUTO_REQUEST AND ("DB2440_GLOBAL_DATA".GLOBAL_DATA.ANY_MACHINE_CYCLE_RUN OR "DB1101_MACHINE_SEQUENCE".RUNNING)) OR ("DB2001_MODES_GENERAL".GENERAL.CHANGE_TO_SEMIAUTO_ALARM AND NOT "DB2120_MPP_ITC_IPC".RESET_FAULTS)) AND NOT "DB2001_MODES_GENERAL".GENERAL.CHANGE_TO_MANUAL_ALARM AND #O_BYTE_0.CHANGE_MODE_SEOC_ALARM;
   "DB426_ALARMS_WARNINGS".WARNINGS."740009" := "DB2001_MODES_GENERAL".GENERAL.CHANGE_TO_SEMIAUTO_ALARM;
END_REGION

REGION Network 27: CHANGE TO MANUAL MODE ALARM
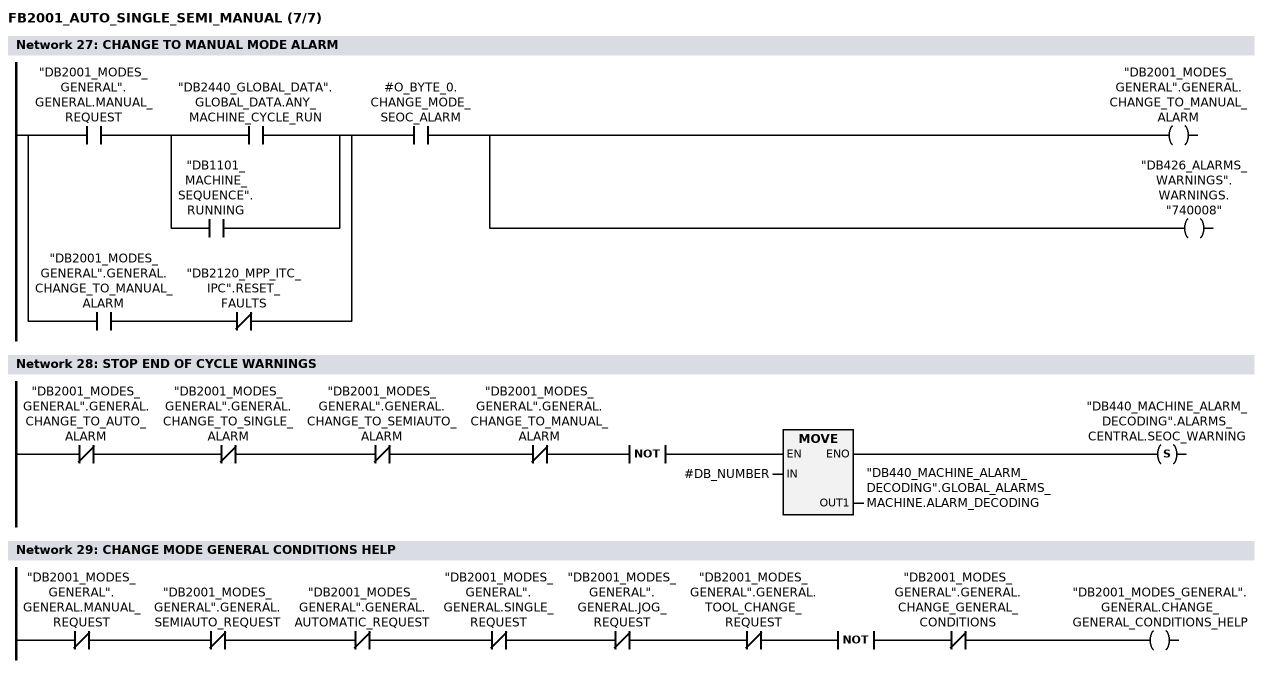
   RUNG wire#powerrail
      Contact( "DB2001_MODES_GENERAL".GENERAL.MANUAL_REQUEST )
      wire#w1
      Contact( "DB2440_GLOBAL_DATA".GLOBAL_DATA.ANY_MACHINE_CYCLE_RUN )
      wire#w2
      Contact( #O_BYTE_0.CHANGE_MODE_SEOC_ALARM )
      wire#w3
      Coil( "DB2001_MODES_GENERAL".GENERAL.CHANGE_TO_MANUAL_ALARM )
   END_RUNG
   RUNG wire#w1
      Contact( "DB1101_MACHINE_SEQUENCE".RUNNING )
   END_RUNG wire#w2
   RUNG wire#powerrail
      Contact( "DB2001_MODES_GENERAL".GENERAL.CHANGE_TO_MANUAL_ALARM )
      I_Contact( "DB2120_MPP_ITC_IPC".RESET_FAULTS )
   END_RUNG wire#w2
   RUNG wire#w3
      Coil( "DB426_ALARMS_WARNINGS".WARNINGS."740008" )
   END_RUNG
   // the same network as SCL:
   "DB2001_MODES_GENERAL".GENERAL.CHANGE_TO_MANUAL_ALARM := (("DB2001_MODES_GENERAL".GENERAL.MANUAL_REQUEST AND ("DB2440_GLOBAL_DATA".GLOBAL_DATA.ANY_MACHINE_CYCLE_RUN OR "DB1101_MACHINE_SEQUENCE".RUNNING)) OR ("DB2001_MODES_GENERAL".GENERAL.CHANGE_TO_MANUAL_ALARM AND NOT "DB2120_MPP_ITC_IPC".RESET_FAULTS)) AND #O_BYTE_0.CHANGE_MODE_SEOC_ALARM;
   "DB426_ALARMS_WARNINGS".WARNINGS."740008" := "DB2001_MODES_GENERAL".GENERAL.CHANGE_TO_MANUAL_ALARM;
END_REGION

REGION Network 28: STOP END OF CYCLE WARNINGS
   RUNG wire#powerrail
      I_Contact( "DB2001_MODES_GENERAL".GENERAL.CHANGE_TO_AUTO_ALARM )
      I_Contact( "DB2001_MODES_GENERAL".GENERAL.CHANGE_TO_SINGLE_ALARM )
      I_Contact( "DB2001_MODES_GENERAL".GENERAL.CHANGE_TO_SEMIAUTO_ALARM )
      I_Contact( "DB2001_MODES_GENERAL".GENERAL.CHANGE_TO_MANUAL_ALARM )
      Not()
      { S7_GenerateENO := "TRUE" } Move(in := #DB_NUMBER, out1 => "DB440_MACHINE_ALARM_DECODING".GLOBAL_ALARMS_MACHINE.ALARM_DECODING)
      S_Coil( "DB440_MACHINE_ALARM_DECODING".ALARMS_CENTRAL.SEOC_WARNING )
   END_RUNG
   // the same network as SCL:
   // ENO of a box is taken as its EN; it also drops when the box reports an error
   IF NOT (NOT "DB2001_MODES_GENERAL".GENERAL.CHANGE_TO_AUTO_ALARM AND NOT "DB2001_MODES_GENERAL".GENERAL.CHANGE_TO_SINGLE_ALARM AND NOT "DB2001_MODES_GENERAL".GENERAL.CHANGE_TO_SEMIAUTO_ALARM AND NOT "DB2001_MODES_GENERAL".GENERAL.CHANGE_TO_MANUAL_ALARM) THEN
       "DB440_MACHINE_ALARM_DECODING".GLOBAL_ALARMS_MACHINE.ALARM_DECODING := #DB_NUMBER;
       "DB440_MACHINE_ALARM_DECODING".ALARMS_CENTRAL.SEOC_WARNING := TRUE;
   END_IF;
END_REGION

REGION Network 29: CHANGE MODE GENERAL CONDITIONS HELP
   RUNG wire#powerrail
      I_Contact( "DB2001_MODES_GENERAL".GENERAL.MANUAL_REQUEST )
      I_Contact( "DB2001_MODES_GENERAL".GENERAL.SEMIAUTO_REQUEST )
      I_Contact( "DB2001_MODES_GENERAL".GENERAL.AUTOMATIC_REQUEST )
      I_Contact( "DB2001_MODES_GENERAL".GENERAL.SINGLE_REQUEST )
      I_Contact( "DB2001_MODES_GENERAL".GENERAL.JOG_REQUEST )
      I_Contact( "DB2001_MODES_GENERAL".GENERAL.TOOL_CHANGE_REQUEST )
      Not()
      I_Contact( "DB2001_MODES_GENERAL".GENERAL.CHANGE_GENERAL_CONDITIONS )
      Coil( "DB2001_MODES_GENERAL".GENERAL.CHANGE_GENERAL_CONDITIONS_HELP )
   END_RUNG
   // the same network as SCL:
   "DB2001_MODES_GENERAL".GENERAL.CHANGE_GENERAL_CONDITIONS_HELP := NOT (NOT "DB2001_MODES_GENERAL".GENERAL.MANUAL_REQUEST AND NOT "DB2001_MODES_GENERAL".GENERAL.SEMIAUTO_REQUEST AND NOT "DB2001_MODES_GENERAL".GENERAL.AUTOMATIC_REQUEST AND NOT "DB2001_MODES_GENERAL".GENERAL.SINGLE_REQUEST AND NOT "DB2001_MODES_GENERAL".GENERAL.JOG_REQUEST AND NOT "DB2001_MODES_GENERAL".GENERAL.TOOL_CHANGE_REQUEST) AND NOT "DB2001_MODES_GENERAL".GENERAL.CHANGE_GENERAL_CONDITIONS;
END_REGION
END_FUNCTION_BLOCK

FUNCTION_BLOCK "FB2002_BA_MODE"   // FB2002, LAD
{ S7_Optimized_Access := 'FALSE' }
VERSION : 0.1
// stored: AutoNumber false, IsIECCheckEnabled false, SetENOAutomatically false, UDAEnableTagReadback false
   VAR_INPUT
      OPTIONS_0 { ExternalAccessible := 'False'; ExternalVisible := 'False'; ExternalWritable := 'False'} : Byte := 2#0000_0000;   // OPTIONS BYTE 0
      BA1_BUTTON_I { ExternalAccessible := 'False'; ExternalVisible := 'False'; ExternalWritable := 'False'} : Bool;   // BA1 BUTTON INPUT
      BA2_BUTTON_I { ExternalAccessible := 'False'; ExternalVisible := 'False'; ExternalWritable := 'False'} : Bool;   // BA2 BUTTON INPUT
      BA3_BUTTON_I { ExternalAccessible := 'False'; ExternalVisible := 'False'; ExternalWritable := 'False'} : Bool;   // BA3 BUTTON INPUT
      BA5_BUTTON_I { ExternalAccessible := 'False'; ExternalVisible := 'False'; ExternalWritable := 'False'} : Bool;   // BA5 BUTTON INPUT
      SAFETY_ENABLED_W_DOOR_OPENED { ExternalAccessible := 'False'; ExternalVisible := 'False'; ExternalWritable := 'False'} : Bool;   // SAFETY ENABLED WITH DOOR OPENED (ENABLING DEVICE AND HT10 ENABLE BUTTON)
      SAFETY_GATES_CLSD_AND_LCKD { ExternalAccessible := 'False'; ExternalVisible := 'False'; ExternalWritable := 'False'} : Bool;   // SAFETY GATES CLOSED AND LOCKED
      START_SERVICES_GLOBAL { ExternalAccessible := 'False'; ExternalVisible := 'False'; ExternalWritable := 'False'} : Bool;   // START SERVICES GLOBAL
      ANY_MCH_CYCLE_RUN { ExternalAccessible := 'False'; ExternalVisible := 'False'; ExternalWritable := 'False'} : Bool;   // ANY MACHINE CYCLE RUNNING
      MCH_RESET_FAULTS { ExternalAccessible := 'False'; ExternalVisible := 'False'; ExternalWritable := 'False'} : Bool;   // MACHINE_RESET_FAULTS
   END_VAR
   VAR_OUTPUT
      NO_BA_MODE_SLCTD_WRN { ExternalAccessible := 'False'; ExternalVisible := 'False'; ExternalWritable := 'False'} : Bool;   // NO BA MODE SELECTED WARNING
      CHANGE_TO_BA1_MODE_WRN { ExternalAccessible := 'False'; ExternalVisible := 'False'; ExternalWritable := 'False'} : Bool;   // CHANGE TO BA1 MODE WARNING
      CHANGE_TO_BA2_MODE_WRN { ExternalAccessible := 'False'; ExternalVisible := 'False'; ExternalWritable := 'False'} : Bool;   // CHANGE TO BA2 MODE WARNING
      CHANGE_TO_BA3_MODE_WRN { ExternalAccessible := 'False'; ExternalVisible := 'False'; ExternalWritable := 'False'} : Bool;   // CHANGE TO BA3 MODE WARNING
      CHANGE_TO_BA5_MODE_WRN { ExternalAccessible := 'False'; ExternalVisible := 'False'; ExternalWritable := 'False'} : Bool;   // CHANGE TO BA5 MODE WARNING
      BA1_MODE_LED_O { ExternalAccessible := 'False'; ExternalVisible := 'False'; ExternalWritable := 'False'} : Bool;   // BA1 MODE BUTTON LED OUTPUT
      BA2_MODE_LED_O { ExternalAccessible := 'False'; ExternalVisible := 'False'; ExternalWritable := 'False'} : Bool;   // BA2 MODE BUTTON LED OUTPUT
      BA3_MODE_LED_O { ExternalAccessible := 'False'; ExternalVisible := 'False'; ExternalWritable := 'False'} : Bool;   // BA3 MODE BUTTON LED OUTPUT
   END_VAR
   VAR_IN_OUT
      MODE_GROUP_GENERAL_DB : "AUTO_SINGLE_SEMI_MANUAL";
      MODE_GROUP_BA_DB : "BA_MODE";
   END_VAR
   VAR_TEMP
      INPUTS_MASK : Byte;   // INPUT MASK
      O_BYTE_0 : Struct   // OPTIONS BYTE 0
         BA_BUTTONS : Bool;   // BA MODE BUTTONS OPTION
         CHANGE_MODE_SEOC_ALARM : Bool;   // CHANGE MODE SEOC ALARM OPTION
         MODE_SELECTED_MEMORY : Bool;   // MODE SELECTED MEMORY OPTION
         SPARE : Bool;
         SPARE_1 : Bool;
         SPARE_2 : Bool;
         SPARE_3 : Bool;
         SPARE_4 : Bool;
      END_STRUCT;
      DB_NUMBER : DInt;   // DB NUMBER FOR ALARM DECODING
   END_VAR
   VAR_TEMP   // added for the SCL form of the ladder/FBD networks
      _w1 : Bool;
      _w2 : Bool;
   END_VAR
BEGIN

NETWORK
TITLE = READ INSTANCE DB
      L     DINO;
      +     10#800000;
      T     #DB_NUMBER;


REGION Network 2: OPTIONS
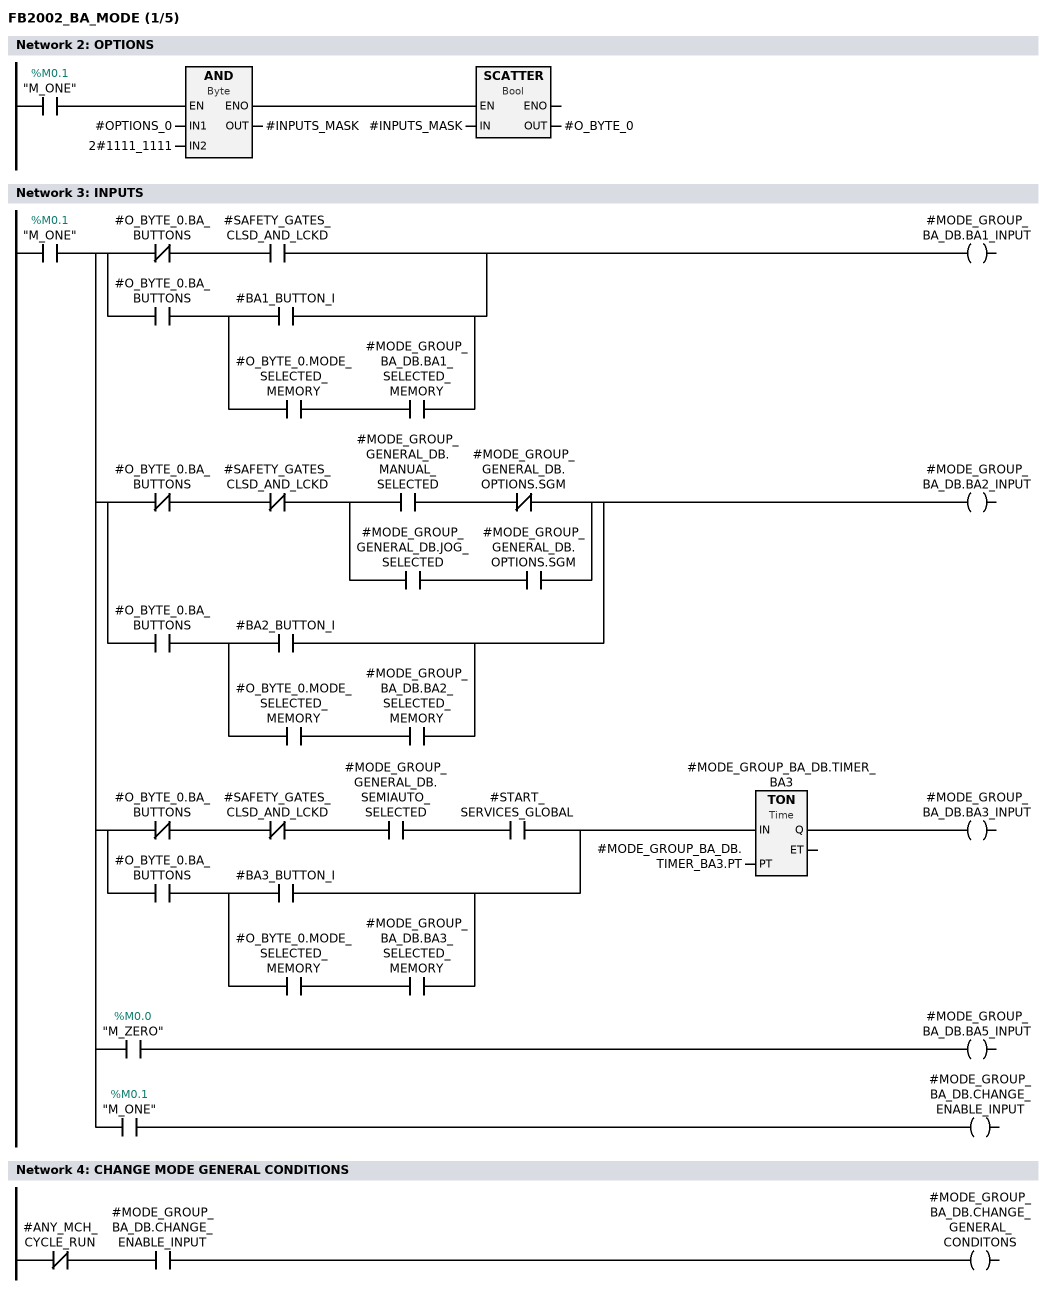
   RUNG wire#powerrail
      Contact( "M_ONE" )
      { S7_Templates := "SrcType := Byte"; S7_GenerateENO := "TRUE" } And(in1 := #OPTIONS_0, in2 := 2#1111_1111, out => #INPUTS_MASK)
      { S7_Templates := "[dest_type := Bool, src_type := Byte]" } SCATTER(IN := #INPUTS_MASK, OUT => #O_BYTE_0)
   END_RUNG
   // the same network as SCL:
   IF "M_ONE" THEN
       #INPUTS_MASK := #OPTIONS_0 AND 2#1111_1111;
       SCATTER(IN := #INPUTS_MASK, OUT => #O_BYTE_0);
   END_IF;
END_REGION

REGION Network 3: INPUTS
   RUNG wire#powerrail
      Contact( "M_ONE" )
      wire#w1
      I_Contact( #O_BYTE_0.BA_BUTTONS )
      Contact( #SAFETY_GATES_CLSD_AND_LCKD )
      wire#w2
      Coil( #MODE_GROUP_BA_DB.BA1_INPUT )
   END_RUNG
   RUNG wire#w1
      Contact( #O_BYTE_0.BA_BUTTONS )
      wire#w3
      Contact( #BA1_BUTTON_I )
   END_RUNG wire#w2
   RUNG wire#w3
      Contact( #O_BYTE_0.MODE_SELECTED_MEMORY )
      Contact( #MODE_GROUP_BA_DB.BA1_SELECTED_MEMORY )
   END_RUNG wire#w2
   RUNG wire#w1
      I_Contact( #O_BYTE_0.BA_BUTTONS )
      I_Contact( #SAFETY_GATES_CLSD_AND_LCKD )
      wire#w4
      Contact( #MODE_GROUP_GENERAL_DB.MANUAL_SELECTED )
      I_Contact( #MODE_GROUP_GENERAL_DB.OPTIONS.SGM )
      wire#w5
      Coil( #MODE_GROUP_BA_DB.BA2_INPUT )
   END_RUNG
   RUNG wire#w4
      Contact( #MODE_GROUP_GENERAL_DB.JOG_SELECTED )
      Contact( #MODE_GROUP_GENERAL_DB.OPTIONS.SGM )
   END_RUNG wire#w5
   RUNG wire#w1
      Contact( #O_BYTE_0.BA_BUTTONS )
      wire#w6
      Contact( #BA2_BUTTON_I )
   END_RUNG wire#w5
   RUNG wire#w6
      Contact( #O_BYTE_0.MODE_SELECTED_MEMORY )
      Contact( #MODE_GROUP_BA_DB.BA2_SELECTED_MEMORY )
   END_RUNG wire#w5
   RUNG wire#w1
      I_Contact( #O_BYTE_0.BA_BUTTONS )
      I_Contact( #SAFETY_GATES_CLSD_AND_LCKD )
      Contact( #MODE_GROUP_GENERAL_DB.SEMIAUTO_SELECTED )
      Contact( #START_SERVICES_GLOBAL )
      wire#w7
      { S7_Templates := "time_type := Time" } #MODE_GROUP_BA_DB.TIMER_BA3.TON(pt := #MODE_GROUP_BA_DB.TIMER_BA3.PT, et =>)
      Coil( #MODE_GROUP_BA_DB.BA3_INPUT )
   END_RUNG
   RUNG wire#w1
      Contact( #O_BYTE_0.BA_BUTTONS )
      wire#w8
      Contact( #BA3_BUTTON_I )
   END_RUNG wire#w7
   RUNG wire#w8
      Contact( #O_BYTE_0.MODE_SELECTED_MEMORY )
      Contact( #MODE_GROUP_BA_DB.BA3_SELECTED_MEMORY )
   END_RUNG wire#w7
   RUNG wire#w1
      Contact( "M_ZERO" )
      Coil( #MODE_GROUP_BA_DB.BA5_INPUT )
   END_RUNG
   RUNG wire#w1
      Contact( "M_ONE" )
      Coil( #MODE_GROUP_BA_DB.CHANGE_ENABLE_INPUT )
   END_RUNG
   // the same network as SCL:
   #MODE_GROUP_BA_DB.BA1_INPUT := "M_ONE" AND ((NOT #O_BYTE_0.BA_BUTTONS AND #SAFETY_GATES_CLSD_AND_LCKD) OR (#O_BYTE_0.BA_BUTTONS AND (#BA1_BUTTON_I OR (#O_BYTE_0.MODE_SELECTED_MEMORY AND #MODE_GROUP_BA_DB.BA1_SELECTED_MEMORY))));
   #MODE_GROUP_BA_DB.BA2_INPUT := "M_ONE" AND ((NOT #O_BYTE_0.BA_BUTTONS AND NOT #SAFETY_GATES_CLSD_AND_LCKD AND ((#MODE_GROUP_GENERAL_DB.MANUAL_SELECTED AND NOT #MODE_GROUP_GENERAL_DB.OPTIONS.SGM) OR (#MODE_GROUP_GENERAL_DB.JOG_SELECTED AND #MODE_GROUP_GENERAL_DB.OPTIONS.SGM))) OR (#O_BYTE_0.BA_BUTTONS AND (#BA2_BUTTON_I OR (#O_BYTE_0.MODE_SELECTED_MEMORY AND #MODE_GROUP_BA_DB.BA2_SELECTED_MEMORY))));
   #MODE_GROUP_BA_DB.TIMER_BA3.TON(IN := "M_ONE" AND ((NOT #O_BYTE_0.BA_BUTTONS AND NOT #SAFETY_GATES_CLSD_AND_LCKD AND #MODE_GROUP_GENERAL_DB.SEMIAUTO_SELECTED AND #START_SERVICES_GLOBAL) OR (#O_BYTE_0.BA_BUTTONS AND (#BA3_BUTTON_I OR (#O_BYTE_0.MODE_SELECTED_MEMORY AND #MODE_GROUP_BA_DB.BA3_SELECTED_MEMORY)))),
                           PT := #MODE_GROUP_BA_DB.TIMER_BA3.PT);
   #MODE_GROUP_BA_DB.BA3_INPUT := #MODE_GROUP_BA_DB.TIMER_BA3.Q;
   #MODE_GROUP_BA_DB.BA5_INPUT := "M_ONE" AND "M_ZERO";
   #MODE_GROUP_BA_DB.CHANGE_ENABLE_INPUT := "M_ONE" AND "M_ONE";
END_REGION

REGION Network 4: CHANGE MODE GENERAL CONDITIONS
   RUNG wire#powerrail
      I_Contact( #ANY_MCH_CYCLE_RUN )
      Contact( #MODE_GROUP_BA_DB.CHANGE_ENABLE_INPUT )
      Coil( #MODE_GROUP_BA_DB.CHANGE_GENERAL_CONDITONS )
   END_RUNG
   // the same network as SCL:
   #MODE_GROUP_BA_DB.CHANGE_GENERAL_CONDITONS := NOT #ANY_MCH_CYCLE_RUN AND #MODE_GROUP_BA_DB.CHANGE_ENABLE_INPUT;
END_REGION

REGION Network 5: OPERATOR HELP
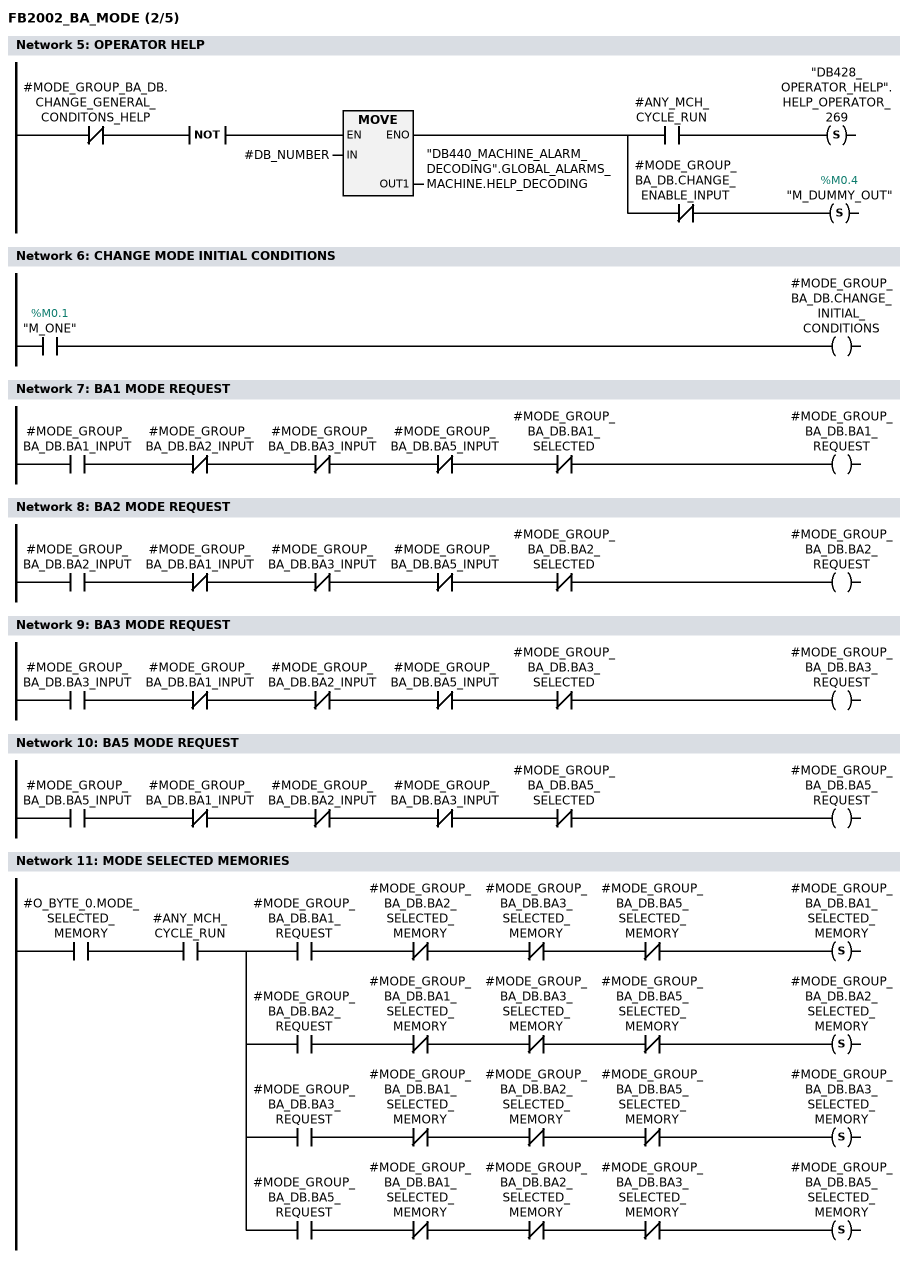
   RUNG wire#powerrail
      I_Contact( #MODE_GROUP_BA_DB.CHANGE_GENERAL_CONDITONS_HELP )
      Not()
      { S7_GenerateENO := "TRUE" } Move(in := #DB_NUMBER, out1 => "DB440_MACHINE_ALARM_DECODING".GLOBAL_ALARMS_MACHINE.HELP_DECODING)
      wire#w1
      Contact( #ANY_MCH_CYCLE_RUN )
      S_Coil( "DB428_OPERATOR_HELP".HELP_OPERATOR_269 )
   END_RUNG
   RUNG wire#w1
      I_Contact( #MODE_GROUP_BA_DB.CHANGE_ENABLE_INPUT )
      S_Coil( "M_DUMMY_OUT" )
   END_RUNG
   // the same network as SCL:
   // ENO of a box is taken as its EN; it also drops when the box reports an error
   #_w1 := NOT (NOT #MODE_GROUP_BA_DB.CHANGE_GENERAL_CONDITONS_HELP);
   IF #_w1 THEN "DB440_MACHINE_ALARM_DECODING".GLOBAL_ALARMS_MACHINE.HELP_DECODING := #DB_NUMBER; END_IF;
   IF #_w1 AND #ANY_MCH_CYCLE_RUN THEN "DB428_OPERATOR_HELP".HELP_OPERATOR_269 := TRUE; END_IF;
   IF #_w1 AND NOT #MODE_GROUP_BA_DB.CHANGE_ENABLE_INPUT THEN "M_DUMMY_OUT" := TRUE; END_IF;
END_REGION

REGION Network 6: CHANGE MODE INITIAL CONDITIONS
   RUNG wire#powerrail
      Contact( "M_ONE" )
      Coil( #MODE_GROUP_BA_DB.CHANGE_INITIAL_CONDITIONS )
   END_RUNG
   // the same network as SCL:
   #MODE_GROUP_BA_DB.CHANGE_INITIAL_CONDITIONS := "M_ONE";
END_REGION

REGION Network 7: BA1 MODE REQUEST
   RUNG wire#powerrail
      Contact( #MODE_GROUP_BA_DB.BA1_INPUT )
      I_Contact( #MODE_GROUP_BA_DB.BA2_INPUT )
      I_Contact( #MODE_GROUP_BA_DB.BA3_INPUT )
      I_Contact( #MODE_GROUP_BA_DB.BA5_INPUT )
      I_Contact( #MODE_GROUP_BA_DB.BA1_SELECTED )
      Coil( #MODE_GROUP_BA_DB.BA1_REQUEST )
   END_RUNG
   // the same network as SCL:
   #MODE_GROUP_BA_DB.BA1_REQUEST := #MODE_GROUP_BA_DB.BA1_INPUT AND NOT #MODE_GROUP_BA_DB.BA2_INPUT AND NOT #MODE_GROUP_BA_DB.BA3_INPUT AND NOT #MODE_GROUP_BA_DB.BA5_INPUT AND NOT #MODE_GROUP_BA_DB.BA1_SELECTED;
END_REGION

REGION Network 8: BA2 MODE REQUEST
   RUNG wire#powerrail
      Contact( #MODE_GROUP_BA_DB.BA2_INPUT )
      I_Contact( #MODE_GROUP_BA_DB.BA1_INPUT )
      I_Contact( #MODE_GROUP_BA_DB.BA3_INPUT )
      I_Contact( #MODE_GROUP_BA_DB.BA5_INPUT )
      I_Contact( #MODE_GROUP_BA_DB.BA2_SELECTED )
      Coil( #MODE_GROUP_BA_DB.BA2_REQUEST )
   END_RUNG
   // the same network as SCL:
   #MODE_GROUP_BA_DB.BA2_REQUEST := #MODE_GROUP_BA_DB.BA2_INPUT AND NOT #MODE_GROUP_BA_DB.BA1_INPUT AND NOT #MODE_GROUP_BA_DB.BA3_INPUT AND NOT #MODE_GROUP_BA_DB.BA5_INPUT AND NOT #MODE_GROUP_BA_DB.BA2_SELECTED;
END_REGION

REGION Network 9: BA3 MODE REQUEST
   RUNG wire#powerrail
      Contact( #MODE_GROUP_BA_DB.BA3_INPUT )
      I_Contact( #MODE_GROUP_BA_DB.BA1_INPUT )
      I_Contact( #MODE_GROUP_BA_DB.BA2_INPUT )
      I_Contact( #MODE_GROUP_BA_DB.BA5_INPUT )
      I_Contact( #MODE_GROUP_BA_DB.BA3_SELECTED )
      Coil( #MODE_GROUP_BA_DB.BA3_REQUEST )
   END_RUNG
   // the same network as SCL:
   #MODE_GROUP_BA_DB.BA3_REQUEST := #MODE_GROUP_BA_DB.BA3_INPUT AND NOT #MODE_GROUP_BA_DB.BA1_INPUT AND NOT #MODE_GROUP_BA_DB.BA2_INPUT AND NOT #MODE_GROUP_BA_DB.BA5_INPUT AND NOT #MODE_GROUP_BA_DB.BA3_SELECTED;
END_REGION

REGION Network 10: BA5 MODE REQUEST
   RUNG wire#powerrail
      Contact( #MODE_GROUP_BA_DB.BA5_INPUT )
      I_Contact( #MODE_GROUP_BA_DB.BA1_INPUT )
      I_Contact( #MODE_GROUP_BA_DB.BA2_INPUT )
      I_Contact( #MODE_GROUP_BA_DB.BA3_INPUT )
      I_Contact( #MODE_GROUP_BA_DB.BA5_SELECTED )
      Coil( #MODE_GROUP_BA_DB.BA5_REQUEST )
   END_RUNG
   // the same network as SCL:
   #MODE_GROUP_BA_DB.BA5_REQUEST := #MODE_GROUP_BA_DB.BA5_INPUT AND NOT #MODE_GROUP_BA_DB.BA1_INPUT AND NOT #MODE_GROUP_BA_DB.BA2_INPUT AND NOT #MODE_GROUP_BA_DB.BA3_INPUT AND NOT #MODE_GROUP_BA_DB.BA5_SELECTED;
END_REGION

REGION Network 11: MODE SELECTED MEMORIES
   RUNG wire#powerrail
      Contact( #O_BYTE_0.MODE_SELECTED_MEMORY )
      Contact( #ANY_MCH_CYCLE_RUN )
      wire#w1
      Contact( #MODE_GROUP_BA_DB.BA1_REQUEST )
      I_Contact( #MODE_GROUP_BA_DB.BA2_SELECTED_MEMORY )
      I_Contact( #MODE_GROUP_BA_DB.BA3_SELECTED_MEMORY )
      I_Contact( #MODE_GROUP_BA_DB.BA5_SELECTED_MEMORY )
      S_Coil( #MODE_GROUP_BA_DB.BA1_SELECTED_MEMORY )
   END_RUNG
   RUNG wire#w1
      Contact( #MODE_GROUP_BA_DB.BA2_REQUEST )
      I_Contact( #MODE_GROUP_BA_DB.BA1_SELECTED_MEMORY )
      I_Contact( #MODE_GROUP_BA_DB.BA3_SELECTED_MEMORY )
      I_Contact( #MODE_GROUP_BA_DB.BA5_SELECTED_MEMORY )
      S_Coil( #MODE_GROUP_BA_DB.BA2_SELECTED_MEMORY )
   END_RUNG
   RUNG wire#w1
      Contact( #MODE_GROUP_BA_DB.BA3_REQUEST )
      I_Contact( #MODE_GROUP_BA_DB.BA1_SELECTED_MEMORY )
      I_Contact( #MODE_GROUP_BA_DB.BA2_SELECTED_MEMORY )
      I_Contact( #MODE_GROUP_BA_DB.BA5_SELECTED_MEMORY )
      S_Coil( #MODE_GROUP_BA_DB.BA3_SELECTED_MEMORY )
   END_RUNG
   RUNG wire#w1
      Contact( #MODE_GROUP_BA_DB.BA5_REQUEST )
      I_Contact( #MODE_GROUP_BA_DB.BA1_SELECTED_MEMORY )
      I_Contact( #MODE_GROUP_BA_DB.BA2_SELECTED_MEMORY )
      I_Contact( #MODE_GROUP_BA_DB.BA3_SELECTED_MEMORY )
      S_Coil( #MODE_GROUP_BA_DB.BA5_SELECTED_MEMORY )
   END_RUNG
   // the same network as SCL:
   #_w1 := #O_BYTE_0.MODE_SELECTED_MEMORY AND #ANY_MCH_CYCLE_RUN;
   IF #_w1 AND #MODE_GROUP_BA_DB.BA1_REQUEST AND NOT #MODE_GROUP_BA_DB.BA2_SELECTED_MEMORY AND NOT #MODE_GROUP_BA_DB.BA3_SELECTED_MEMORY AND NOT #MODE_GROUP_BA_DB.BA5_SELECTED_MEMORY THEN
       #MODE_GROUP_BA_DB.BA1_SELECTED_MEMORY := TRUE;
   END_IF;
   IF #_w1 AND #MODE_GROUP_BA_DB.BA2_REQUEST AND NOT #MODE_GROUP_BA_DB.BA1_SELECTED_MEMORY AND NOT #MODE_GROUP_BA_DB.BA3_SELECTED_MEMORY AND NOT #MODE_GROUP_BA_DB.BA5_SELECTED_MEMORY THEN
       #MODE_GROUP_BA_DB.BA2_SELECTED_MEMORY := TRUE;
   END_IF;
   IF #_w1 AND #MODE_GROUP_BA_DB.BA3_REQUEST AND NOT #MODE_GROUP_BA_DB.BA1_SELECTED_MEMORY AND NOT #MODE_GROUP_BA_DB.BA2_SELECTED_MEMORY AND NOT #MODE_GROUP_BA_DB.BA5_SELECTED_MEMORY THEN
       #MODE_GROUP_BA_DB.BA3_SELECTED_MEMORY := TRUE;
   END_IF;
   IF #_w1 AND #MODE_GROUP_BA_DB.BA5_REQUEST AND NOT #MODE_GROUP_BA_DB.BA1_SELECTED_MEMORY AND NOT #MODE_GROUP_BA_DB.BA2_SELECTED_MEMORY AND NOT #MODE_GROUP_BA_DB.BA3_SELECTED_MEMORY THEN
       #MODE_GROUP_BA_DB.BA5_SELECTED_MEMORY := TRUE;
   END_IF;
END_REGION

REGION Network 12: BA1 MODE SELECTED
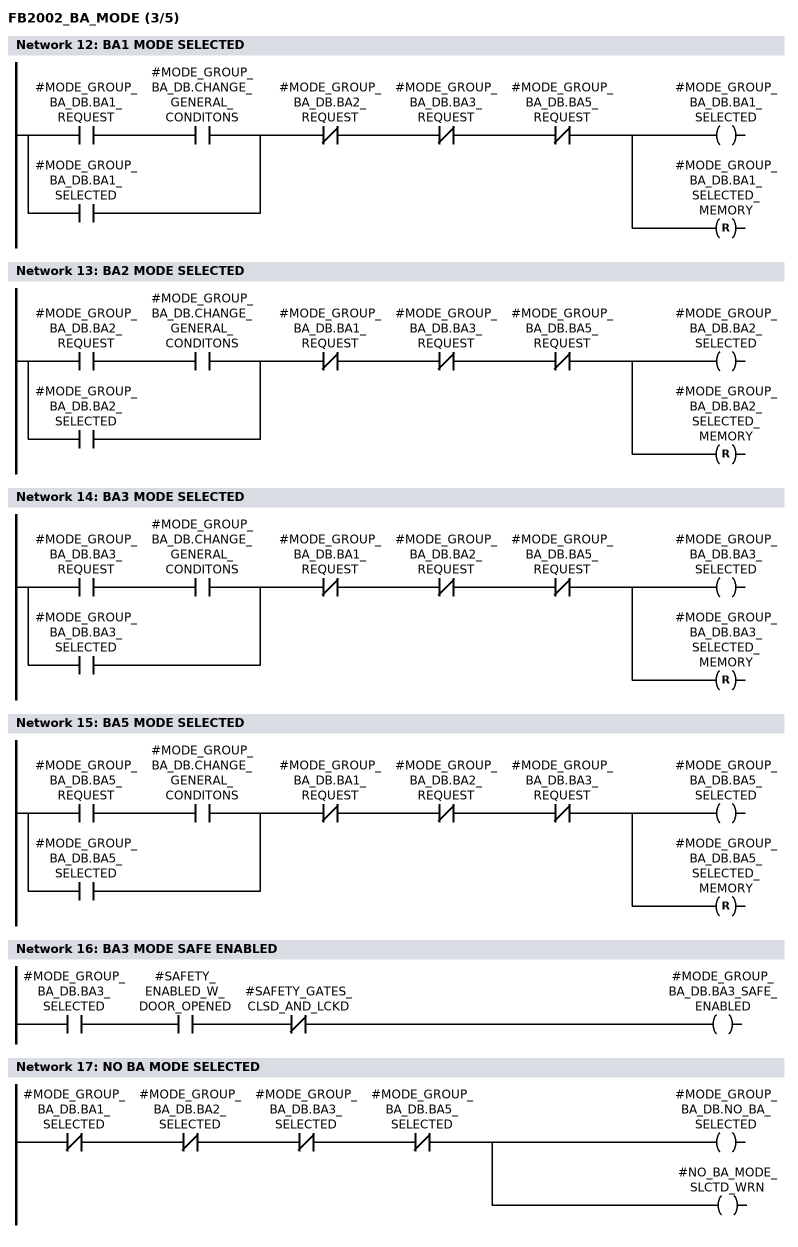
   RUNG wire#powerrail
      Contact( #MODE_GROUP_BA_DB.BA1_REQUEST )
      Contact( #MODE_GROUP_BA_DB.CHANGE_GENERAL_CONDITONS )
      wire#w1
      I_Contact( #MODE_GROUP_BA_DB.BA2_REQUEST )
      I_Contact( #MODE_GROUP_BA_DB.BA3_REQUEST )
      I_Contact( #MODE_GROUP_BA_DB.BA5_REQUEST )
      wire#w2
      Coil( #MODE_GROUP_BA_DB.BA1_SELECTED )
   END_RUNG
   RUNG wire#powerrail
      Contact( #MODE_GROUP_BA_DB.BA1_SELECTED )
   END_RUNG wire#w1
   RUNG wire#w2
      R_Coil( #MODE_GROUP_BA_DB.BA1_SELECTED_MEMORY )
   END_RUNG
   // the same network as SCL:
   #MODE_GROUP_BA_DB.BA1_SELECTED := ((#MODE_GROUP_BA_DB.BA1_REQUEST AND #MODE_GROUP_BA_DB.CHANGE_GENERAL_CONDITONS) OR #MODE_GROUP_BA_DB.BA1_SELECTED) AND NOT #MODE_GROUP_BA_DB.BA2_REQUEST AND NOT #MODE_GROUP_BA_DB.BA3_REQUEST AND NOT #MODE_GROUP_BA_DB.BA5_REQUEST;
   IF #MODE_GROUP_BA_DB.BA1_SELECTED THEN #MODE_GROUP_BA_DB.BA1_SELECTED_MEMORY := FALSE; END_IF;
END_REGION

REGION Network 13: BA2 MODE SELECTED
   RUNG wire#powerrail
      Contact( #MODE_GROUP_BA_DB.BA2_REQUEST )
      Contact( #MODE_GROUP_BA_DB.CHANGE_GENERAL_CONDITONS )
      wire#w1
      I_Contact( #MODE_GROUP_BA_DB.BA1_REQUEST )
      I_Contact( #MODE_GROUP_BA_DB.BA3_REQUEST )
      I_Contact( #MODE_GROUP_BA_DB.BA5_REQUEST )
      wire#w2
      Coil( #MODE_GROUP_BA_DB.BA2_SELECTED )
   END_RUNG
   RUNG wire#powerrail
      Contact( #MODE_GROUP_BA_DB.BA2_SELECTED )
   END_RUNG wire#w1
   RUNG wire#w2
      R_Coil( #MODE_GROUP_BA_DB.BA2_SELECTED_MEMORY )
   END_RUNG
   // the same network as SCL:
   #MODE_GROUP_BA_DB.BA2_SELECTED := ((#MODE_GROUP_BA_DB.BA2_REQUEST AND #MODE_GROUP_BA_DB.CHANGE_GENERAL_CONDITONS) OR #MODE_GROUP_BA_DB.BA2_SELECTED) AND NOT #MODE_GROUP_BA_DB.BA1_REQUEST AND NOT #MODE_GROUP_BA_DB.BA3_REQUEST AND NOT #MODE_GROUP_BA_DB.BA5_REQUEST;
   IF #MODE_GROUP_BA_DB.BA2_SELECTED THEN #MODE_GROUP_BA_DB.BA2_SELECTED_MEMORY := FALSE; END_IF;
END_REGION

REGION Network 14: BA3 MODE SELECTED
   RUNG wire#powerrail
      Contact( #MODE_GROUP_BA_DB.BA3_REQUEST )
      Contact( #MODE_GROUP_BA_DB.CHANGE_GENERAL_CONDITONS )
      wire#w1
      I_Contact( #MODE_GROUP_BA_DB.BA1_REQUEST )
      I_Contact( #MODE_GROUP_BA_DB.BA2_REQUEST )
      I_Contact( #MODE_GROUP_BA_DB.BA5_REQUEST )
      wire#w2
      Coil( #MODE_GROUP_BA_DB.BA3_SELECTED )
   END_RUNG
   RUNG wire#powerrail
      Contact( #MODE_GROUP_BA_DB.BA3_SELECTED )
   END_RUNG wire#w1
   RUNG wire#w2
      R_Coil( #MODE_GROUP_BA_DB.BA3_SELECTED_MEMORY )
   END_RUNG
   // the same network as SCL:
   #MODE_GROUP_BA_DB.BA3_SELECTED := ((#MODE_GROUP_BA_DB.BA3_REQUEST AND #MODE_GROUP_BA_DB.CHANGE_GENERAL_CONDITONS) OR #MODE_GROUP_BA_DB.BA3_SELECTED) AND NOT #MODE_GROUP_BA_DB.BA1_REQUEST AND NOT #MODE_GROUP_BA_DB.BA2_REQUEST AND NOT #MODE_GROUP_BA_DB.BA5_REQUEST;
   IF #MODE_GROUP_BA_DB.BA3_SELECTED THEN #MODE_GROUP_BA_DB.BA3_SELECTED_MEMORY := FALSE; END_IF;
END_REGION

REGION Network 15: BA5 MODE SELECTED
   RUNG wire#powerrail
      Contact( #MODE_GROUP_BA_DB.BA5_REQUEST )
      Contact( #MODE_GROUP_BA_DB.CHANGE_GENERAL_CONDITONS )
      wire#w1
      I_Contact( #MODE_GROUP_BA_DB.BA1_REQUEST )
      I_Contact( #MODE_GROUP_BA_DB.BA2_REQUEST )
      I_Contact( #MODE_GROUP_BA_DB.BA3_REQUEST )
      wire#w2
      Coil( #MODE_GROUP_BA_DB.BA5_SELECTED )
   END_RUNG
   RUNG wire#powerrail
      Contact( #MODE_GROUP_BA_DB.BA5_SELECTED )
   END_RUNG wire#w1
   RUNG wire#w2
      R_Coil( #MODE_GROUP_BA_DB.BA5_SELECTED_MEMORY )
   END_RUNG
   // the same network as SCL:
   #MODE_GROUP_BA_DB.BA5_SELECTED := ((#MODE_GROUP_BA_DB.BA5_REQUEST AND #MODE_GROUP_BA_DB.CHANGE_GENERAL_CONDITONS) OR #MODE_GROUP_BA_DB.BA5_SELECTED) AND NOT #MODE_GROUP_BA_DB.BA1_REQUEST AND NOT #MODE_GROUP_BA_DB.BA2_REQUEST AND NOT #MODE_GROUP_BA_DB.BA3_REQUEST;
   IF #MODE_GROUP_BA_DB.BA5_SELECTED THEN #MODE_GROUP_BA_DB.BA5_SELECTED_MEMORY := FALSE; END_IF;
END_REGION

REGION Network 16: BA3 MODE SAFE ENABLED
   RUNG wire#powerrail
      Contact( #MODE_GROUP_BA_DB.BA3_SELECTED )
      Contact( #SAFETY_ENABLED_W_DOOR_OPENED )
      I_Contact( #SAFETY_GATES_CLSD_AND_LCKD )
      Coil( #MODE_GROUP_BA_DB.BA3_SAFE_ENABLED )
   END_RUNG
   // the same network as SCL:
   #MODE_GROUP_BA_DB.BA3_SAFE_ENABLED := #MODE_GROUP_BA_DB.BA3_SELECTED AND #SAFETY_ENABLED_W_DOOR_OPENED AND NOT #SAFETY_GATES_CLSD_AND_LCKD;
END_REGION

REGION Network 17: NO BA MODE SELECTED
   RUNG wire#powerrail
      I_Contact( #MODE_GROUP_BA_DB.BA1_SELECTED )
      I_Contact( #MODE_GROUP_BA_DB.BA2_SELECTED )
      I_Contact( #MODE_GROUP_BA_DB.BA3_SELECTED )
      I_Contact( #MODE_GROUP_BA_DB.BA5_SELECTED )
      wire#w1
      Coil( #MODE_GROUP_BA_DB.NO_BA_SELECTED )
   END_RUNG
   RUNG wire#w1
      Coil( #NO_BA_MODE_SLCTD_WRN )
   END_RUNG
   // the same network as SCL:
   #MODE_GROUP_BA_DB.NO_BA_SELECTED := NOT #MODE_GROUP_BA_DB.BA1_SELECTED AND NOT #MODE_GROUP_BA_DB.BA2_SELECTED AND NOT #MODE_GROUP_BA_DB.BA3_SELECTED AND NOT #MODE_GROUP_BA_DB.BA5_SELECTED;
   #NO_BA_MODE_SLCTD_WRN := #MODE_GROUP_BA_DB.NO_BA_SELECTED;
END_REGION

REGION Network 18: CHANGE TO BA1 MODE ALARM
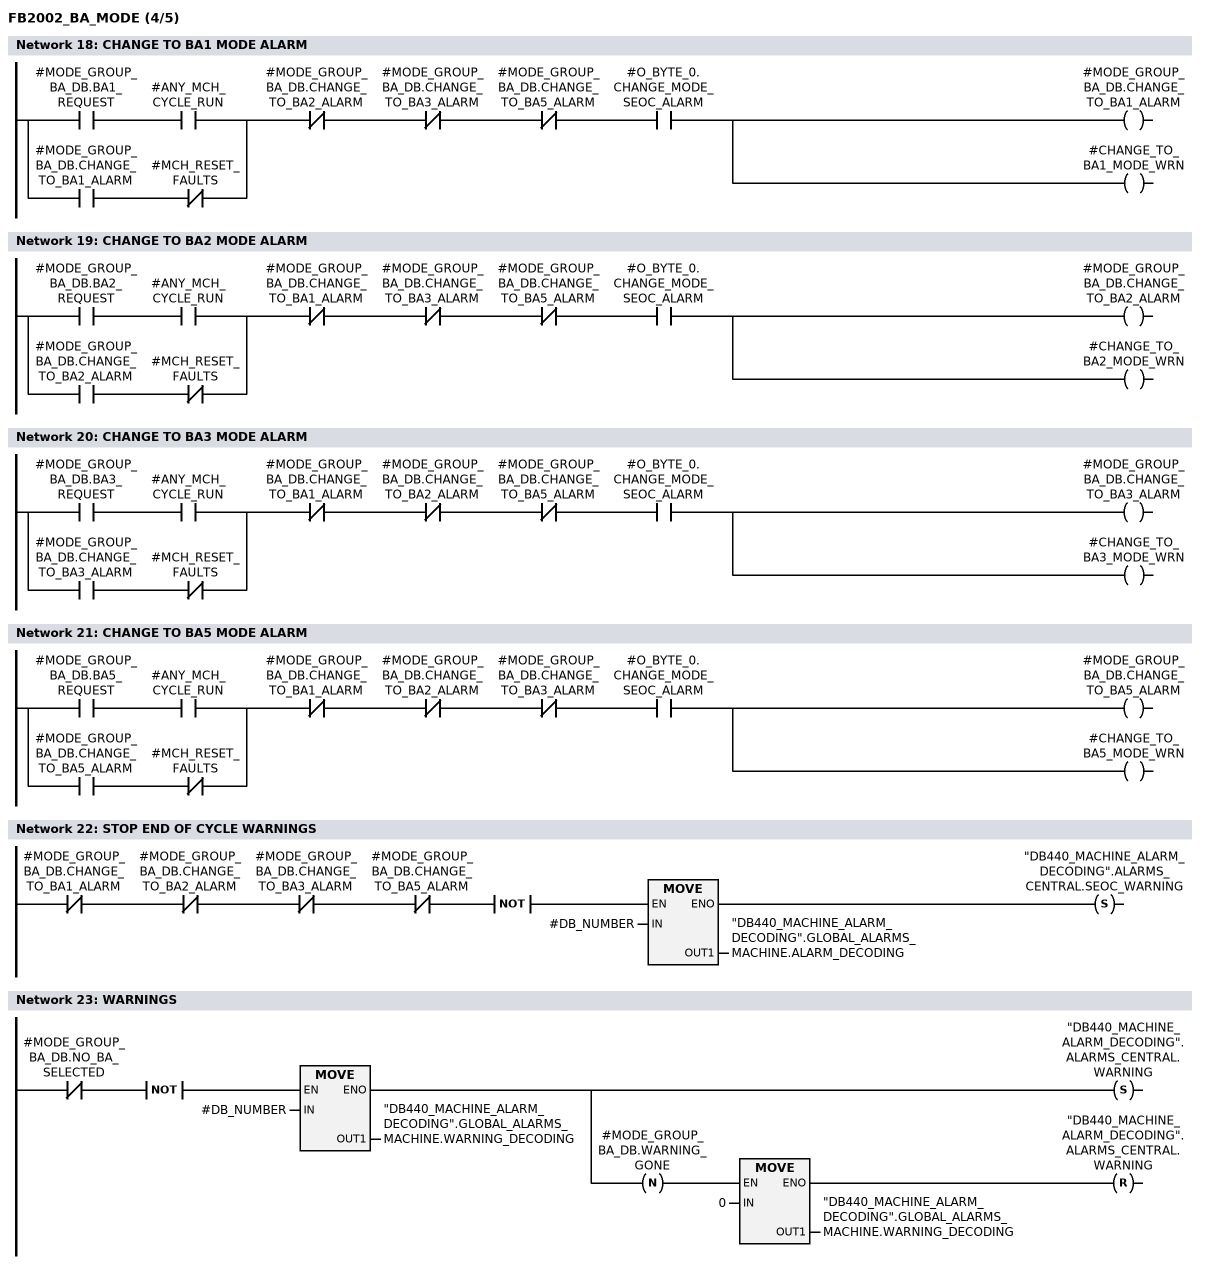
   RUNG wire#powerrail
      Contact( #MODE_GROUP_BA_DB.BA1_REQUEST )
      Contact( #ANY_MCH_CYCLE_RUN )
      wire#w1
      I_Contact( #MODE_GROUP_BA_DB.CHANGE_TO_BA2_ALARM )
      I_Contact( #MODE_GROUP_BA_DB.CHANGE_TO_BA3_ALARM )
      I_Contact( #MODE_GROUP_BA_DB.CHANGE_TO_BA5_ALARM )
      Contact( #O_BYTE_0.CHANGE_MODE_SEOC_ALARM )
      wire#w2
      Coil( #MODE_GROUP_BA_DB.CHANGE_TO_BA1_ALARM )
   END_RUNG
   RUNG wire#powerrail
      Contact( #MODE_GROUP_BA_DB.CHANGE_TO_BA1_ALARM )
      I_Contact( #MCH_RESET_FAULTS )
   END_RUNG wire#w1
   RUNG wire#w2
      Coil( #CHANGE_TO_BA1_MODE_WRN )
   END_RUNG
   // the same network as SCL:
   #MODE_GROUP_BA_DB.CHANGE_TO_BA1_ALARM := ((#MODE_GROUP_BA_DB.BA1_REQUEST AND #ANY_MCH_CYCLE_RUN) OR (#MODE_GROUP_BA_DB.CHANGE_TO_BA1_ALARM AND NOT #MCH_RESET_FAULTS)) AND NOT #MODE_GROUP_BA_DB.CHANGE_TO_BA2_ALARM AND NOT #MODE_GROUP_BA_DB.CHANGE_TO_BA3_ALARM AND NOT #MODE_GROUP_BA_DB.CHANGE_TO_BA5_ALARM AND #O_BYTE_0.CHANGE_MODE_SEOC_ALARM;
   #CHANGE_TO_BA1_MODE_WRN := #MODE_GROUP_BA_DB.CHANGE_TO_BA1_ALARM;
END_REGION

REGION Network 19: CHANGE TO BA2 MODE ALARM
   RUNG wire#powerrail
      Contact( #MODE_GROUP_BA_DB.BA2_REQUEST )
      Contact( #ANY_MCH_CYCLE_RUN )
      wire#w1
      I_Contact( #MODE_GROUP_BA_DB.CHANGE_TO_BA1_ALARM )
      I_Contact( #MODE_GROUP_BA_DB.CHANGE_TO_BA3_ALARM )
      I_Contact( #MODE_GROUP_BA_DB.CHANGE_TO_BA5_ALARM )
      Contact( #O_BYTE_0.CHANGE_MODE_SEOC_ALARM )
      wire#w2
      Coil( #MODE_GROUP_BA_DB.CHANGE_TO_BA2_ALARM )
   END_RUNG
   RUNG wire#powerrail
      Contact( #MODE_GROUP_BA_DB.CHANGE_TO_BA2_ALARM )
      I_Contact( #MCH_RESET_FAULTS )
   END_RUNG wire#w1
   RUNG wire#w2
      Coil( #CHANGE_TO_BA2_MODE_WRN )
   END_RUNG
   // the same network as SCL:
   #MODE_GROUP_BA_DB.CHANGE_TO_BA2_ALARM := ((#MODE_GROUP_BA_DB.BA2_REQUEST AND #ANY_MCH_CYCLE_RUN) OR (#MODE_GROUP_BA_DB.CHANGE_TO_BA2_ALARM AND NOT #MCH_RESET_FAULTS)) AND NOT #MODE_GROUP_BA_DB.CHANGE_TO_BA1_ALARM AND NOT #MODE_GROUP_BA_DB.CHANGE_TO_BA3_ALARM AND NOT #MODE_GROUP_BA_DB.CHANGE_TO_BA5_ALARM AND #O_BYTE_0.CHANGE_MODE_SEOC_ALARM;
   #CHANGE_TO_BA2_MODE_WRN := #MODE_GROUP_BA_DB.CHANGE_TO_BA2_ALARM;
END_REGION

